REGION Network 3: Cylinder Selection ( Domestic / Commercial )
   // We have to receive from FIFO Entry-
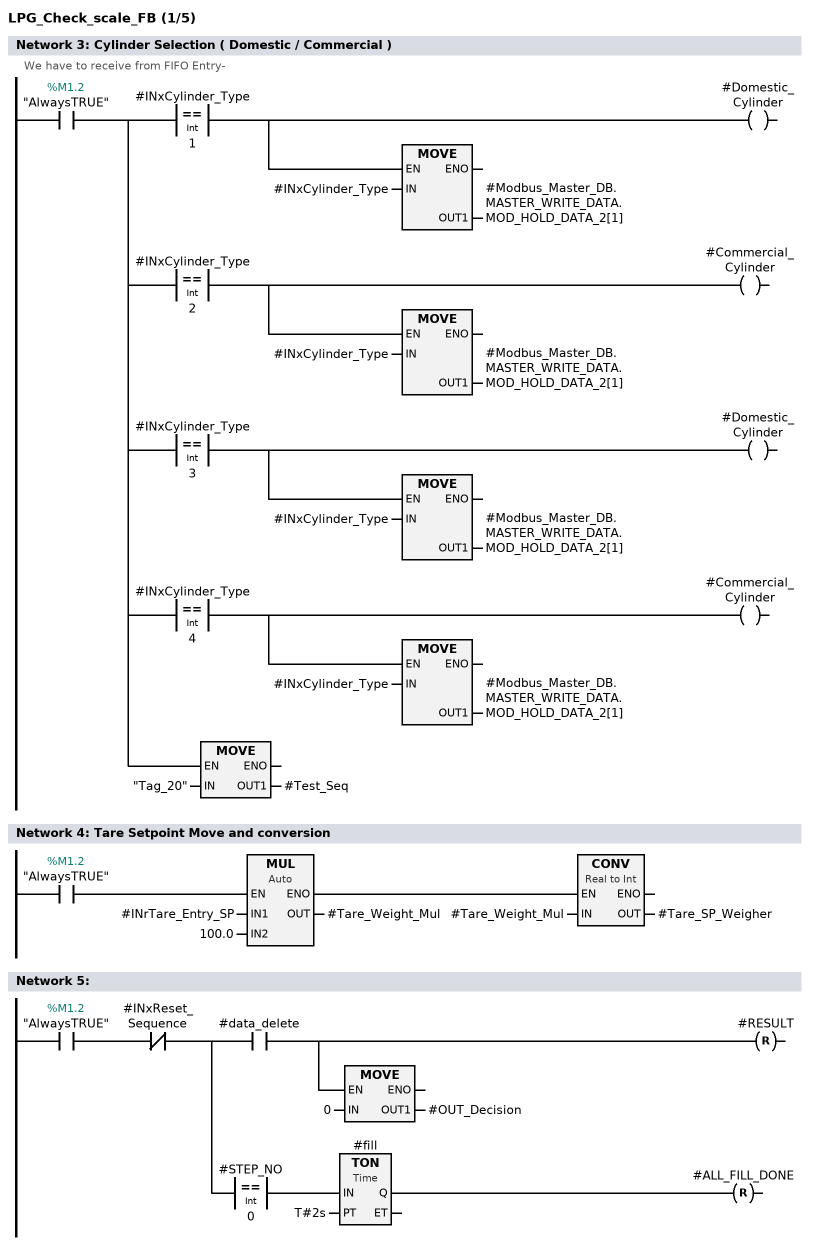
   RUNG wire#powerrail
      Contact( "AlwaysTRUE" )
      wire#w1
      { S7_Templates := "SrcType := Int" } EQ_Contact(in1 := #INxCylinder_Type, in2 := 1)
      wire#w2
      Coil( #Domestic_Cylinder )
   END_RUNG
   RUNG wire#w2
      Move(in := #INxCylinder_Type, out1 => #Modbus_Master_DB.MASTER_WRITE_DATA.MOD_HOLD_DATA_2[1])
   END_RUNG
   RUNG wire#w1
      { S7_Templates := "SrcType := Int" } EQ_Contact(in1 := #INxCylinder_Type, in2 := 2)
      wire#w3
      Coil( #Commercial_Cylinder )
   END_RUNG
   RUNG wire#w3
      Move(in := #INxCylinder_Type, out1 => #Modbus_Master_DB.MASTER_WRITE_DATA.MOD_HOLD_DATA_2[1])
   END_RUNG
   RUNG wire#w1
      { S7_Templates := "SrcType := Int" } EQ_Contact(in1 := #INxCylinder_Type, in2 := 3)
      wire#w4
      Coil( #Domestic_Cylinder )
   END_RUNG
   RUNG wire#w4
      Move(in := #INxCylinder_Type, out1 => #Modbus_Master_DB.MASTER_WRITE_DATA.MOD_HOLD_DATA_2[1])
   END_RUNG
   RUNG wire#w1
      { S7_Templates := "SrcType := Int" } EQ_Contact(in1 := #INxCylinder_Type, in2 := 4)
      wire#w5
      Coil( #Commercial_Cylinder )
   END_RUNG
   RUNG wire#w5
      Move(in := #INxCylinder_Type, out1 => #Modbus_Master_DB.MASTER_WRITE_DATA.MOD_HOLD_DATA_2[1])
   END_RUNG
   RUNG wire#w1
      Move(in := "Tag_20", out1 => #Test_Seq)
   END_RUNG
   // the same network as SCL:
   #Domestic_Cylinder := "AlwaysTRUE" AND (#INxCylinder_Type = 1);
   IF #Domestic_Cylinder THEN
       #Modbus_Master_DB.MASTER_WRITE_DATA.MOD_HOLD_DATA_2[1] := #INxCylinder_Type;
   END_IF;
   #Commercial_Cylinder := "AlwaysTRUE" AND (#INxCylinder_Type = 2);
   IF #Commercial_Cylinder THEN
       #Modbus_Master_DB.MASTER_WRITE_DATA.MOD_HOLD_DATA_2[1] := #INxCylinder_Type;
   END_IF;
   #Domestic_Cylinder := "AlwaysTRUE" AND (#INxCylinder_Type = 3);
   IF #Domestic_Cylinder THEN
       #Modbus_Master_DB.MASTER_WRITE_DATA.MOD_HOLD_DATA_2[1] := #INxCylinder_Type;
   END_IF;
   #Commercial_Cylinder := "AlwaysTRUE" AND (#INxCylinder_Type = 4);
   IF #Commercial_Cylinder THEN
       #Modbus_Master_DB.MASTER_WRITE_DATA.MOD_HOLD_DATA_2[1] := #INxCylinder_Type;
   END_IF;
   IF "AlwaysTRUE" THEN #Test_Seq := "Tag_20"; END_IF;
END_REGION

REGION Network 4: Tare Setpoint Move and conversion
   RUNG wire#powerrail
      Contact( "AlwaysTRUE" )
      Mul(in1 := #INrTare_Entry_SP, in2 := 100.0, out => #Tare_Weight_Mul)
      { S7_Templates := "[SrcType := Real, DestType := Int]" } Convert(in := #Tare_Weight_Mul, out => #Tare_SP_Weigher)
   END_RUNG
   // the same network as SCL:
   IF "AlwaysTRUE" THEN
       #Tare_Weight_Mul := #INrTare_Entry_SP * 100.0;
       #Tare_SP_Weigher := REAL_TO_INT(#Tare_Weight_Mul);
   END_IF;
END_REGION

REGION Network 5
   RUNG wire#powerrail
      Contact( "AlwaysTRUE" )
      I_Contact( #INxReset_Sequence )
      wire#w1
      Contact( #data_delete )
      wire#w2
      R_Coil( #RESULT )
   END_RUNG
   RUNG wire#w2
      Move(in := 0, out1 => #OUT_Decision)
   END_RUNG
   RUNG wire#w1
      { S7_Templates := "SrcType := Int" } EQ_Contact(in1 := #STEP_NO, in2 := 0)
      { S7_Templates := "time_type := Time" } #fill.TON(pt := T#2s, et =>)
      R_Coil( #ALL_FILL_DONE )
   END_RUNG
   // the same network as SCL:
   #_w1 := "AlwaysTRUE" AND NOT #INxReset_Sequence;
   IF #_w1 AND #data_delete THEN
       #RESULT := FALSE;
       #OUT_Decision := 0;
   END_IF;
   #fill(IN := #_w1 AND (#STEP_NO = 0), PT := T#2s);   // TON
   IF #fill.Q THEN #ALL_FILL_DONE := FALSE; END_IF;
END_REGION

REGION Network 6: Cylinder Selection
   // Cylinder Selection will write the logic later
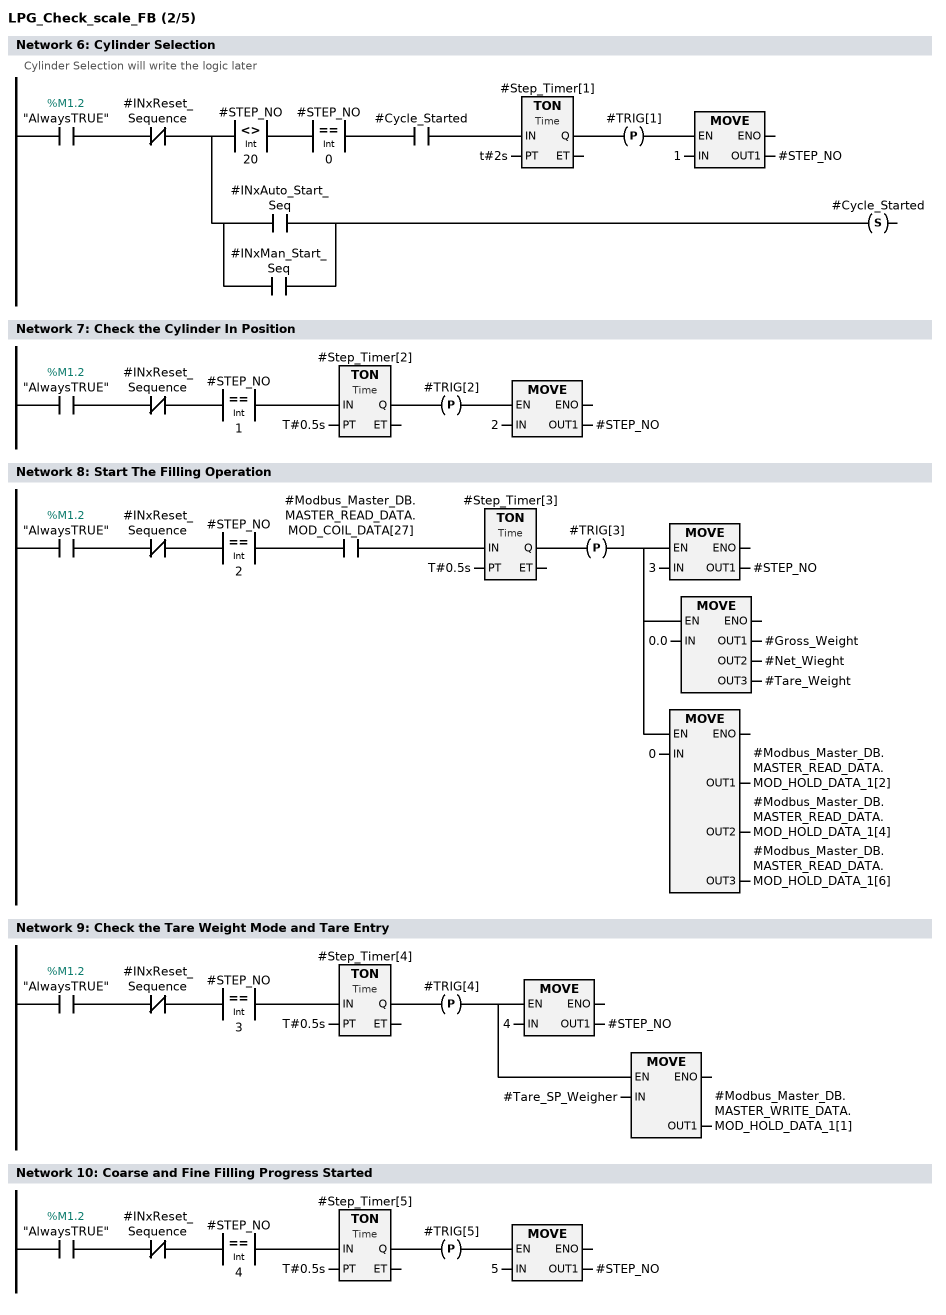
   RUNG wire#powerrail
      Contact( "AlwaysTRUE" )
      I_Contact( #INxReset_Sequence )
      wire#w1
      { S7_Templates := "SrcType := Int" } NE_Contact(in1 := #STEP_NO, in2 := 20)
      { S7_Templates := "SrcType := Int" } EQ_Contact(in1 := #STEP_NO, in2 := 0)
      Contact( #Cycle_Started )
      { S7_Templates := "time_type := Time" } #Step_Timer[1].TON(pt := t#2s, et =>)
      P_Trig( #TRIG[1] )
      Move(in := 1, out1 => #STEP_NO)
   END_RUNG
   RUNG wire#w1
      Contact( #INxAuto_Start_Seq )
      wire#w2
      S_Coil( #Cycle_Started )
   END_RUNG
   RUNG wire#w1
      Contact( #INxMan_Start_Seq )
   END_RUNG wire#w2
   // the same network as SCL:
   #_w1 := "AlwaysTRUE" AND NOT #INxReset_Sequence;
   #Step_Timer[1].TON(IN := #_w1 AND (#STEP_NO <> 20) AND (#STEP_NO = 0) AND #Cycle_Started, PT := t#2s);
   #_w2 := #Step_Timer[1].Q AND NOT #TRIG[1];   // rising edge
   #TRIG[1] := #Step_Timer[1].Q;
   IF #_w2 THEN #STEP_NO := 1; END_IF;
   IF #_w1 AND (#INxAuto_Start_Seq OR #INxMan_Start_Seq) THEN #Cycle_Started := TRUE; END_IF;
END_REGION

REGION Network 7: Check the Cylinder In Position
   RUNG wire#powerrail
      Contact( "AlwaysTRUE" )
      I_Contact( #INxReset_Sequence )
      { S7_Templates := "SrcType := Int" } EQ_Contact(in1 := #STEP_NO, in2 := 1)
      { S7_Templates := "time_type := Time" } #Step_Timer[2].TON(pt := T#0.5s, et =>)
      P_Trig( #TRIG[2] )
      Move(in := 2, out1 => #STEP_NO)
   END_RUNG
   // the same network as SCL:
   #Step_Timer[2].TON(IN := "AlwaysTRUE" AND NOT #INxReset_Sequence AND (#STEP_NO = 1), PT := T#0.5s);
   #_w1 := #Step_Timer[2].Q AND NOT #TRIG[2];   // rising edge
   #TRIG[2] := #Step_Timer[2].Q;
   IF #_w1 THEN #STEP_NO := 2; END_IF;
END_REGION

REGION Network 8: Start The Filling Operation
   RUNG wire#powerrail
      Contact( "AlwaysTRUE" )
      I_Contact( #INxReset_Sequence )
      { S7_Templates := "SrcType := Int" } EQ_Contact(in1 := #STEP_NO, in2 := 2)
      Contact( #Modbus_Master_DB.MASTER_READ_DATA.MOD_COIL_DATA[27] )
      { S7_Templates := "time_type := Time" } #Step_Timer[3].TON(pt := T#0.5s, et =>)
      P_Trig( #TRIG[3] )
      wire#w1
      Move(in := 3, out1 => #STEP_NO)
   END_RUNG
   RUNG wire#w1
      Move(in := 0.0, out1 => #Gross_Weight, out2 => #Net_Wieght, out3 => #Tare_Weight)
   END_RUNG
   RUNG wire#w1
      Move(in := 0, out1 => #Modbus_Master_DB.MASTER_READ_DATA.MOD_HOLD_DATA_1[2], out2 => #Modbus_Master_DB.MASTER_READ_DATA.MOD_HOLD_DATA_1[4], out3 => #Modbus_Master_DB.MASTER_READ_DATA.MOD_HOLD_DATA_1[6])
   END_RUNG
   // the same network as SCL:
   #Step_Timer[3].TON(IN := "AlwaysTRUE" AND NOT #INxReset_Sequence AND (#STEP_NO = 2) AND #Modbus_Master_DB.MASTER_READ_DATA.MOD_COIL_DATA[27],
                      PT := T#0.5s);
   #_w1 := #Step_Timer[3].Q AND NOT #TRIG[3];   // rising edge
   #TRIG[3] := #Step_Timer[3].Q;
   IF #_w1 THEN
       #STEP_NO := 3;
       #Gross_Weight := 0.0;
       #Net_Wieght := 0.0;
       #Tare_Weight := 0.0;
       #Modbus_Master_DB.MASTER_READ_DATA.MOD_HOLD_DATA_1[2] := 0;
       #Modbus_Master_DB.MASTER_READ_DATA.MOD_HOLD_DATA_1[4] := 0;
       #Modbus_Master_DB.MASTER_READ_DATA.MOD_HOLD_DATA_1[6] := 0;
   END_IF;
END_REGION

REGION Network 9: Check the Tare Weight Mode and Tare Entry
   RUNG wire#powerrail
      Contact( "AlwaysTRUE" )
      I_Contact( #INxReset_Sequence )
      { S7_Templates := "SrcType := Int" } EQ_Contact(in1 := #STEP_NO, in2 := 3)
      { S7_Templates := "time_type := Time" } #Step_Timer[4].TON(pt := T#0.5s, et =>)
      P_Trig( #TRIG[4] )
      wire#w1
      Move(in := 4, out1 => #STEP_NO)
   END_RUNG
   RUNG wire#w1
      Move(in := #Tare_SP_Weigher, out1 => #Modbus_Master_DB.MASTER_WRITE_DATA.MOD_HOLD_DATA_1[1])
   END_RUNG
   // the same network as SCL:
   #Step_Timer[4].TON(IN := "AlwaysTRUE" AND NOT #INxReset_Sequence AND (#STEP_NO = 3), PT := T#0.5s);
   #_w1 := #Step_Timer[4].Q AND NOT #TRIG[4];   // rising edge
   #TRIG[4] := #Step_Timer[4].Q;
   IF #_w1 THEN
       #STEP_NO := 4;
       #Modbus_Master_DB.MASTER_WRITE_DATA.MOD_HOLD_DATA_1[1] := #Tare_SP_Weigher;
   END_IF;
END_REGION

REGION Network 10: Coarse and Fine Filling Progress Started
   RUNG wire#powerrail
      Contact( "AlwaysTRUE" )
      I_Contact( #INxReset_Sequence )
      { S7_Templates := "SrcType := Int" } EQ_Contact(in1 := #STEP_NO, in2 := 4)
      { S7_Templates := "time_type := Time" } #Step_Timer[5].TON(pt := T#0.5s, et =>)
      P_Trig( #TRIG[5] )
      Move(in := 5, out1 => #STEP_NO)
   END_RUNG
   // the same network as SCL:
   #Step_Timer[5].TON(IN := "AlwaysTRUE" AND NOT #INxReset_Sequence AND (#STEP_NO = 4), PT := T#0.5s);
   #_w1 := #Step_Timer[5].Q AND NOT #TRIG[5];   // rising edge
   #TRIG[5] := #Step_Timer[5].Q;
   IF #_w1 THEN #STEP_NO := 5; END_IF;
END_REGION

REGION Network 11: Coarse Filling Completed
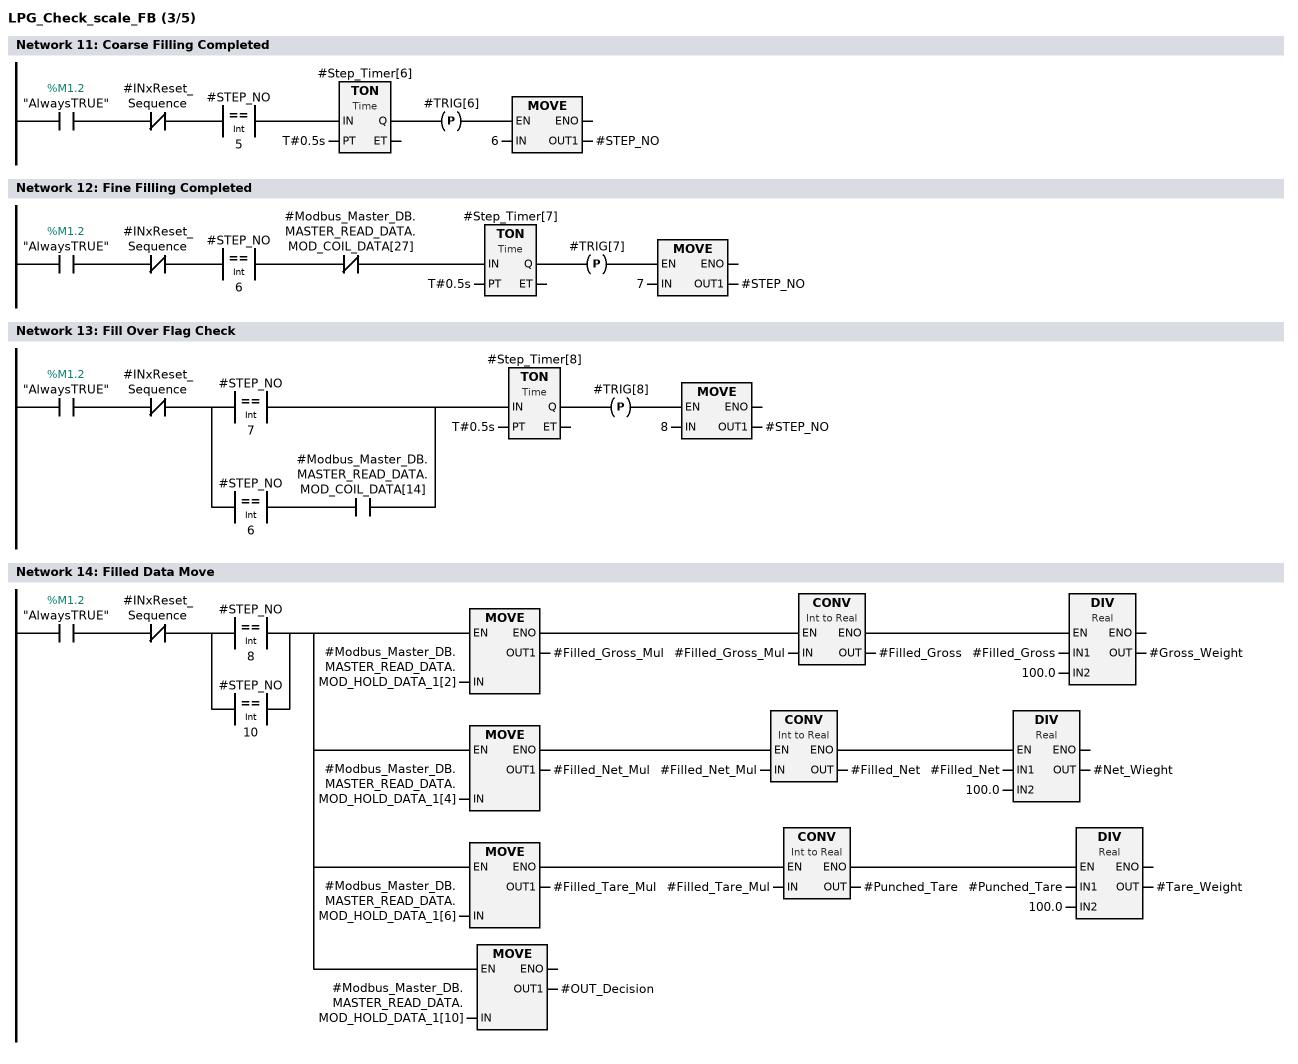
   RUNG wire#powerrail
      Contact( "AlwaysTRUE" )
      I_Contact( #INxReset_Sequence )
      { S7_Templates := "SrcType := Int" } EQ_Contact(in1 := #STEP_NO, in2 := 5)
      { S7_Templates := "time_type := Time" } #Step_Timer[6].TON(pt := T#0.5s, et =>)
      P_Trig( #TRIG[6] )
      Move(in := 6, out1 => #STEP_NO)
   END_RUNG
   // the same network as SCL:
   #Step_Timer[6].TON(IN := "AlwaysTRUE" AND NOT #INxReset_Sequence AND (#STEP_NO = 5), PT := T#0.5s);
   #_w1 := #Step_Timer[6].Q AND NOT #TRIG[6];   // rising edge
   #TRIG[6] := #Step_Timer[6].Q;
   IF #_w1 THEN #STEP_NO := 6; END_IF;
END_REGION

REGION Network 12: Fine Filling Completed
   RUNG wire#powerrail
      Contact( "AlwaysTRUE" )
      I_Contact( #INxReset_Sequence )
      { S7_Templates := "SrcType := Int" } EQ_Contact(in1 := #STEP_NO, in2 := 6)
      I_Contact( #Modbus_Master_DB.MASTER_READ_DATA.MOD_COIL_DATA[27] )
      { S7_Templates := "time_type := Time" } #Step_Timer[7].TON(pt := T#0.5s, et =>)
      P_Trig( #TRIG[7] )
      Move(in := 7, out1 => #STEP_NO)
   END_RUNG
   // the same network as SCL:
   #Step_Timer[7].TON(IN := "AlwaysTRUE" AND NOT #INxReset_Sequence AND (#STEP_NO = 6) AND NOT #Modbus_Master_DB.MASTER_READ_DATA.MOD_COIL_DATA[27],
                      PT := T#0.5s);
   #_w1 := #Step_Timer[7].Q AND NOT #TRIG[7];   // rising edge
   #TRIG[7] := #Step_Timer[7].Q;
   IF #_w1 THEN #STEP_NO := 7; END_IF;
END_REGION

REGION Network 13: Fill Over Flag Check
   RUNG wire#powerrail
      Contact( "AlwaysTRUE" )
      I_Contact( #INxReset_Sequence )
      wire#w1
      { S7_Templates := "SrcType := Int" } EQ_Contact(in1 := #STEP_NO, in2 := 7)
      wire#w2
      { S7_Templates := "time_type := Time" } #Step_Timer[8].TON(pt := T#0.5s, et =>)
      P_Trig( #TRIG[8] )
      Move(in := 8, out1 => #STEP_NO)
   END_RUNG
   RUNG wire#w1
      { S7_Templates := "SrcType := Int" } EQ_Contact(in1 := #STEP_NO, in2 := 6)
      Contact( #Modbus_Master_DB.MASTER_READ_DATA.MOD_COIL_DATA[14] )
   END_RUNG wire#w2
   // the same network as SCL:
   #Step_Timer[8].TON(IN := "AlwaysTRUE" AND NOT #INxReset_Sequence AND ((#STEP_NO = 7) OR ((#STEP_NO = 6) AND #Modbus_Master_DB.MASTER_READ_DATA.MOD_COIL_DATA[14])),
                      PT := T#0.5s);
   #_w1 := #Step_Timer[8].Q AND NOT #TRIG[8];   // rising edge
   #TRIG[8] := #Step_Timer[8].Q;
   IF #_w1 THEN #STEP_NO := 8; END_IF;
END_REGION

REGION Network 14: Filled Data Move
   RUNG wire#powerrail
      Contact( "AlwaysTRUE" )
      I_Contact( #INxReset_Sequence )
      wire#w1
      { S7_Templates := "SrcType := Int" } EQ_Contact(in1 := #STEP_NO, in2 := 8)
      wire#w2
      Move(in := #Modbus_Master_DB.MASTER_READ_DATA.MOD_HOLD_DATA_1[2], out1 => #Filled_Gross_Mul)
      { S7_Templates := "[SrcType := Int, DestType := Real]" } Convert(in := #Filled_Gross_Mul, out => #Filled_Gross)
      { S7_Templates := "SrcType := Real" } Div(in1 := #Filled_Gross, in2 := 100.0, out => #Gross_Weight)
   END_RUNG
   RUNG wire#w1
      { S7_Templates := "SrcType := Int" } EQ_Contact(in1 := #STEP_NO, in2 := 10)
   END_RUNG wire#w2
   RUNG wire#w2
      Move(in := #Modbus_Master_DB.MASTER_READ_DATA.MOD_HOLD_DATA_1[4], out1 => #Filled_Net_Mul)
      { S7_Templates := "[SrcType := Int, DestType := Real]" } Convert(in := #Filled_Net_Mul, out => #Filled_Net)
      { S7_Templates := "SrcType := Real" } Div(in1 := #Filled_Net, in2 := 100.0, out => #Net_Wieght)
   END_RUNG
   RUNG wire#w2
      Move(in := #Modbus_Master_DB.MASTER_READ_DATA.MOD_HOLD_DATA_1[6], out1 => #Filled_Tare_Mul)
      { S7_Templates := "[SrcType := Int, DestType := Real]" } Convert(in := #Filled_Tare_Mul, out => #Punched_Tare)
      { S7_Templates := "SrcType := Real" } Div(in1 := #Punched_Tare, in2 := 100.0, out => #Tare_Weight)
   END_RUNG
   RUNG wire#w2
      Move(in := #Modbus_Master_DB.MASTER_READ_DATA.MOD_HOLD_DATA_1[10], out1 => #OUT_Decision)
   END_RUNG
   // the same network as SCL:
   IF "AlwaysTRUE" AND NOT #INxReset_Sequence AND ((#STEP_NO = 8) OR (#STEP_NO = 10)) THEN
       #Filled_Gross_Mul := #Modbus_Master_DB.MASTER_READ_DATA.MOD_HOLD_DATA_1[2];
       #Filled_Gross := INT_TO_REAL(#Filled_Gross_Mul);
       #Gross_Weight := #Filled_Gross / 100.0;
       #Filled_Net_Mul := #Modbus_Master_DB.MASTER_READ_DATA.MOD_HOLD_DATA_1[4];
       #Filled_Net := INT_TO_REAL(#Filled_Net_Mul);
       #Net_Wieght := #Filled_Net / 100.0;
       #Filled_Tare_Mul := #Modbus_Master_DB.MASTER_READ_DATA.MOD_HOLD_DATA_1[6];
       #Punched_Tare := INT_TO_REAL(#Filled_Tare_Mul);
       #Tare_Weight := #Punched_Tare / 100.0;
       #OUT_Decision := #Modbus_Master_DB.MASTER_READ_DATA.MOD_HOLD_DATA_1[10];
   END_IF;
END_REGION

REGION Network 15: Filling Operation Complete
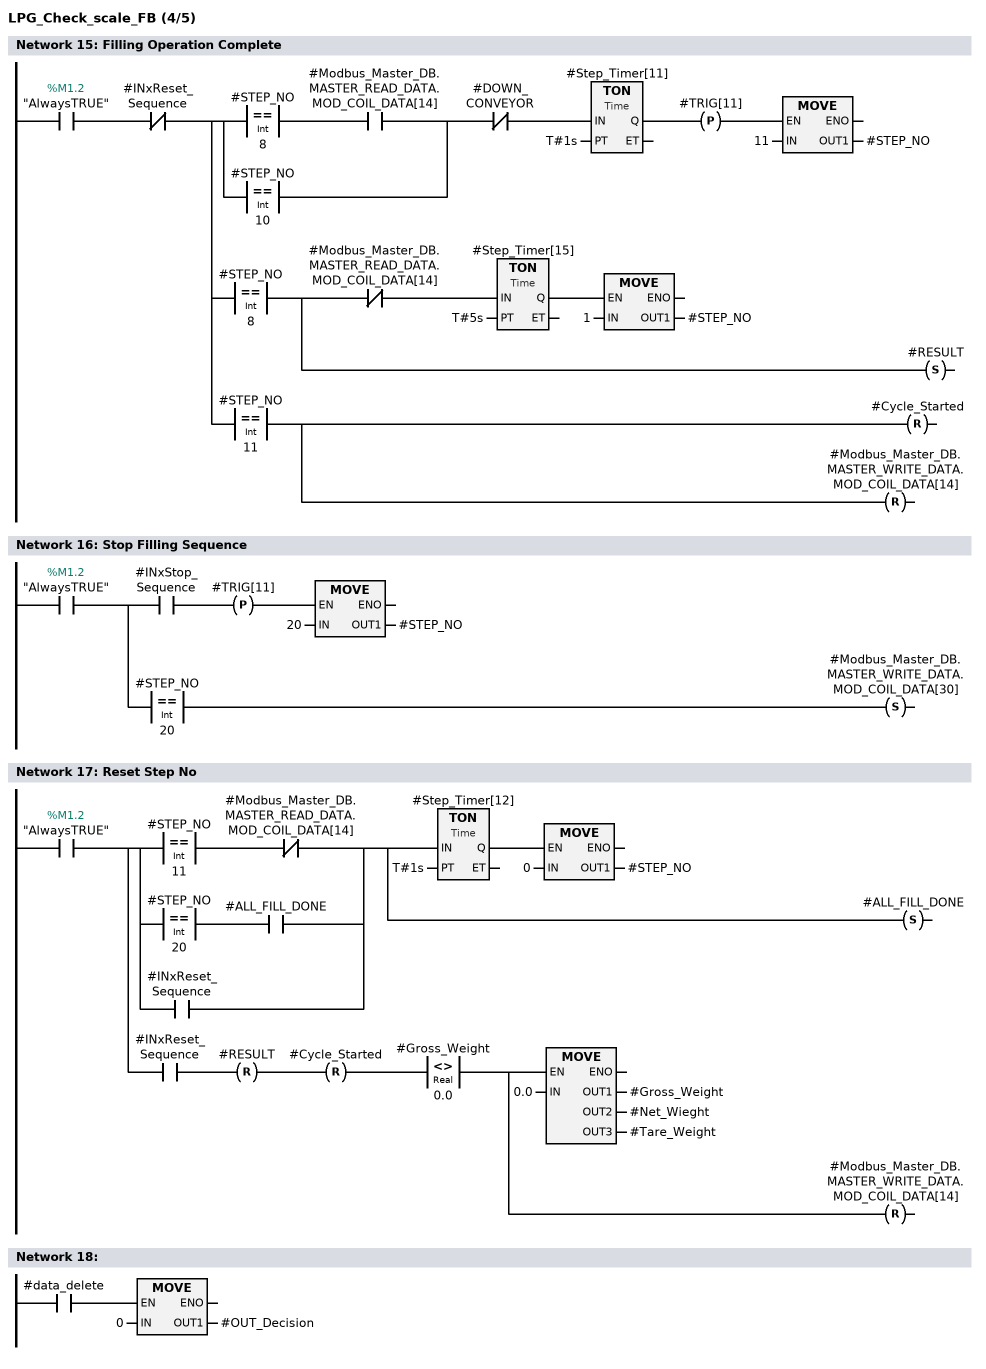
   RUNG wire#powerrail
      Contact( "AlwaysTRUE" )
      I_Contact( #INxReset_Sequence )
      wire#w1
      { S7_Templates := "SrcType := Int" } EQ_Contact(in1 := #STEP_NO, in2 := 8)
      Contact( #Modbus_Master_DB.MASTER_READ_DATA.MOD_COIL_DATA[14] )
      wire#w2
      I_Contact( #DOWN_CONVEYOR )
      { S7_Templates := "time_type := Time" } #Step_Timer[11].TON(pt := T#1s, et =>)
      P_Trig( #TRIG[11] )
      Move(in := 11, out1 => #STEP_NO)
   END_RUNG
   RUNG wire#w1
      { S7_Templates := "SrcType := Int" } EQ_Contact(in1 := #STEP_NO, in2 := 10)
   END_RUNG wire#w2
   RUNG wire#w1
      { S7_Templates := "SrcType := Int" } EQ_Contact(in1 := #STEP_NO, in2 := 8)
      wire#w3
      I_Contact( #Modbus_Master_DB.MASTER_READ_DATA.MOD_COIL_DATA[14] )
      { S7_Templates := "time_type := Time" } #Step_Timer[15].TON(pt := T#5s, et =>)
      Move(in := 1, out1 => #STEP_NO)
   END_RUNG
   RUNG wire#w3
      S_Coil( #RESULT )
   END_RUNG
   RUNG wire#w1
      { S7_Templates := "SrcType := Int" } EQ_Contact(in1 := #STEP_NO, in2 := 11)
      wire#w4
      R_Coil( #Cycle_Started )
   END_RUNG
   RUNG wire#w4
      R_Coil( #Modbus_Master_DB.MASTER_WRITE_DATA.MOD_COIL_DATA[14] )
   END_RUNG
   // the same network as SCL:
   #_w1 := "AlwaysTRUE" AND NOT #INxReset_Sequence;
   #Step_Timer[11].TON(IN := #_w1 AND (((#STEP_NO = 8) AND #Modbus_Master_DB.MASTER_READ_DATA.MOD_COIL_DATA[14]) OR (#STEP_NO = 10)) AND NOT #DOWN_CONVEYOR,
                       PT := T#1s);
   #_w2 := #Step_Timer[11].Q AND NOT #TRIG[11];   // rising edge
   #TRIG[11] := #Step_Timer[11].Q;
   IF #_w2 THEN #STEP_NO := 11; END_IF;
   #_w3 := #_w1 AND (#STEP_NO = 8);
   #Step_Timer[15].TON(IN := #_w3 AND NOT #Modbus_Master_DB.MASTER_READ_DATA.MOD_COIL_DATA[14], PT := T#5s);
   IF #Step_Timer[15].Q THEN #STEP_NO := 1; END_IF;
   IF #_w3 THEN #RESULT := TRUE; END_IF;
   IF #_w1 AND (#STEP_NO = 11) THEN
       #Cycle_Started := FALSE;
       #Modbus_Master_DB.MASTER_WRITE_DATA.MOD_COIL_DATA[14] := FALSE;
   END_IF;
END_REGION

REGION Network 16: Stop Filling Sequence
   RUNG wire#powerrail
      Contact( "AlwaysTRUE" )
      wire#w1
      Contact( #INxStop_Sequence )
      P_Trig( #TRIG[11] )
      Move(in := 20, out1 => #STEP_NO)
   END_RUNG
   RUNG wire#w1
      { S7_Templates := "SrcType := Int" } EQ_Contact(in1 := #STEP_NO, in2 := 20)
      S_Coil( #Modbus_Master_DB.MASTER_WRITE_DATA.MOD_COIL_DATA[30] )
   END_RUNG
   // the same network as SCL:
   #_w1 := "AlwaysTRUE" AND #INxStop_Sequence;
   #_w2 := #_w1 AND NOT #TRIG[11];   // rising edge
   #TRIG[11] := #_w1;
   IF #_w2 THEN #STEP_NO := 20; END_IF;
   IF "AlwaysTRUE" AND (#STEP_NO = 20) THEN
       #Modbus_Master_DB.MASTER_WRITE_DATA.MOD_COIL_DATA[30] := TRUE;
   END_IF;
END_REGION

REGION Network 17: Reset Step No
   RUNG wire#powerrail
      Contact( "AlwaysTRUE" )
      wire#w1
      { S7_Templates := "SrcType := Int" } EQ_Contact(in1 := #STEP_NO, in2 := 11)
      I_Contact( #Modbus_Master_DB.MASTER_READ_DATA.MOD_COIL_DATA[14] )
      wire#w2
      { S7_Templates := "time_type := Time" } #Step_Timer[12].TON(pt := T#1s, et =>)
      Move(in := 0, out1 => #STEP_NO)
   END_RUNG
   RUNG wire#w1
      { S7_Templates := "SrcType := Int" } EQ_Contact(in1 := #STEP_NO, in2 := 20)
      Contact( #ALL_FILL_DONE )
   END_RUNG wire#w2
   RUNG wire#w1
      Contact( #INxReset_Sequence )
   END_RUNG wire#w2
   RUNG wire#w2
      S_Coil( #ALL_FILL_DONE )
   END_RUNG
   RUNG wire#w1
      Contact( #INxReset_Sequence )
      R_Coil( #RESULT )
      R_Coil( #Cycle_Started )
      { S7_Templates := "SrcType := Real" } NE_Contact(in1 := #Gross_Weight, in2 := 0.0)
      wire#w3
      Move(in := 0.0, out1 => #Gross_Weight, out2 => #Net_Wieght, out3 => #Tare_Weight)
   END_RUNG
   RUNG wire#w3
      R_Coil( #Modbus_Master_DB.MASTER_WRITE_DATA.MOD_COIL_DATA[14] )
   END_RUNG
   // the same network as SCL:
   #_w1 := "AlwaysTRUE" AND (((#STEP_NO = 11) AND NOT #Modbus_Master_DB.MASTER_READ_DATA.MOD_COIL_DATA[14]) OR ((#STEP_NO = 20) AND #ALL_FILL_DONE) OR #INxReset_Sequence);
   #Step_Timer[12].TON(IN := #_w1, PT := T#1s);
   IF #Step_Timer[12].Q THEN #STEP_NO := 0; END_IF;
   IF #_w1 THEN #ALL_FILL_DONE := TRUE; END_IF;
   #_w2 := "AlwaysTRUE" AND #INxReset_Sequence;
   IF #_w2 THEN
       #RESULT := FALSE;
       #Cycle_Started := FALSE;
   END_IF;
   #_w3 := #_w2 AND (#Gross_Weight <> 0.0);
   IF #_w3 THEN
       #Gross_Weight := 0.0;
       #Net_Wieght := 0.0;
       #Tare_Weight := 0.0;
       #Modbus_Master_DB.MASTER_WRITE_DATA.MOD_COIL_DATA[14] := FALSE;
   END_IF;
END_REGION

REGION Network 18
   RUNG wire#powerrail
      Contact( #data_delete )
      Move(in := 0, out1 => #OUT_Decision)
   END_RUNG
   // the same network as SCL:
   IF #data_delete THEN #OUT_Decision := 0; END_IF;
END_REGION

REGION Network 19: Output Mapping
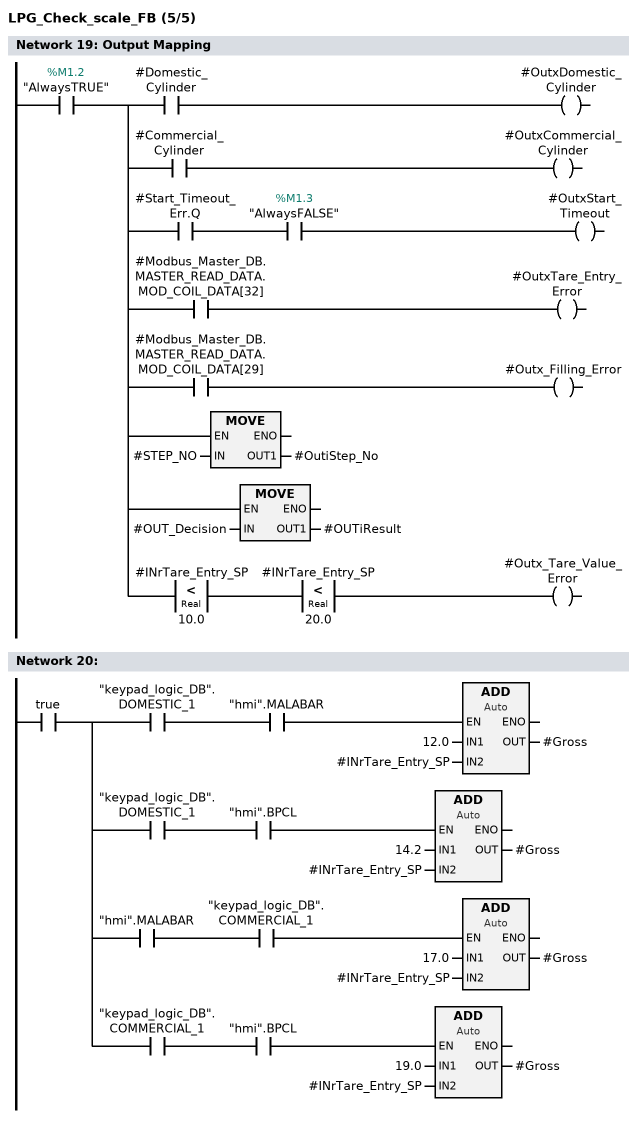
   RUNG wire#powerrail
      Contact( "AlwaysTRUE" )
      wire#w1
      Contact( #Domestic_Cylinder )
      Coil( #OutxDomestic_Cylinder )
   END_RUNG
   RUNG wire#w1
      Contact( #Commercial_Cylinder )
      Coil( #OutxCommercial_Cylinder )
   END_RUNG
   RUNG wire#w1
      Contact( #Start_Timeout_Err.Q )
      Contact( "AlwaysFALSE" )
      Coil( #OutxStart_Timeout )
   END_RUNG
   RUNG wire#w1
      Contact( #Modbus_Master_DB.MASTER_READ_DATA.MOD_COIL_DATA[32] )
      Coil( #OutxTare_Entry_Error )
   END_RUNG
   RUNG wire#w1
      Contact( #Modbus_Master_DB.MASTER_READ_DATA.MOD_COIL_DATA[29] )
      Coil( #Outx_Filling_Error )
   END_RUNG
   RUNG wire#w1
      Move(in := #STEP_NO, out1 => #OutiStep_No)
   END_RUNG
   RUNG wire#w1
      Move(in := #OUT_Decision, out1 => #OUTiResult)
   END_RUNG
   RUNG wire#w1
      { S7_Templates := "SrcType := Real" } LT_Contact(in1 := #INrTare_Entry_SP, in2 := 10.0)
      { S7_Templates := "SrcType := Real" } LT_Contact(in1 := #INrTare_Entry_SP, in2 := 20.0)
      Coil( #Outx_Tare_Value_Error )
   END_RUNG
   // the same network as SCL:
   #OutxDomestic_Cylinder := "AlwaysTRUE" AND #Domestic_Cylinder;
   #OutxCommercial_Cylinder := "AlwaysTRUE" AND #Commercial_Cylinder;
   #OutxStart_Timeout := "AlwaysTRUE" AND #Start_Timeout_Err.Q AND "AlwaysFALSE";
   #OutxTare_Entry_Error := "AlwaysTRUE" AND #Modbus_Master_DB.MASTER_READ_DATA.MOD_COIL_DATA[32];
   #Outx_Filling_Error := "AlwaysTRUE" AND #Modbus_Master_DB.MASTER_READ_DATA.MOD_COIL_DATA[29];
   IF "AlwaysTRUE" THEN
       #OutiStep_No := #STEP_NO;
       #OUTiResult := #OUT_Decision;
   END_IF;
   #Outx_Tare_Value_Error := "AlwaysTRUE" AND (#INrTare_Entry_SP < 10.0) AND (#INrTare_Entry_SP < 20.0);
END_REGION

REGION Network 20
   RUNG wire#powerrail
      Contact( true )
      wire#w1
      Contact( "keypad_logic_DB".DOMESTIC_1 )
      Contact( "hmi".MALABAR )
      Add(in1 := 12.0, in2 := #INrTare_Entry_SP, out => #Gross)
   END_RUNG
   RUNG wire#w1
      Contact( "keypad_logic_DB".DOMESTIC_1 )
      Contact( "hmi".BPCL )
      Add(in1 := 14.2, in2 := #INrTare_Entry_SP, out => #Gross)
   END_RUNG
   RUNG wire#w1
      Contact( "hmi".MALABAR )
      Contact( "keypad_logic_DB".COMMERCIAL_1 )
      Add(in1 := 17.0, in2 := #INrTare_Entry_SP, out => #Gross)
   END_RUNG
   RUNG wire#w1
      Contact( "keypad_logic_DB".COMMERCIAL_1 )
      Contact( "hmi".BPCL )
      Add(in1 := 19.0, in2 := #INrTare_Entry_SP, out => #Gross)
   END_RUNG
   // the same network as SCL:
   IF true AND "keypad_logic_DB".DOMESTIC_1 AND "hmi".MALABAR THEN
       #Gross := 12.0 + #INrTare_Entry_SP;
   END_IF;
   IF true AND "keypad_logic_DB".DOMESTIC_1 AND "hmi".BPCL THEN #Gross := 14.2 + #INrTare_Entry_SP; END_IF;
   IF true AND "hmi".MALABAR AND "keypad_logic_DB".COMMERCIAL_1 THEN
       #Gross := 17.0 + #INrTare_Entry_SP;
   END_IF;
   IF true AND "keypad_logic_DB".COMMERCIAL_1 AND "hmi".BPCL THEN #Gross := 19.0 + #INrTare_Entry_SP; END_IF;
END_REGION
END_FUNCTION_BLOCK

FUNCTION_BLOCK "TCP_CHECK_SCALE"   // FB172, LAD
{ S7_Optimized_Access := 'TRUE' }
VERSION : 0.1
// stored: AutoNumber false, IsIECCheckEnabled false, IsRetainMemResEnabled false, MemoryReserve 100, SetENOAutomatically false, UDAEnableTagReadback false
   VAR_OUTPUT
      Modbus_Busy : Bool;
   END_VAR
   VAR_IN_OUT
      Mod_TCP_Setup : "Mod_TCP_Data";
      LPG_Fill_Data : "LPG_FILL_DATA_1";
   END_VAR
   VAR
      PStep_No : Struct
         MASTER_STEP_NO : "Master_Step_No";
      END_STRUCT;
      Write_Bit_Address : Int;
      TRIG : Array[1..100] of Bool;
      MOD_MASTER1_REQ : Array[1..10] of Bool;
      MOD_MASTER2_REQ : Array[1..10] of Bool;
      MOD_MASTER3_REQ : Array[1..10] of Bool;
      MOD_MASTER4_REQ : Array[1..10] of Bool;
      MOD_MASTER5_REQ : Array[1..10] of Bool;
      MOD_MASTER6_REQ : Array[1..10] of Bool;
      MAS_TRG_EXTN { S7_SetPoint := 'True'} : TOF_TIME;
      Tare_delay { S7_SetPoint := 'True'} : TON_TIME;
   END_VAR
   VAR_TEMP   // added for the SCL form of the ladder/FBD networks
      _w1 : Bool;
      _w2 : Bool;
      _w3 : Bool;
      _w4 : Bool;
   END_VAR
BEGIN

REGION Network 1: FILLING LINE-1 STATION-1
END_REGION

REGION Network 2: Write Master-1 Holding Register Request(Tare Weight Entry)
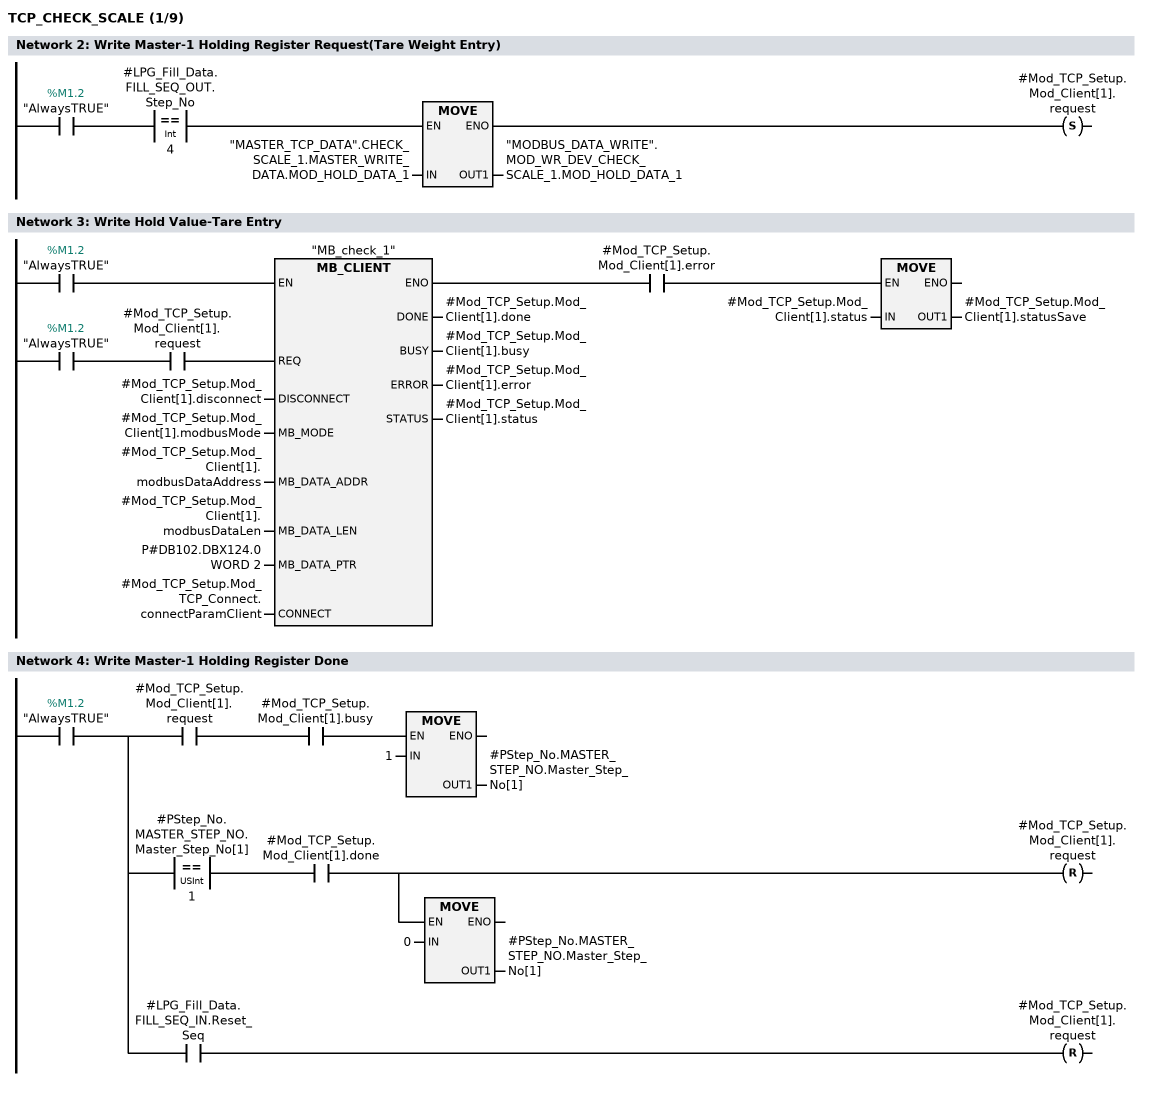
   RUNG wire#powerrail
      Contact( "AlwaysTRUE" )
      { S7_Templates := "SrcType := Int" } EQ_Contact(in1 := #LPG_Fill_Data.FILL_SEQ_OUT.Step_No, in2 := 4)
      Move(in := "MASTER_TCP_DATA".CHECK_SCALE_1.MASTER_WRITE_DATA.MOD_HOLD_DATA_1, out1 => "MODBUS_DATA_WRITE".MOD_WR_DEV_CHECK_SCALE_1.MOD_HOLD_DATA_1)
      S_Coil( #Mod_TCP_Setup.Mod_Client[1].request )
   END_RUNG
   // the same network as SCL:
   IF "AlwaysTRUE" AND (#LPG_Fill_Data.FILL_SEQ_OUT.Step_No = 4) THEN
       "MODBUS_DATA_WRITE".MOD_WR_DEV_CHECK_SCALE_1.MOD_HOLD_DATA_1 := "MASTER_TCP_DATA".CHECK_SCALE_1.MASTER_WRITE_DATA.MOD_HOLD_DATA_1;
       #Mod_TCP_Setup.Mod_Client[1].request := TRUE;
   END_IF;
END_REGION

REGION Network 3: Write Hold Value-Tare Entry
   RUNG wire#powerrail
      Contact( "AlwaysTRUE" )
      "MB_check_1".MB_CLIENT(REQ := wire#w1, DISCONNECT := #Mod_TCP_Setup.Mod_Client[1].disconnect, MB_MODE := #Mod_TCP_Setup.Mod_Client[1].modbusMode, MB_DATA_ADDR := #Mod_TCP_Setup.Mod_Client[1].modbusDataAddress, MB_DATA_LEN := #Mod_TCP_Setup.Mod_Client[1].modbusDataLen, MB_DATA_PTR := P#DB102.DBX124.0 WORD 2, CONNECT := #Mod_TCP_Setup.Mod_TCP_Connect.connectParamClient, DONE => #Mod_TCP_Setup.Mod_Client[1].done, BUSY => #Mod_TCP_Setup.Mod_Client[1].busy, ERROR => #Mod_TCP_Setup.Mod_Client[1].error, STATUS => #Mod_TCP_Setup.Mod_Client[1].status)
      Contact( #Mod_TCP_Setup.Mod_Client[1].error )
      Move(in := #Mod_TCP_Setup.Mod_Client[1].status, out1 => #Mod_TCP_Setup.Mod_Client[1].statusSave)
   END_RUNG
   RUNG wire#powerrail
      Contact( "AlwaysTRUE" )
      Contact( #Mod_TCP_Setup.Mod_Client[1].request )
   END_RUNG wire#w1
   // the same network as SCL:
   "MB_check_1"(EN := "AlwaysTRUE",   // MB_CLIENT
                REQ := "AlwaysTRUE" AND #Mod_TCP_Setup.Mod_Client[1].request,
                DISCONNECT := #Mod_TCP_Setup.Mod_Client[1].disconnect,
                MB_MODE := #Mod_TCP_Setup.Mod_Client[1].modbusMode,
                MB_DATA_ADDR := #Mod_TCP_Setup.Mod_Client[1].modbusDataAddress,
                MB_DATA_LEN := #Mod_TCP_Setup.Mod_Client[1].modbusDataLen,
                MB_DATA_PTR := P#DB102.DBX124.0 WORD 2,
                CONNECT := #Mod_TCP_Setup.Mod_TCP_Connect.connectParamClient,
                DONE => #Mod_TCP_Setup.Mod_Client[1].done,
                BUSY => #Mod_TCP_Setup.Mod_Client[1].busy,
                ERROR => #Mod_TCP_Setup.Mod_Client[1].error,
                STATUS => #Mod_TCP_Setup.Mod_Client[1].status,
                ENO => #_w1);
   IF #_w1 AND #Mod_TCP_Setup.Mod_Client[1].error THEN
       #Mod_TCP_Setup.Mod_Client[1].statusSave := #Mod_TCP_Setup.Mod_Client[1].status;
   END_IF;
END_REGION

REGION Network 4: Write Master-1 Holding Register Done
   RUNG wire#powerrail
      Contact( "AlwaysTRUE" )
      wire#w1
      Contact( #Mod_TCP_Setup.Mod_Client[1].request )
      Contact( #Mod_TCP_Setup.Mod_Client[1].busy )
      Move(in := 1, out1 => #PStep_No.MASTER_STEP_NO.Master_Step_No[1])
   END_RUNG
   RUNG wire#w1
      { S7_Templates := "SrcType := USInt" } EQ_Contact(in1 := #PStep_No.MASTER_STEP_NO.Master_Step_No[1], in2 := 1)
      Contact( #Mod_TCP_Setup.Mod_Client[1].done )
      wire#w2
      R_Coil( #Mod_TCP_Setup.Mod_Client[1].request )
   END_RUNG
   RUNG wire#w2
      Move(in := 0, out1 => #PStep_No.MASTER_STEP_NO.Master_Step_No[1])
   END_RUNG
   RUNG wire#w1
      Contact( #LPG_Fill_Data.FILL_SEQ_IN.Reset_Seq )
      R_Coil( #Mod_TCP_Setup.Mod_Client[1].request )
   END_RUNG
   // the same network as SCL:
   IF "AlwaysTRUE" AND #Mod_TCP_Setup.Mod_Client[1].request AND #Mod_TCP_Setup.Mod_Client[1].busy THEN
       #PStep_No.MASTER_STEP_NO.Master_Step_No[1] := 1;
   END_IF;
   #_w1 := "AlwaysTRUE" AND (#PStep_No.MASTER_STEP_NO.Master_Step_No[1] = 1) AND #Mod_TCP_Setup.Mod_Client[1].done;
   IF #_w1 THEN
       #Mod_TCP_Setup.Mod_Client[1].request := FALSE;
       #PStep_No.MASTER_STEP_NO.Master_Step_No[1] := 0;
   END_IF;
   IF "AlwaysTRUE" AND #LPG_Fill_Data.FILL_SEQ_IN.Reset_Seq THEN
       #Mod_TCP_Setup.Mod_Client[1].request := FALSE;
   END_IF;
END_REGION

REGION Network 5: Modbus Master2 Read Request(Filled Data)
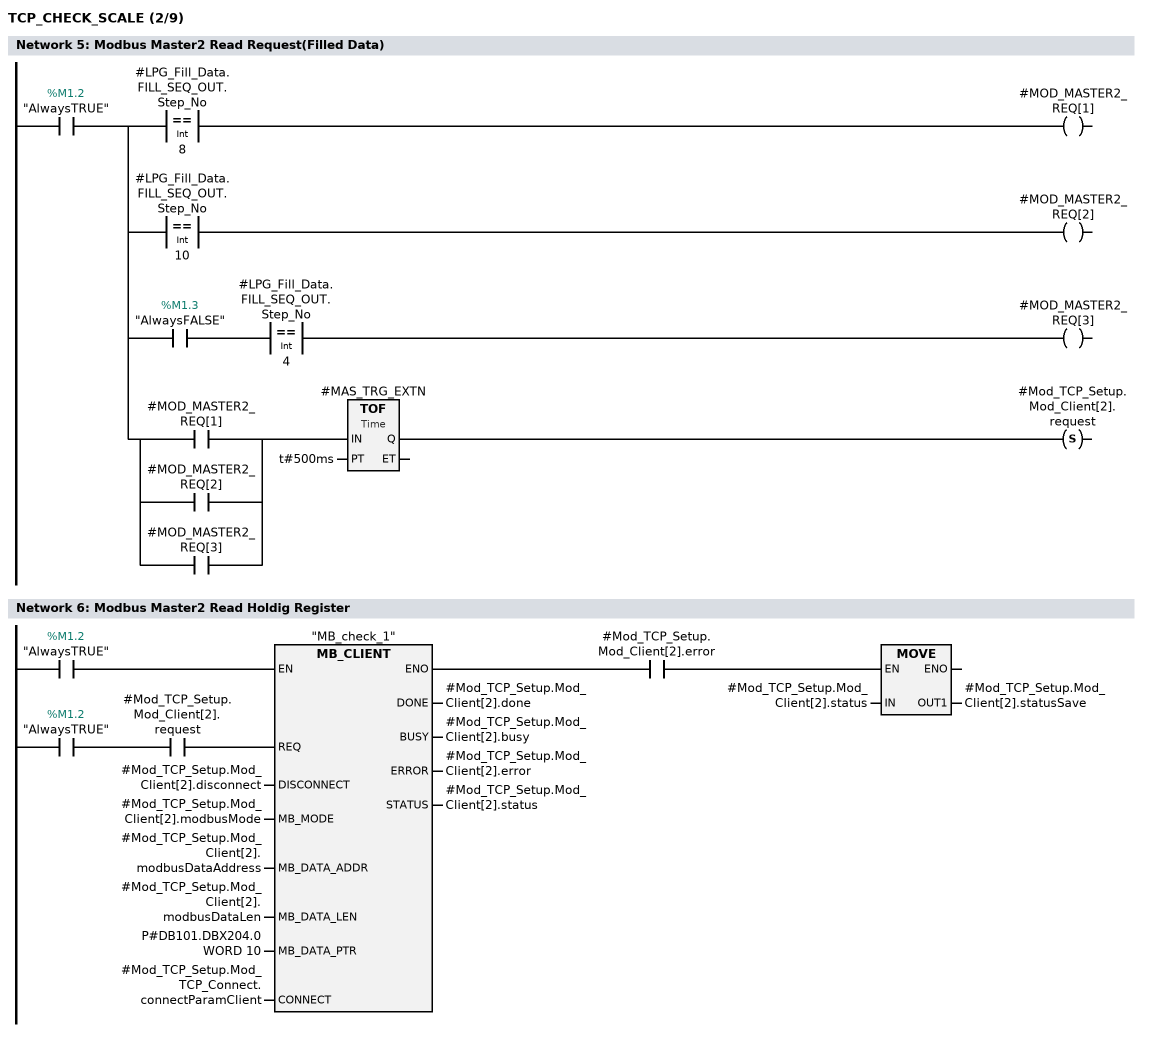
   RUNG wire#powerrail
      Contact( "AlwaysTRUE" )
      wire#w1
      { S7_Templates := "SrcType := Int" } EQ_Contact(in1 := #LPG_Fill_Data.FILL_SEQ_OUT.Step_No, in2 := 8)
      Coil( #MOD_MASTER2_REQ[1] )
   END_RUNG
   RUNG wire#w1
      { S7_Templates := "SrcType := Int" } EQ_Contact(in1 := #LPG_Fill_Data.FILL_SEQ_OUT.Step_No, in2 := 10)
      Coil( #MOD_MASTER2_REQ[2] )
   END_RUNG
   RUNG wire#w1
      Contact( "AlwaysFALSE" )
      { S7_Templates := "SrcType := Int" } EQ_Contact(in1 := #LPG_Fill_Data.FILL_SEQ_OUT.Step_No, in2 := 4)
      Coil( #MOD_MASTER2_REQ[3] )
   END_RUNG
   RUNG wire#w1
      Contact( #MOD_MASTER2_REQ[1] )
      wire#w2
      { S7_Templates := "time_type := Time" } #MAS_TRG_EXTN.TOF(pt := t#500ms, et =>)
      S_Coil( #Mod_TCP_Setup.Mod_Client[2].request )
   END_RUNG
   RUNG wire#w1
      Contact( #MOD_MASTER2_REQ[2] )
   END_RUNG wire#w2
   RUNG wire#w1
      Contact( #MOD_MASTER2_REQ[3] )
   END_RUNG wire#w2
   // the same network as SCL:
   #MOD_MASTER2_REQ[1] := "AlwaysTRUE" AND (#LPG_Fill_Data.FILL_SEQ_OUT.Step_No = 8);
   #MOD_MASTER2_REQ[2] := "AlwaysTRUE" AND (#LPG_Fill_Data.FILL_SEQ_OUT.Step_No = 10);
   #MOD_MASTER2_REQ[3] := "AlwaysTRUE" AND "AlwaysFALSE" AND (#LPG_Fill_Data.FILL_SEQ_OUT.Step_No = 4);
   #MAS_TRG_EXTN(IN := "AlwaysTRUE" AND (#MOD_MASTER2_REQ[1] OR #MOD_MASTER2_REQ[2] OR #MOD_MASTER2_REQ[3]),   // TOF
                 PT := t#500ms);
   IF #MAS_TRG_EXTN.Q THEN #Mod_TCP_Setup.Mod_Client[2].request := TRUE; END_IF;
END_REGION

REGION Network 6: Modbus Master2 Read Holdig Register
   RUNG wire#powerrail
      Contact( "AlwaysTRUE" )
      "MB_check_1".MB_CLIENT(REQ := wire#w1, DISCONNECT := #Mod_TCP_Setup.Mod_Client[2].disconnect, MB_MODE := #Mod_TCP_Setup.Mod_Client[2].modbusMode, MB_DATA_ADDR := #Mod_TCP_Setup.Mod_Client[2].modbusDataAddress, MB_DATA_LEN := #Mod_TCP_Setup.Mod_Client[2].modbusDataLen, MB_DATA_PTR := P#DB101.DBX204.0 WORD 10, CONNECT := #Mod_TCP_Setup.Mod_TCP_Connect.connectParamClient, DONE => #Mod_TCP_Setup.Mod_Client[2].done, BUSY => #Mod_TCP_Setup.Mod_Client[2].busy, ERROR => #Mod_TCP_Setup.Mod_Client[2].error, STATUS => #Mod_TCP_Setup.Mod_Client[2].status)
      Contact( #Mod_TCP_Setup.Mod_Client[2].error )
      Move(in := #Mod_TCP_Setup.Mod_Client[2].status, out1 => #Mod_TCP_Setup.Mod_Client[2].statusSave)
   END_RUNG
   RUNG wire#powerrail
      Contact( "AlwaysTRUE" )
      Contact( #Mod_TCP_Setup.Mod_Client[2].request )
   END_RUNG wire#w1
   // the same network as SCL:
   "MB_check_1"(EN := "AlwaysTRUE",   // MB_CLIENT
                REQ := "AlwaysTRUE" AND #Mod_TCP_Setup.Mod_Client[2].request,
                DISCONNECT := #Mod_TCP_Setup.Mod_Client[2].disconnect,
                MB_MODE := #Mod_TCP_Setup.Mod_Client[2].modbusMode,
                MB_DATA_ADDR := #Mod_TCP_Setup.Mod_Client[2].modbusDataAddress,
                MB_DATA_LEN := #Mod_TCP_Setup.Mod_Client[2].modbusDataLen,
                MB_DATA_PTR := P#DB101.DBX204.0 WORD 10,
                CONNECT := #Mod_TCP_Setup.Mod_TCP_Connect.connectParamClient,
                DONE => #Mod_TCP_Setup.Mod_Client[2].done,
                BUSY => #Mod_TCP_Setup.Mod_Client[2].busy,
                ERROR => #Mod_TCP_Setup.Mod_Client[2].error,
                STATUS => #Mod_TCP_Setup.Mod_Client[2].status,
                ENO => #_w1);
   IF #_w1 AND #Mod_TCP_Setup.Mod_Client[2].error THEN
       #Mod_TCP_Setup.Mod_Client[2].statusSave := #Mod_TCP_Setup.Mod_Client[2].status;
   END_IF;
END_REGION

REGION Network 7: Read Master-2 Holding Register Value
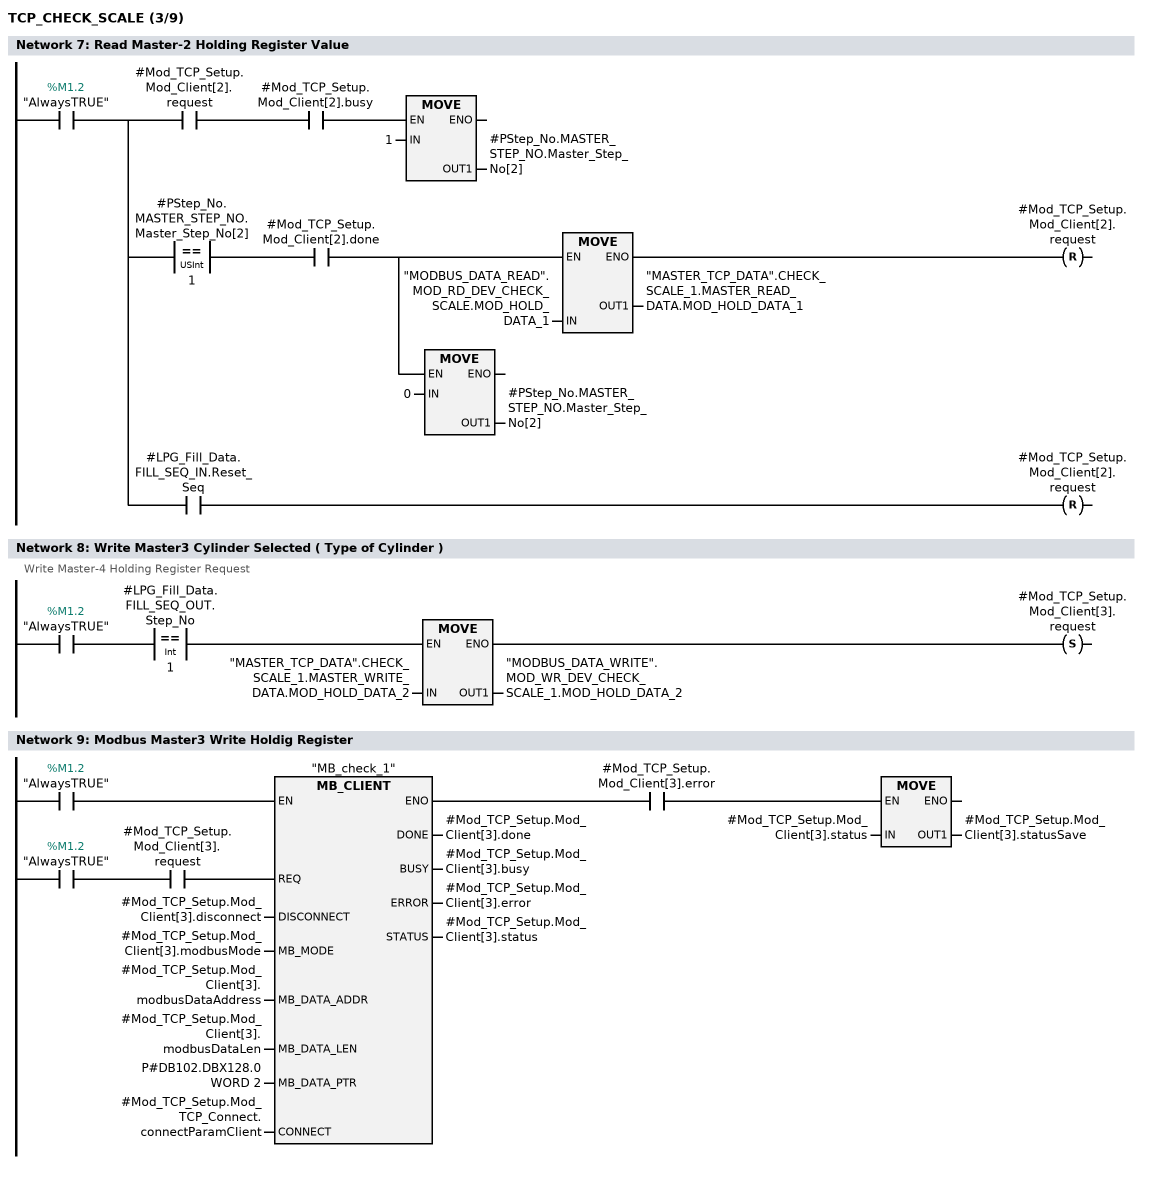
   RUNG wire#powerrail
      Contact( "AlwaysTRUE" )
      wire#w1
      Contact( #Mod_TCP_Setup.Mod_Client[2].request )
      Contact( #Mod_TCP_Setup.Mod_Client[2].busy )
      Move(in := 1, out1 => #PStep_No.MASTER_STEP_NO.Master_Step_No[2])
   END_RUNG
   RUNG wire#w1
      { S7_Templates := "SrcType := USInt" } EQ_Contact(in1 := #PStep_No.MASTER_STEP_NO.Master_Step_No[2], in2 := 1)
      Contact( #Mod_TCP_Setup.Mod_Client[2].done )
      wire#w2
      Move(in := "MODBUS_DATA_READ".MOD_RD_DEV_CHECK_SCALE.MOD_HOLD_DATA_1, out1 => "MASTER_TCP_DATA".CHECK_SCALE_1.MASTER_READ_DATA.MOD_HOLD_DATA_1)
      R_Coil( #Mod_TCP_Setup.Mod_Client[2].request )
   END_RUNG
   RUNG wire#w2
      Move(in := 0, out1 => #PStep_No.MASTER_STEP_NO.Master_Step_No[2])
   END_RUNG
   RUNG wire#w1
      Contact( #LPG_Fill_Data.FILL_SEQ_IN.Reset_Seq )
      R_Coil( #Mod_TCP_Setup.Mod_Client[2].request )
   END_RUNG
   // the same network as SCL:
   IF "AlwaysTRUE" AND #Mod_TCP_Setup.Mod_Client[2].request AND #Mod_TCP_Setup.Mod_Client[2].busy THEN
       #PStep_No.MASTER_STEP_NO.Master_Step_No[2] := 1;
   END_IF;
   IF "AlwaysTRUE" AND (#PStep_No.MASTER_STEP_NO.Master_Step_No[2] = 1) AND #Mod_TCP_Setup.Mod_Client[2].done THEN
       "MASTER_TCP_DATA".CHECK_SCALE_1.MASTER_READ_DATA.MOD_HOLD_DATA_1 := "MODBUS_DATA_READ".MOD_RD_DEV_CHECK_SCALE.MOD_HOLD_DATA_1;
   END_IF;
   #_w1 := "AlwaysTRUE" AND (#PStep_No.MASTER_STEP_NO.Master_Step_No[2] = 1) AND #Mod_TCP_Setup.Mod_Client[2].done;
   IF #_w1 THEN
       #Mod_TCP_Setup.Mod_Client[2].request := FALSE;
       #PStep_No.MASTER_STEP_NO.Master_Step_No[2] := 0;
   END_IF;
   IF "AlwaysTRUE" AND #LPG_Fill_Data.FILL_SEQ_IN.Reset_Seq THEN
       #Mod_TCP_Setup.Mod_Client[2].request := FALSE;
   END_IF;
END_REGION

REGION Network 8: Write Master3 Cylinder Selected ( Type of Cylinder )
   // Write Master-4 Holding Register Request
   RUNG wire#powerrail
      Contact( "AlwaysTRUE" )
      { S7_Templates := "SrcType := Int" } EQ_Contact(in1 := #LPG_Fill_Data.FILL_SEQ_OUT.Step_No, in2 := 1)
      Move(in := "MASTER_TCP_DATA".CHECK_SCALE_1.MASTER_WRITE_DATA.MOD_HOLD_DATA_2, out1 => "MODBUS_DATA_WRITE".MOD_WR_DEV_CHECK_SCALE_1.MOD_HOLD_DATA_2)
      S_Coil( #Mod_TCP_Setup.Mod_Client[3].request )
   END_RUNG
   // the same network as SCL:
   IF "AlwaysTRUE" AND (#LPG_Fill_Data.FILL_SEQ_OUT.Step_No = 1) THEN
       "MODBUS_DATA_WRITE".MOD_WR_DEV_CHECK_SCALE_1.MOD_HOLD_DATA_2 := "MASTER_TCP_DATA".CHECK_SCALE_1.MASTER_WRITE_DATA.MOD_HOLD_DATA_2;
       #Mod_TCP_Setup.Mod_Client[3].request := TRUE;
   END_IF;
END_REGION

REGION Network 9: Modbus Master3 Write Holdig Register
   RUNG wire#powerrail
      Contact( "AlwaysTRUE" )
      "MB_check_1".MB_CLIENT(REQ := wire#w1, DISCONNECT := #Mod_TCP_Setup.Mod_Client[3].disconnect, MB_MODE := #Mod_TCP_Setup.Mod_Client[3].modbusMode, MB_DATA_ADDR := #Mod_TCP_Setup.Mod_Client[3].modbusDataAddress, MB_DATA_LEN := #Mod_TCP_Setup.Mod_Client[3].modbusDataLen, MB_DATA_PTR := P#DB102.DBX128.0 WORD 2, CONNECT := #Mod_TCP_Setup.Mod_TCP_Connect.connectParamClient, DONE => #Mod_TCP_Setup.Mod_Client[3].done, BUSY => #Mod_TCP_Setup.Mod_Client[3].busy, ERROR => #Mod_TCP_Setup.Mod_Client[3].error, STATUS => #Mod_TCP_Setup.Mod_Client[3].status)
      Contact( #Mod_TCP_Setup.Mod_Client[3].error )
      Move(in := #Mod_TCP_Setup.Mod_Client[3].status, out1 => #Mod_TCP_Setup.Mod_Client[3].statusSave)
   END_RUNG
   RUNG wire#powerrail
      Contact( "AlwaysTRUE" )
      Contact( #Mod_TCP_Setup.Mod_Client[3].request )
   END_RUNG wire#w1
   // the same network as SCL:
   "MB_check_1"(EN := "AlwaysTRUE",   // MB_CLIENT
                REQ := "AlwaysTRUE" AND #Mod_TCP_Setup.Mod_Client[3].request,
                DISCONNECT := #Mod_TCP_Setup.Mod_Client[3].disconnect,
                MB_MODE := #Mod_TCP_Setup.Mod_Client[3].modbusMode,
                MB_DATA_ADDR := #Mod_TCP_Setup.Mod_Client[3].modbusDataAddress,
                MB_DATA_LEN := #Mod_TCP_Setup.Mod_Client[3].modbusDataLen,
                MB_DATA_PTR := P#DB102.DBX128.0 WORD 2,
                CONNECT := #Mod_TCP_Setup.Mod_TCP_Connect.connectParamClient,
                DONE => #Mod_TCP_Setup.Mod_Client[3].done,
                BUSY => #Mod_TCP_Setup.Mod_Client[3].busy,
                ERROR => #Mod_TCP_Setup.Mod_Client[3].error,
                STATUS => #Mod_TCP_Setup.Mod_Client[3].status,
                ENO => #_w1);
   IF #_w1 AND #Mod_TCP_Setup.Mod_Client[3].error THEN
       #Mod_TCP_Setup.Mod_Client[3].statusSave := #Mod_TCP_Setup.Mod_Client[3].status;
   END_IF;
END_REGION

REGION Network 10: Write Master-3 Holding Register Done
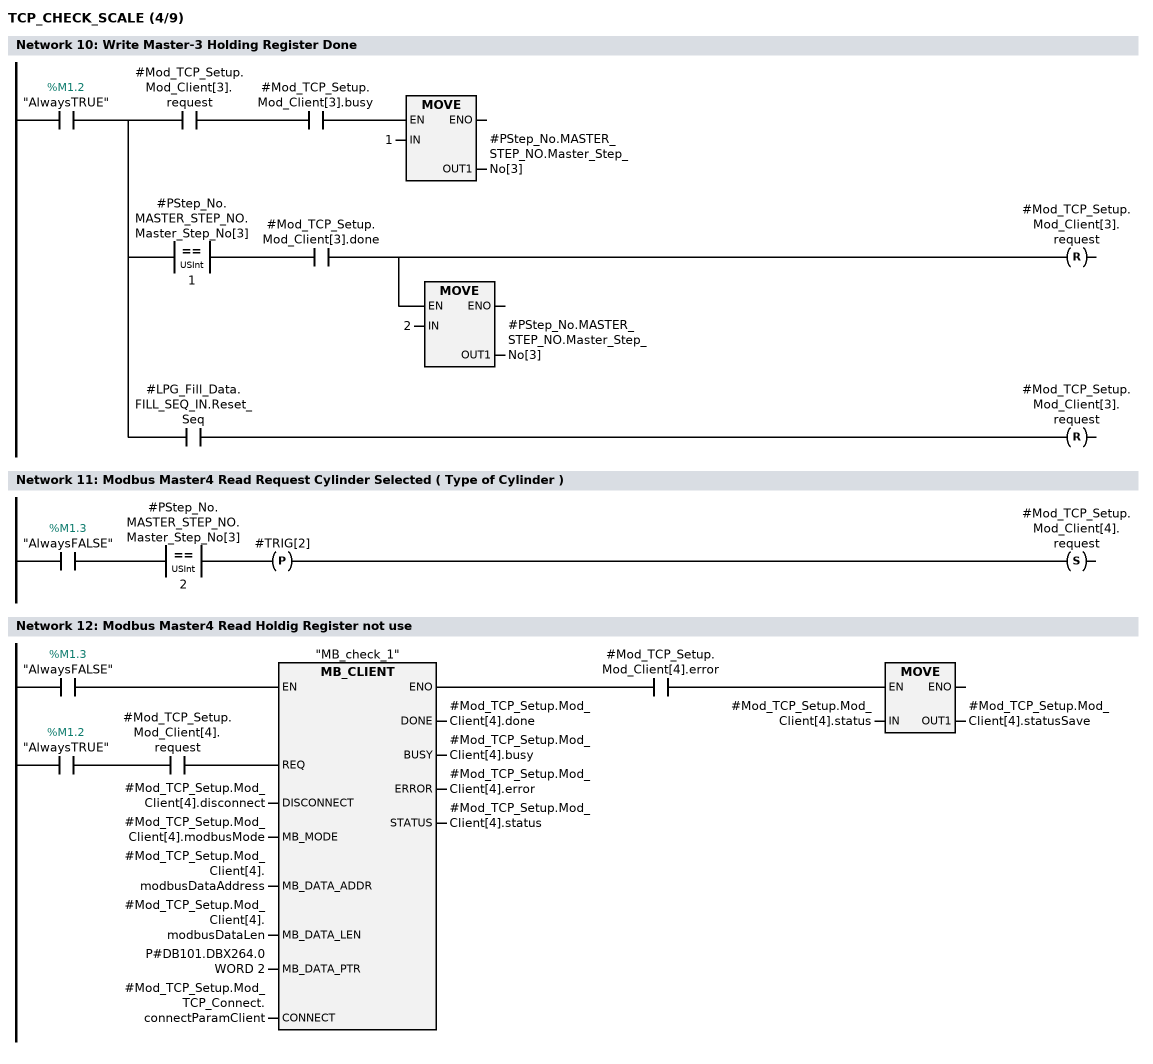
   RUNG wire#powerrail
      Contact( "AlwaysTRUE" )
      wire#w1
      Contact( #Mod_TCP_Setup.Mod_Client[3].request )
      Contact( #Mod_TCP_Setup.Mod_Client[3].busy )
      Move(in := 1, out1 => #PStep_No.MASTER_STEP_NO.Master_Step_No[3])
   END_RUNG
   RUNG wire#w1
      { S7_Templates := "SrcType := USInt" } EQ_Contact(in1 := #PStep_No.MASTER_STEP_NO.Master_Step_No[3], in2 := 1)
      Contact( #Mod_TCP_Setup.Mod_Client[3].done )
      wire#w2
      R_Coil( #Mod_TCP_Setup.Mod_Client[3].request )
   END_RUNG
   RUNG wire#w2
      Move(in := 2, out1 => #PStep_No.MASTER_STEP_NO.Master_Step_No[3])
   END_RUNG
   RUNG wire#w1
      Contact( #LPG_Fill_Data.FILL_SEQ_IN.Reset_Seq )
      R_Coil( #Mod_TCP_Setup.Mod_Client[3].request )
   END_RUNG
   // the same network as SCL:
   IF "AlwaysTRUE" AND #Mod_TCP_Setup.Mod_Client[3].request AND #Mod_TCP_Setup.Mod_Client[3].busy THEN
       #PStep_No.MASTER_STEP_NO.Master_Step_No[3] := 1;
   END_IF;
   #_w1 := "AlwaysTRUE" AND (#PStep_No.MASTER_STEP_NO.Master_Step_No[3] = 1) AND #Mod_TCP_Setup.Mod_Client[3].done;
   IF #_w1 THEN
       #Mod_TCP_Setup.Mod_Client[3].request := FALSE;
       #PStep_No.MASTER_STEP_NO.Master_Step_No[3] := 2;
   END_IF;
   IF "AlwaysTRUE" AND #LPG_Fill_Data.FILL_SEQ_IN.Reset_Seq THEN
       #Mod_TCP_Setup.Mod_Client[3].request := FALSE;
   END_IF;
END_REGION

REGION Network 11: Modbus Master4 Read Request Cylinder Selected ( Type of Cylinder )
   RUNG wire#powerrail
      Contact( "AlwaysFALSE" )
      { S7_Templates := "SrcType := USInt" } EQ_Contact(in1 := #PStep_No.MASTER_STEP_NO.Master_Step_No[3], in2 := 2)
      P_Trig( #TRIG[2] )
      S_Coil( #Mod_TCP_Setup.Mod_Client[4].request )
   END_RUNG
   // the same network as SCL:
   #_w1 := "AlwaysFALSE" AND (#PStep_No.MASTER_STEP_NO.Master_Step_No[3] = 2);
   #_w2 := #_w1 AND NOT #TRIG[2];   // rising edge
   #TRIG[2] := #_w1;
   IF #_w2 THEN #Mod_TCP_Setup.Mod_Client[4].request := TRUE; END_IF;
END_REGION

REGION Network 12: Modbus Master4 Read Holdig Register not use
   RUNG wire#powerrail
      Contact( "AlwaysFALSE" )
      "MB_check_1".MB_CLIENT(REQ := wire#w1, DISCONNECT := #Mod_TCP_Setup.Mod_Client[4].disconnect, MB_MODE := #Mod_TCP_Setup.Mod_Client[4].modbusMode, MB_DATA_ADDR := #Mod_TCP_Setup.Mod_Client[4].modbusDataAddress, MB_DATA_LEN := #Mod_TCP_Setup.Mod_Client[4].modbusDataLen, MB_DATA_PTR := P#DB101.DBX264.0 WORD 2, CONNECT := #Mod_TCP_Setup.Mod_TCP_Connect.connectParamClient, DONE => #Mod_TCP_Setup.Mod_Client[4].done, BUSY => #Mod_TCP_Setup.Mod_Client[4].busy, ERROR => #Mod_TCP_Setup.Mod_Client[4].error, STATUS => #Mod_TCP_Setup.Mod_Client[4].status)
      Contact( #Mod_TCP_Setup.Mod_Client[4].error )
      Move(in := #Mod_TCP_Setup.Mod_Client[4].status, out1 => #Mod_TCP_Setup.Mod_Client[4].statusSave)
   END_RUNG
   RUNG wire#powerrail
      Contact( "AlwaysTRUE" )
      Contact( #Mod_TCP_Setup.Mod_Client[4].request )
   END_RUNG wire#w1
   // the same network as SCL:
   "MB_check_1"(EN := "AlwaysFALSE",   // MB_CLIENT
                REQ := "AlwaysTRUE" AND #Mod_TCP_Setup.Mod_Client[4].request,
                DISCONNECT := #Mod_TCP_Setup.Mod_Client[4].disconnect,
                MB_MODE := #Mod_TCP_Setup.Mod_Client[4].modbusMode,
                MB_DATA_ADDR := #Mod_TCP_Setup.Mod_Client[4].modbusDataAddress,
                MB_DATA_LEN := #Mod_TCP_Setup.Mod_Client[4].modbusDataLen,
                MB_DATA_PTR := P#DB101.DBX264.0 WORD 2,
                CONNECT := #Mod_TCP_Setup.Mod_TCP_Connect.connectParamClient,
                DONE => #Mod_TCP_Setup.Mod_Client[4].done,
                BUSY => #Mod_TCP_Setup.Mod_Client[4].busy,
                ERROR => #Mod_TCP_Setup.Mod_Client[4].error,
                STATUS => #Mod_TCP_Setup.Mod_Client[4].status,
                ENO => #_w1);
   IF #_w1 AND #Mod_TCP_Setup.Mod_Client[4].error THEN
       #Mod_TCP_Setup.Mod_Client[4].statusSave := #Mod_TCP_Setup.Mod_Client[4].status;
   END_IF;
END_REGION

REGION Network 13: Read Master-4 Holding Register Value
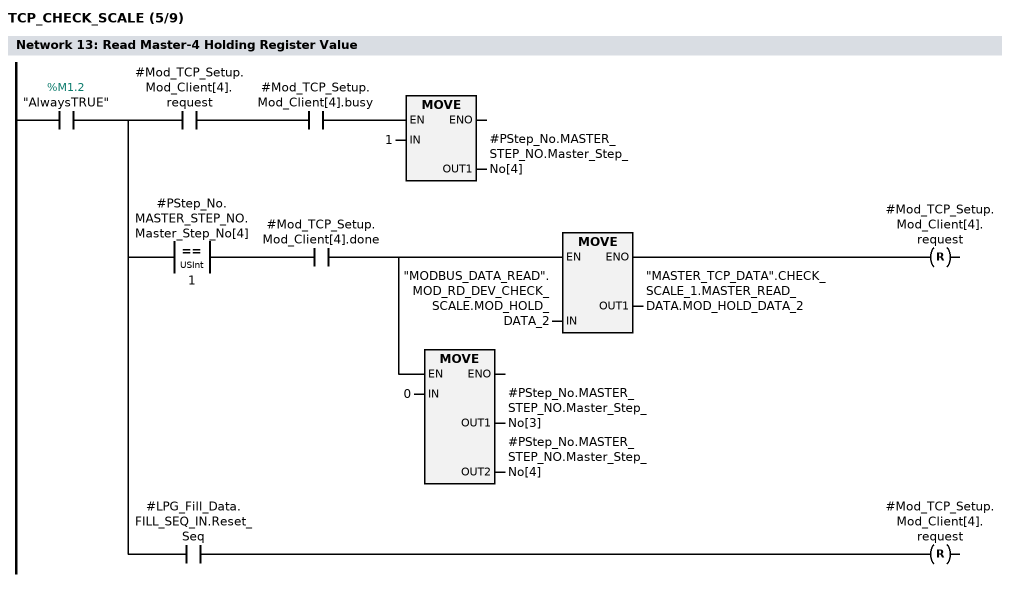
   RUNG wire#powerrail
      Contact( "AlwaysTRUE" )
      wire#w1
      Contact( #Mod_TCP_Setup.Mod_Client[4].request )
      Contact( #Mod_TCP_Setup.Mod_Client[4].busy )
      Move(in := 1, out1 => #PStep_No.MASTER_STEP_NO.Master_Step_No[4])
   END_RUNG
   RUNG wire#w1
      { S7_Templates := "SrcType := USInt" } EQ_Contact(in1 := #PStep_No.MASTER_STEP_NO.Master_Step_No[4], in2 := 1)
      Contact( #Mod_TCP_Setup.Mod_Client[4].done )
      wire#w2
      Move(in := "MODBUS_DATA_READ".MOD_RD_DEV_CHECK_SCALE.MOD_HOLD_DATA_2, out1 => "MASTER_TCP_DATA".CHECK_SCALE_1.MASTER_READ_DATA.MOD_HOLD_DATA_2)
      R_Coil( #Mod_TCP_Setup.Mod_Client[4].request )
   END_RUNG
   RUNG wire#w2
      Move(in := 0, out1 => #PStep_No.MASTER_STEP_NO.Master_Step_No[3], out2 => #PStep_No.MASTER_STEP_NO.Master_Step_No[4])
   END_RUNG
   RUNG wire#w1
      Contact( #LPG_Fill_Data.FILL_SEQ_IN.Reset_Seq )
      R_Coil( #Mod_TCP_Setup.Mod_Client[4].request )
   END_RUNG
   // the same network as SCL:
   IF "AlwaysTRUE" AND #Mod_TCP_Setup.Mod_Client[4].request AND #Mod_TCP_Setup.Mod_Client[4].busy THEN
       #PStep_No.MASTER_STEP_NO.Master_Step_No[4] := 1;
   END_IF;
   IF "AlwaysTRUE" AND (#PStep_No.MASTER_STEP_NO.Master_Step_No[4] = 1) AND #Mod_TCP_Setup.Mod_Client[4].done THEN
       "MASTER_TCP_DATA".CHECK_SCALE_1.MASTER_READ_DATA.MOD_HOLD_DATA_2 := "MODBUS_DATA_READ".MOD_RD_DEV_CHECK_SCALE.MOD_HOLD_DATA_2;
   END_IF;
   #_w1 := "AlwaysTRUE" AND (#PStep_No.MASTER_STEP_NO.Master_Step_No[4] = 1) AND #Mod_TCP_Setup.Mod_Client[4].done;
   IF #_w1 THEN
       #Mod_TCP_Setup.Mod_Client[4].request := FALSE;
       #PStep_No.MASTER_STEP_NO.Master_Step_No[3] := 0;
       #PStep_No.MASTER_STEP_NO.Master_Step_No[4] := 0;
   END_IF;
   IF "AlwaysTRUE" AND #LPG_Fill_Data.FILL_SEQ_IN.Reset_Seq THEN
       #Mod_TCP_Setup.Mod_Client[4].request := FALSE;
   END_IF;
END_REGION

REGION Network 14: Modbus Master5 Read Request(Coil Status)
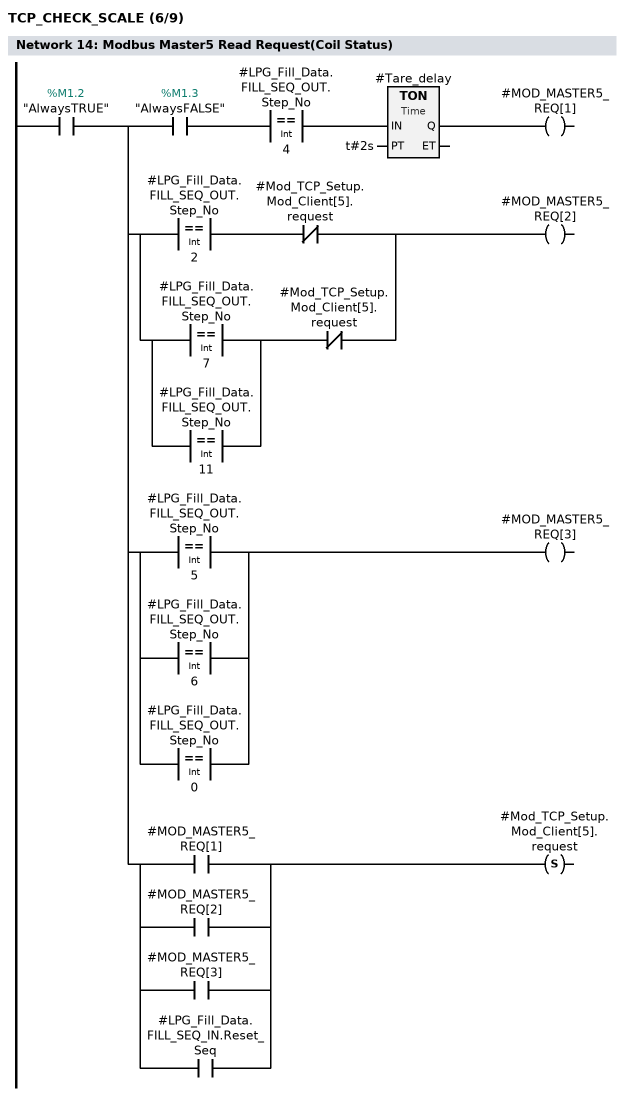
   RUNG wire#powerrail
      Contact( "AlwaysTRUE" )
      wire#w1
      Contact( "AlwaysFALSE" )
      { S7_Templates := "SrcType := Int" } EQ_Contact(in1 := #LPG_Fill_Data.FILL_SEQ_OUT.Step_No, in2 := 4)
      { S7_Templates := "time_type := Time" } #Tare_delay.TON(pt := t#2s, et =>)
      Coil( #MOD_MASTER5_REQ[1] )
   END_RUNG
   RUNG wire#w1
      { S7_Templates := "SrcType := Int" } EQ_Contact(in1 := #LPG_Fill_Data.FILL_SEQ_OUT.Step_No, in2 := 2)
      I_Contact( #Mod_TCP_Setup.Mod_Client[5].request )
      wire#w2
      Coil( #MOD_MASTER5_REQ[2] )
   END_RUNG
   RUNG wire#w1
      { S7_Templates := "SrcType := Int" } EQ_Contact(in1 := #LPG_Fill_Data.FILL_SEQ_OUT.Step_No, in2 := 7)
      wire#w3
      I_Contact( #Mod_TCP_Setup.Mod_Client[5].request )
   END_RUNG wire#w2
   RUNG wire#w1
      { S7_Templates := "SrcType := Int" } EQ_Contact(in1 := #LPG_Fill_Data.FILL_SEQ_OUT.Step_No, in2 := 11)
   END_RUNG wire#w3
   RUNG wire#w1
      { S7_Templates := "SrcType := Int" } EQ_Contact(in1 := #LPG_Fill_Data.FILL_SEQ_OUT.Step_No, in2 := 5)
      wire#w4
      Coil( #MOD_MASTER5_REQ[3] )
   END_RUNG
   RUNG wire#w1
      { S7_Templates := "SrcType := Int" } EQ_Contact(in1 := #LPG_Fill_Data.FILL_SEQ_OUT.Step_No, in2 := 6)
   END_RUNG wire#w4
   RUNG wire#w1
      { S7_Templates := "SrcType := Int" } EQ_Contact(in1 := #LPG_Fill_Data.FILL_SEQ_OUT.Step_No, in2 := 0)
   END_RUNG wire#w4
   RUNG wire#w1
      Contact( #MOD_MASTER5_REQ[1] )
      wire#w5
      S_Coil( #Mod_TCP_Setup.Mod_Client[5].request )
   END_RUNG
   RUNG wire#w1
      Contact( #MOD_MASTER5_REQ[2] )
   END_RUNG wire#w5
   RUNG wire#w1
      Contact( #MOD_MASTER5_REQ[3] )
   END_RUNG wire#w5
   RUNG wire#w1
      Contact( #LPG_Fill_Data.FILL_SEQ_IN.Reset_Seq )
   END_RUNG wire#w5
   // the same network as SCL:
   #Tare_delay(IN := "AlwaysTRUE" AND "AlwaysFALSE" AND (#LPG_Fill_Data.FILL_SEQ_OUT.Step_No = 4), PT := t#2s);   // TON
   #MOD_MASTER5_REQ[1] := #Tare_delay.Q;
   #MOD_MASTER5_REQ[2] := "AlwaysTRUE" AND (((#LPG_Fill_Data.FILL_SEQ_OUT.Step_No = 2) AND NOT #Mod_TCP_Setup.Mod_Client[5].request) OR (((#LPG_Fill_Data.FILL_SEQ_OUT.Step_No = 7) OR (#LPG_Fill_Data.FILL_SEQ_OUT.Step_No = 11)) AND NOT #Mod_TCP_Setup.Mod_Client[5].request));
   #MOD_MASTER5_REQ[3] := "AlwaysTRUE" AND ((#LPG_Fill_Data.FILL_SEQ_OUT.Step_No = 5) OR (#LPG_Fill_Data.FILL_SEQ_OUT.Step_No = 6) OR (#LPG_Fill_Data.FILL_SEQ_OUT.Step_No = 0));
   IF "AlwaysTRUE" AND (#MOD_MASTER5_REQ[1] OR #MOD_MASTER5_REQ[2] OR #MOD_MASTER5_REQ[3] OR #LPG_Fill_Data.FILL_SEQ_IN.Reset_Seq) THEN
       #Mod_TCP_Setup.Mod_Client[5].request := TRUE;
   END_IF;
END_REGION

REGION Network 15: Modbus Master5 Read Coil Status
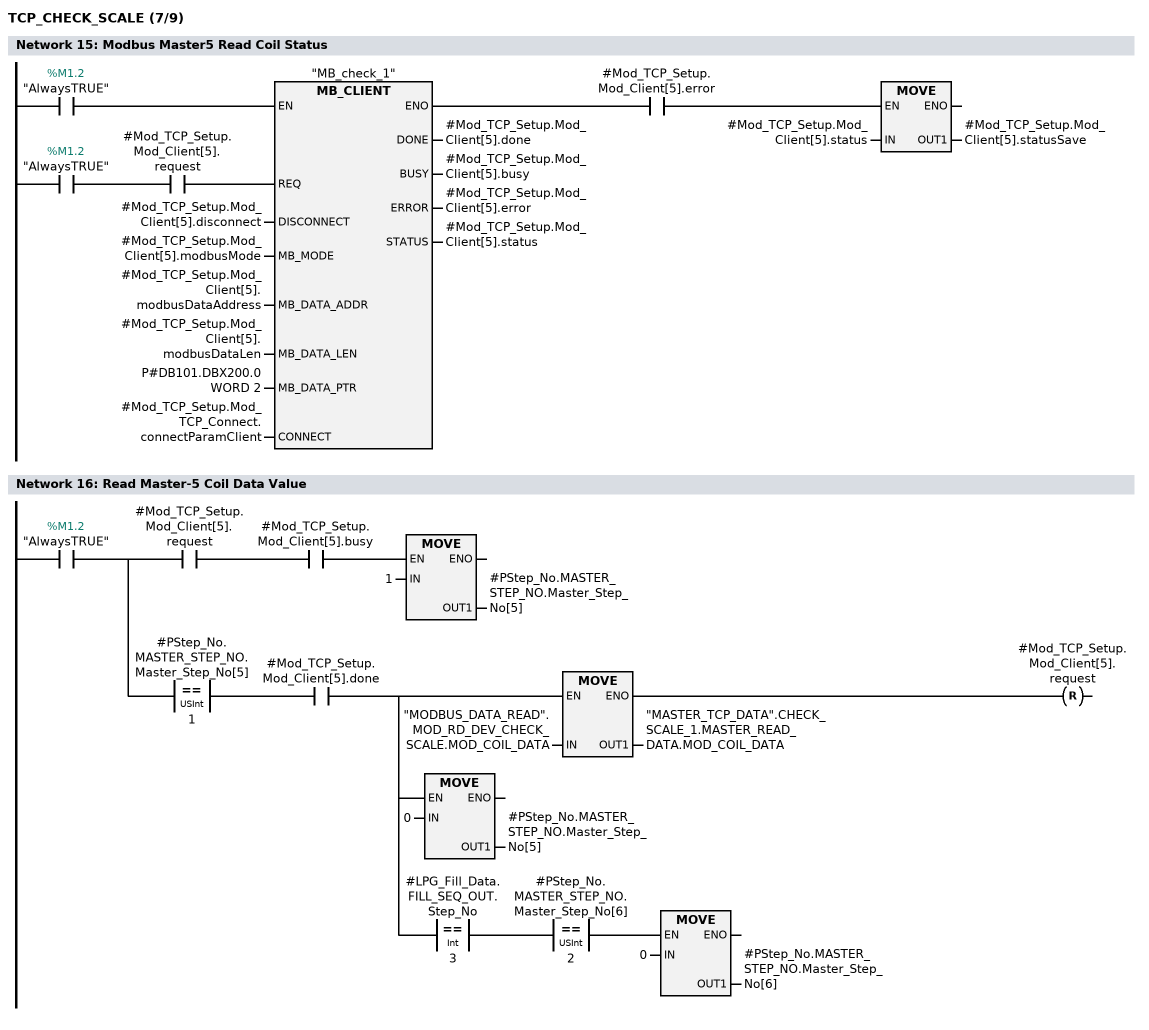
   RUNG wire#powerrail
      Contact( "AlwaysTRUE" )
      "MB_check_1".MB_CLIENT(REQ := wire#w1, DISCONNECT := #Mod_TCP_Setup.Mod_Client[5].disconnect, MB_MODE := #Mod_TCP_Setup.Mod_Client[5].modbusMode, MB_DATA_ADDR := #Mod_TCP_Setup.Mod_Client[5].modbusDataAddress, MB_DATA_LEN := #Mod_TCP_Setup.Mod_Client[5].modbusDataLen, MB_DATA_PTR := P#DB101.DBX200.0 WORD 2, CONNECT := #Mod_TCP_Setup.Mod_TCP_Connect.connectParamClient, DONE => #Mod_TCP_Setup.Mod_Client[5].done, BUSY => #Mod_TCP_Setup.Mod_Client[5].busy, ERROR => #Mod_TCP_Setup.Mod_Client[5].error, STATUS => #Mod_TCP_Setup.Mod_Client[5].status)
      Contact( #Mod_TCP_Setup.Mod_Client[5].error )
      Move(in := #Mod_TCP_Setup.Mod_Client[5].status, out1 => #Mod_TCP_Setup.Mod_Client[5].statusSave)
   END_RUNG
   RUNG wire#powerrail
      Contact( "AlwaysTRUE" )
      Contact( #Mod_TCP_Setup.Mod_Client[5].request )
   END_RUNG wire#w1
   // the same network as SCL:
   "MB_check_1"(EN := "AlwaysTRUE",   // MB_CLIENT
                REQ := "AlwaysTRUE" AND #Mod_TCP_Setup.Mod_Client[5].request,
                DISCONNECT := #Mod_TCP_Setup.Mod_Client[5].disconnect,
                MB_MODE := #Mod_TCP_Setup.Mod_Client[5].modbusMode,
                MB_DATA_ADDR := #Mod_TCP_Setup.Mod_Client[5].modbusDataAddress,
                MB_DATA_LEN := #Mod_TCP_Setup.Mod_Client[5].modbusDataLen,
                MB_DATA_PTR := P#DB101.DBX200.0 WORD 2,
                CONNECT := #Mod_TCP_Setup.Mod_TCP_Connect.connectParamClient,
                DONE => #Mod_TCP_Setup.Mod_Client[5].done,
                BUSY => #Mod_TCP_Setup.Mod_Client[5].busy,
                ERROR => #Mod_TCP_Setup.Mod_Client[5].error,
                STATUS => #Mod_TCP_Setup.Mod_Client[5].status,
                ENO => #_w1);
   IF #_w1 AND #Mod_TCP_Setup.Mod_Client[5].error THEN
       #Mod_TCP_Setup.Mod_Client[5].statusSave := #Mod_TCP_Setup.Mod_Client[5].status;
   END_IF;
END_REGION

REGION Network 16: Read Master-5 Coil Data Value
   RUNG wire#powerrail
      Contact( "AlwaysTRUE" )
      wire#w1
      Contact( #Mod_TCP_Setup.Mod_Client[5].request )
      Contact( #Mod_TCP_Setup.Mod_Client[5].busy )
      Move(in := 1, out1 => #PStep_No.MASTER_STEP_NO.Master_Step_No[5])
   END_RUNG
   RUNG wire#w1
      { S7_Templates := "SrcType := USInt" } EQ_Contact(in1 := #PStep_No.MASTER_STEP_NO.Master_Step_No[5], in2 := 1)
      Contact( #Mod_TCP_Setup.Mod_Client[5].done )
      wire#w2
      Move(in := "MODBUS_DATA_READ".MOD_RD_DEV_CHECK_SCALE.MOD_COIL_DATA, out1 => "MASTER_TCP_DATA".CHECK_SCALE_1.MASTER_READ_DATA.MOD_COIL_DATA)
      R_Coil( #Mod_TCP_Setup.Mod_Client[5].request )
   END_RUNG
   RUNG wire#w2
      Move(in := 0, out1 => #PStep_No.MASTER_STEP_NO.Master_Step_No[5])
   END_RUNG
   RUNG wire#w2
      { S7_Templates := "SrcType := Int" } EQ_Contact(in1 := #LPG_Fill_Data.FILL_SEQ_OUT.Step_No, in2 := 3)
      { S7_Templates := "SrcType := USInt" } EQ_Contact(in1 := #PStep_No.MASTER_STEP_NO.Master_Step_No[6], in2 := 2)
      Move(in := 0, out1 => #PStep_No.MASTER_STEP_NO.Master_Step_No[6])
   END_RUNG
   // the same network as SCL:
   IF "AlwaysTRUE" AND #Mod_TCP_Setup.Mod_Client[5].request AND #Mod_TCP_Setup.Mod_Client[5].busy THEN
       #PStep_No.MASTER_STEP_NO.Master_Step_No[5] := 1;
   END_IF;
   #_w1 := "AlwaysTRUE" AND (#PStep_No.MASTER_STEP_NO.Master_Step_No[5] = 1) AND #Mod_TCP_Setup.Mod_Client[5].done;
   IF #_w1 THEN
       "MASTER_TCP_DATA".CHECK_SCALE_1.MASTER_READ_DATA.MOD_COIL_DATA := "MODBUS_DATA_READ".MOD_RD_DEV_CHECK_SCALE.MOD_COIL_DATA;
       #Mod_TCP_Setup.Mod_Client[5].request := FALSE;
       #PStep_No.MASTER_STEP_NO.Master_Step_No[5] := 0;
   END_IF;
   IF #_w1 AND (#LPG_Fill_Data.FILL_SEQ_OUT.Step_No = 3) AND (#PStep_No.MASTER_STEP_NO.Master_Step_No[6] = 2) THEN
       #PStep_No.MASTER_STEP_NO.Master_Step_No[6] := 0;
   END_IF;
END_REGION

REGION Network 17: Write Coil Data
   // if multiple bit write not working
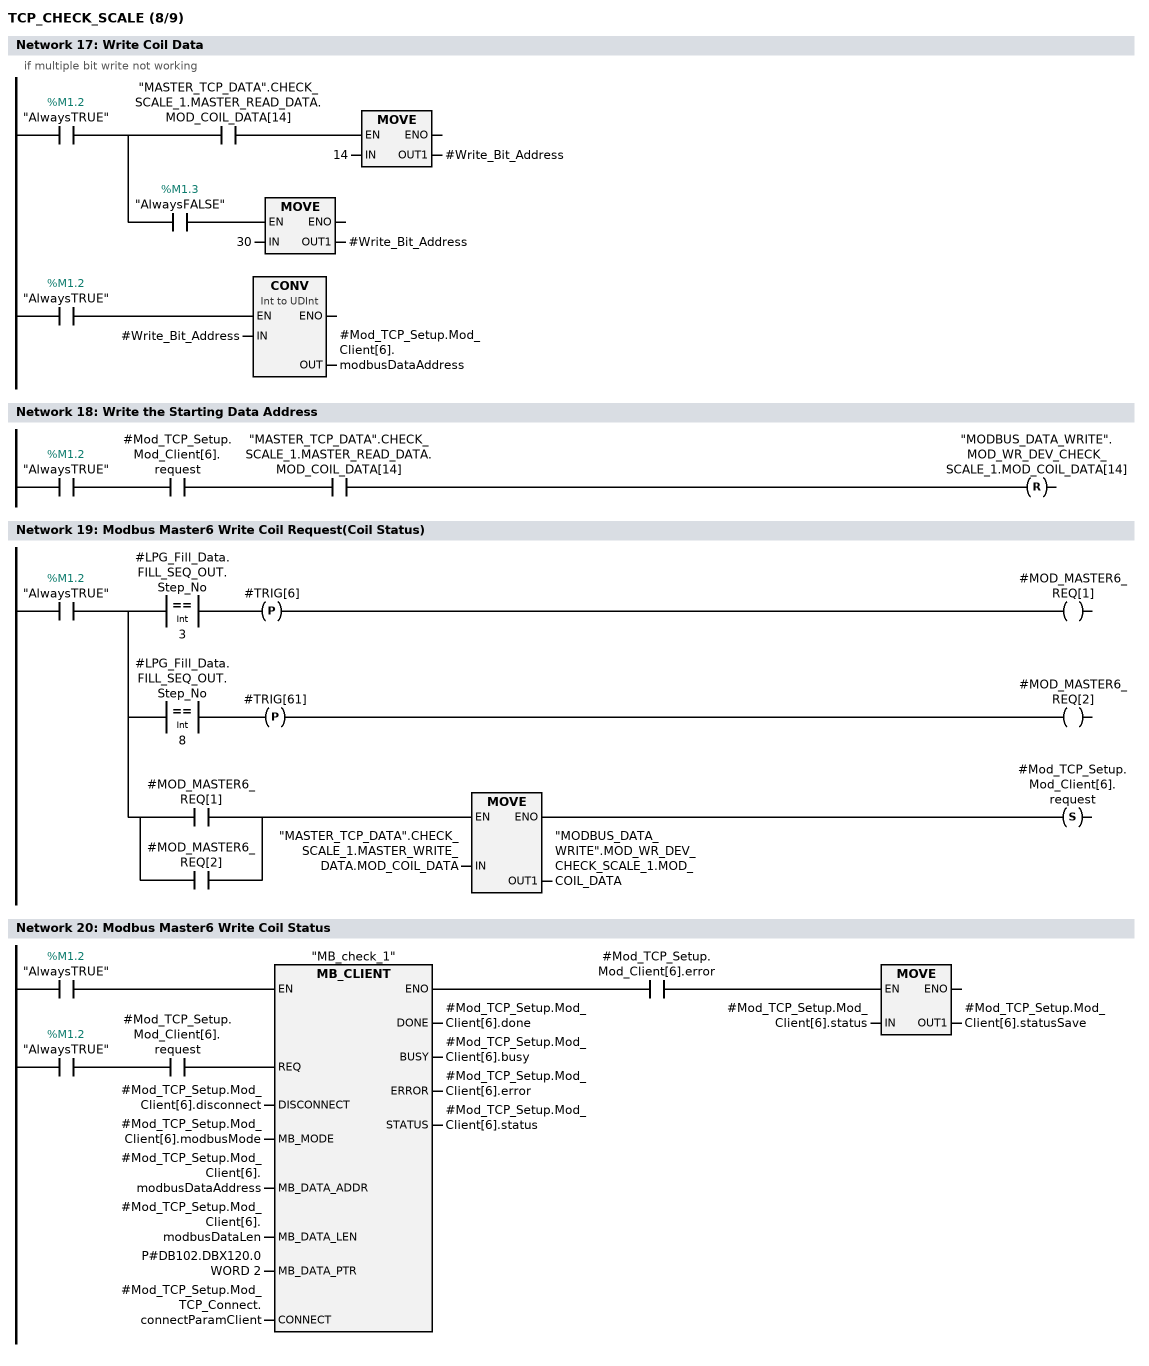
   RUNG wire#powerrail
      Contact( "AlwaysTRUE" )
      wire#w1
      Contact( "MASTER_TCP_DATA".CHECK_SCALE_1.MASTER_READ_DATA.MOD_COIL_DATA[14] )
      Move(in := 14, out1 => #Write_Bit_Address)
   END_RUNG
   RUNG wire#w1
      Contact( "AlwaysFALSE" )
      Move(in := 30, out1 => #Write_Bit_Address)
   END_RUNG
   RUNG wire#powerrail
      Contact( "AlwaysTRUE" )
      { S7_Templates := "[SrcType := Int, DestType := UDInt]" } Convert(in := #Write_Bit_Address, out => #Mod_TCP_Setup.Mod_Client[6].modbusDataAddress)
   END_RUNG
   // the same network as SCL:
   IF "AlwaysTRUE" AND "MASTER_TCP_DATA".CHECK_SCALE_1.MASTER_READ_DATA.MOD_COIL_DATA[14] THEN
       #Write_Bit_Address := 14;
   END_IF;
   IF "AlwaysTRUE" AND "AlwaysFALSE" THEN #Write_Bit_Address := 30; END_IF;
   IF "AlwaysTRUE" THEN
       #Mod_TCP_Setup.Mod_Client[6].modbusDataAddress := INT_TO_UDINT(#Write_Bit_Address);
   END_IF;
END_REGION

REGION Network 18: Write the Starting Data Address
   RUNG wire#powerrail
      Contact( "AlwaysTRUE" )
      Contact( #Mod_TCP_Setup.Mod_Client[6].request )
      Contact( "MASTER_TCP_DATA".CHECK_SCALE_1.MASTER_READ_DATA.MOD_COIL_DATA[14] )
      R_Coil( "MODBUS_DATA_WRITE".MOD_WR_DEV_CHECK_SCALE_1.MOD_COIL_DATA[14] )
   END_RUNG
   // the same network as SCL:
   IF "AlwaysTRUE" AND #Mod_TCP_Setup.Mod_Client[6].request AND "MASTER_TCP_DATA".CHECK_SCALE_1.MASTER_READ_DATA.MOD_COIL_DATA[14] THEN
       "MODBUS_DATA_WRITE".MOD_WR_DEV_CHECK_SCALE_1.MOD_COIL_DATA[14] := FALSE;
   END_IF;
END_REGION

REGION Network 19: Modbus Master6 Write Coil Request(Coil Status)
   RUNG wire#powerrail
      Contact( "AlwaysTRUE" )
      wire#w1
      { S7_Templates := "SrcType := Int" } EQ_Contact(in1 := #LPG_Fill_Data.FILL_SEQ_OUT.Step_No, in2 := 3)
      P_Trig( #TRIG[6] )
      Coil( #MOD_MASTER6_REQ[1] )
   END_RUNG
   RUNG wire#w1
      { S7_Templates := "SrcType := Int" } EQ_Contact(in1 := #LPG_Fill_Data.FILL_SEQ_OUT.Step_No, in2 := 8)
      P_Trig( #TRIG[61] )
      Coil( #MOD_MASTER6_REQ[2] )
   END_RUNG
   RUNG wire#w1
      Contact( #MOD_MASTER6_REQ[1] )
      wire#w2
      Move(in := "MASTER_TCP_DATA".CHECK_SCALE_1.MASTER_WRITE_DATA.MOD_COIL_DATA, out1 => "MODBUS_DATA_WRITE".MOD_WR_DEV_CHECK_SCALE_1.MOD_COIL_DATA)
      S_Coil( #Mod_TCP_Setup.Mod_Client[6].request )
   END_RUNG
   RUNG wire#w1
      Contact( #MOD_MASTER6_REQ[2] )
   END_RUNG wire#w2
   // the same network as SCL:
   #_w1 := "AlwaysTRUE" AND (#LPG_Fill_Data.FILL_SEQ_OUT.Step_No = 3);
   #_w2 := #_w1 AND NOT #TRIG[6];   // rising edge
   #TRIG[6] := #_w1;
   #MOD_MASTER6_REQ[1] := #_w2;
   #_w3 := "AlwaysTRUE" AND (#LPG_Fill_Data.FILL_SEQ_OUT.Step_No = 8);
   #_w4 := #_w3 AND NOT #TRIG[61];   // rising edge
   #TRIG[61] := #_w3;
   #MOD_MASTER6_REQ[2] := #_w4;
   IF "AlwaysTRUE" AND (#MOD_MASTER6_REQ[1] OR #MOD_MASTER6_REQ[2]) THEN
       "MODBUS_DATA_WRITE".MOD_WR_DEV_CHECK_SCALE_1.MOD_COIL_DATA := "MASTER_TCP_DATA".CHECK_SCALE_1.MASTER_WRITE_DATA.MOD_COIL_DATA;
       #Mod_TCP_Setup.Mod_Client[6].request := TRUE;
   END_IF;
END_REGION

REGION Network 20: Modbus Master6 Write Coil Status
   RUNG wire#powerrail
      Contact( "AlwaysTRUE" )
      "MB_check_1".MB_CLIENT(REQ := wire#w1, DISCONNECT := #Mod_TCP_Setup.Mod_Client[6].disconnect, MB_MODE := #Mod_TCP_Setup.Mod_Client[6].modbusMode, MB_DATA_ADDR := #Mod_TCP_Setup.Mod_Client[6].modbusDataAddress, MB_DATA_LEN := #Mod_TCP_Setup.Mod_Client[6].modbusDataLen, MB_DATA_PTR := P#DB102.DBX120.0 WORD 2, CONNECT := #Mod_TCP_Setup.Mod_TCP_Connect.connectParamClient, DONE => #Mod_TCP_Setup.Mod_Client[6].done, BUSY => #Mod_TCP_Setup.Mod_Client[6].busy, ERROR => #Mod_TCP_Setup.Mod_Client[6].error, STATUS => #Mod_TCP_Setup.Mod_Client[6].status)
      Contact( #Mod_TCP_Setup.Mod_Client[6].error )
      Move(in := #Mod_TCP_Setup.Mod_Client[6].status, out1 => #Mod_TCP_Setup.Mod_Client[6].statusSave)
   END_RUNG
   RUNG wire#powerrail
      Contact( "AlwaysTRUE" )
      Contact( #Mod_TCP_Setup.Mod_Client[6].request )
   END_RUNG wire#w1
   // the same network as SCL:
   "MB_check_1"(EN := "AlwaysTRUE",   // MB_CLIENT
                REQ := "AlwaysTRUE" AND #Mod_TCP_Setup.Mod_Client[6].request,
                DISCONNECT := #Mod_TCP_Setup.Mod_Client[6].disconnect,
                MB_MODE := #Mod_TCP_Setup.Mod_Client[6].modbusMode,
                MB_DATA_ADDR := #Mod_TCP_Setup.Mod_Client[6].modbusDataAddress,
                MB_DATA_LEN := #Mod_TCP_Setup.Mod_Client[6].modbusDataLen,
                MB_DATA_PTR := P#DB102.DBX120.0 WORD 2,
                CONNECT := #Mod_TCP_Setup.Mod_TCP_Connect.connectParamClient,
                DONE => #Mod_TCP_Setup.Mod_Client[6].done,
                BUSY => #Mod_TCP_Setup.Mod_Client[6].busy,
                ERROR => #Mod_TCP_Setup.Mod_Client[6].error,
                STATUS => #Mod_TCP_Setup.Mod_Client[6].status,
                ENO => #_w1);
   IF #_w1 AND #Mod_TCP_Setup.Mod_Client[6].error THEN
       #Mod_TCP_Setup.Mod_Client[6].statusSave := #Mod_TCP_Setup.Mod_Client[6].status;
   END_IF;
END_REGION

REGION Network 21: Write Master-6 Coil Data
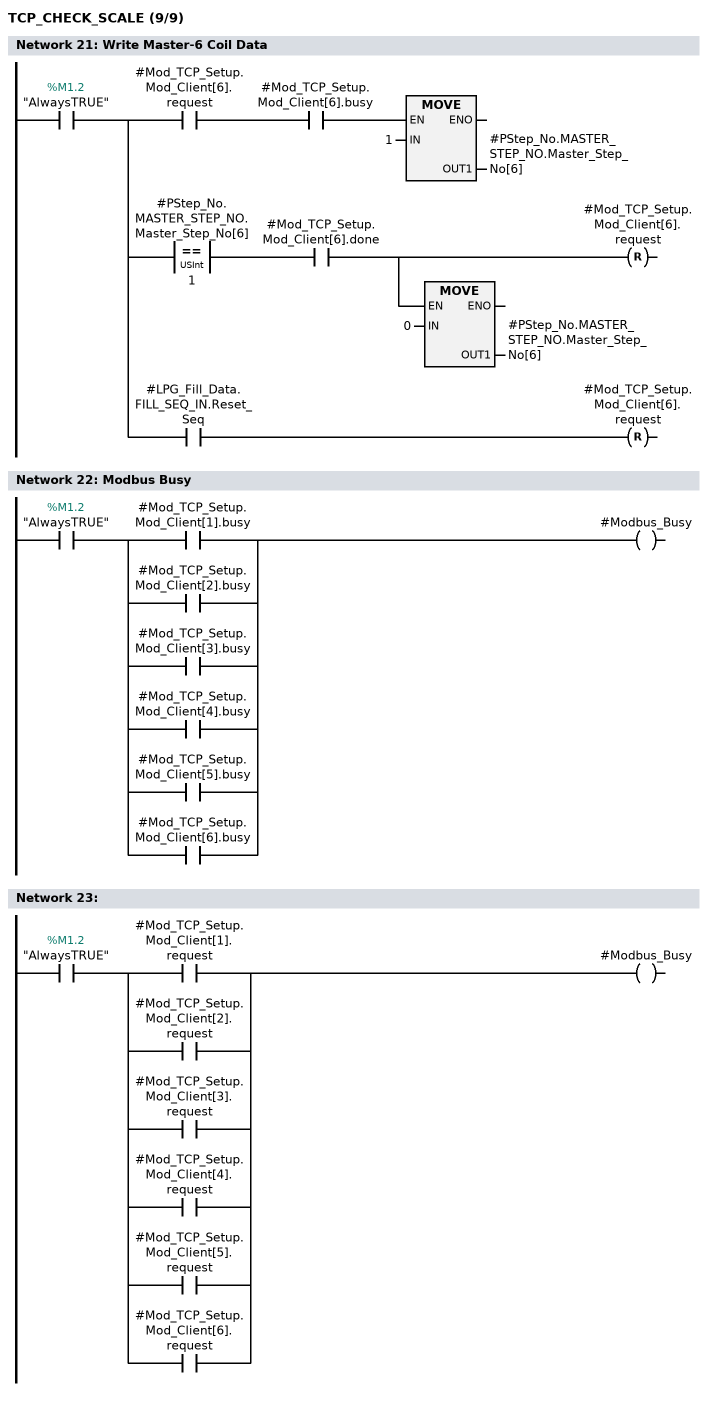
   RUNG wire#powerrail
      Contact( "AlwaysTRUE" )
      wire#w1
      Contact( #Mod_TCP_Setup.Mod_Client[6].request )
      Contact( #Mod_TCP_Setup.Mod_Client[6].busy )
      Move(in := 1, out1 => #PStep_No.MASTER_STEP_NO.Master_Step_No[6])
   END_RUNG
   RUNG wire#w1
      { S7_Templates := "SrcType := USInt" } EQ_Contact(in1 := #PStep_No.MASTER_STEP_NO.Master_Step_No[6], in2 := 1)
      Contact( #Mod_TCP_Setup.Mod_Client[6].done )
      wire#w2
      R_Coil( #Mod_TCP_Setup.Mod_Client[6].request )
   END_RUNG
   RUNG wire#w2
      Move(in := 0, out1 => #PStep_No.MASTER_STEP_NO.Master_Step_No[6])
   END_RUNG
   RUNG wire#w1
      Contact( #LPG_Fill_Data.FILL_SEQ_IN.Reset_Seq )
      R_Coil( #Mod_TCP_Setup.Mod_Client[6].request )
   END_RUNG
   // the same network as SCL:
   IF "AlwaysTRUE" AND #Mod_TCP_Setup.Mod_Client[6].request AND #Mod_TCP_Setup.Mod_Client[6].busy THEN
       #PStep_No.MASTER_STEP_NO.Master_Step_No[6] := 1;
   END_IF;
   #_w1 := "AlwaysTRUE" AND (#PStep_No.MASTER_STEP_NO.Master_Step_No[6] = 1) AND #Mod_TCP_Setup.Mod_Client[6].done;
   IF #_w1 THEN
       #Mod_TCP_Setup.Mod_Client[6].request := FALSE;
       #PStep_No.MASTER_STEP_NO.Master_Step_No[6] := 0;
   END_IF;
   IF "AlwaysTRUE" AND #LPG_Fill_Data.FILL_SEQ_IN.Reset_Seq THEN
       #Mod_TCP_Setup.Mod_Client[6].request := FALSE;
   END_IF;
END_REGION

REGION Network 22: Modbus Busy
   RUNG wire#powerrail
      Contact( "AlwaysTRUE" )
      wire#w1
      Contact( #Mod_TCP_Setup.Mod_Client[1].busy )
      wire#w2
      Coil( #Modbus_Busy )
   END_RUNG
   RUNG wire#w1
      Contact( #Mod_TCP_Setup.Mod_Client[2].busy )
   END_RUNG wire#w2
   RUNG wire#w1
      Contact( #Mod_TCP_Setup.Mod_Client[3].busy )
   END_RUNG wire#w2
   RUNG wire#w1
      Contact( #Mod_TCP_Setup.Mod_Client[4].busy )
   END_RUNG wire#w2
   RUNG wire#w1
      Contact( #Mod_TCP_Setup.Mod_Client[5].busy )
   END_RUNG wire#w2
   RUNG wire#w1
      Contact( #Mod_TCP_Setup.Mod_Client[6].busy )
   END_RUNG wire#w2
   // the same network as SCL:
   #Modbus_Busy := "AlwaysTRUE" AND (#Mod_TCP_Setup.Mod_Client[1].busy OR #Mod_TCP_Setup.Mod_Client[2].busy OR #Mod_TCP_Setup.Mod_Client[3].busy OR #Mod_TCP_Setup.Mod_Client[4].busy OR #Mod_TCP_Setup.Mod_Client[5].busy OR #Mod_TCP_Setup.Mod_Client[6].busy);
END_REGION

REGION Network 23
   RUNG wire#powerrail
      Contact( "AlwaysTRUE" )
      wire#w1
      Contact( #Mod_TCP_Setup.Mod_Client[1].request )
      wire#w2
      Coil( #Modbus_Busy )
   END_RUNG
   RUNG wire#w1
      Contact( #Mod_TCP_Setup.Mod_Client[2].request )
   END_RUNG wire#w2
   RUNG wire#w1
      Contact( #Mod_TCP_Setup.Mod_Client[3].request )
   END_RUNG wire#w2
   RUNG wire#w1
      Contact( #Mod_TCP_Setup.Mod_Client[4].request )
   END_RUNG wire#w2
   RUNG wire#w1
      Contact( #Mod_TCP_Setup.Mod_Client[5].request )
   END_RUNG wire#w2
   RUNG wire#w1
      Contact( #Mod_TCP_Setup.Mod_Client[6].request )
   END_RUNG wire#w2
   // the same network as SCL:
   #Modbus_Busy := "AlwaysTRUE" AND (#Mod_TCP_Setup.Mod_Client[1].request OR #Mod_TCP_Setup.Mod_Client[2].request OR #Mod_TCP_Setup.Mod_Client[3].request OR #Mod_TCP_Setup.Mod_Client[4].request OR #Mod_TCP_Setup.Mod_Client[5].request OR #Mod_TCP_Setup.Mod_Client[6].request);
END_REGION
END_FUNCTION_BLOCK

FUNCTION "CORRECTION_SCALE" : Void   // FC4, LAD
{ S7_Optimized_Access := 'TRUE' }
VERSION : 0.1
// stored: AutoNumber false, IsIECCheckEnabled false, SetENOAutomatically false, UDAEnableTagReadback false
   VAR_TEMP
      cycle_start : Bool;
   END_VAR
BEGIN

REGION Network 1
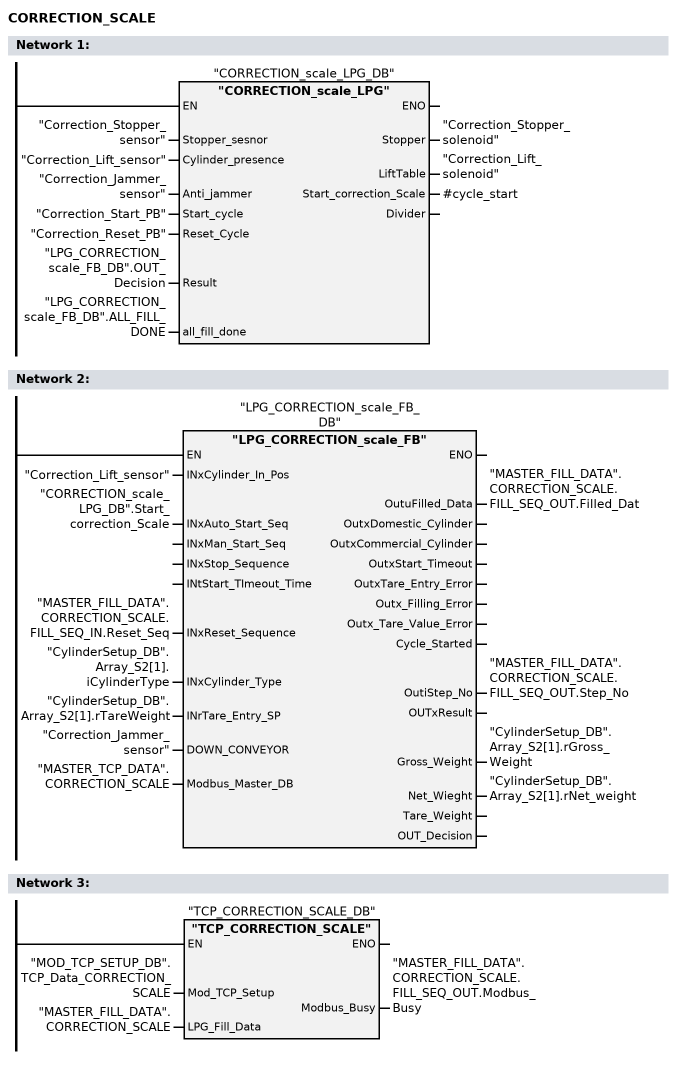
   RUNG wire#powerrail
      "CORRECTION_scale_LPG_DB"(Stopper_sesnor := "Correction_Stopper_sensor", Cylinder_presence := "Correction_Lift_sensor", Anti_jammer := "Correction_Jammer_sensor", Start_cycle := "Correction_Start_PB", Reset_Cycle := "Correction_Reset_PB", Result := "LPG_CORRECTION_scale_FB_DB".OUT_Decision, all_fill_done := "LPG_CORRECTION_scale_FB_DB".ALL_FILL_DONE, Stopper => "Correction_Stopper_solenoid", LiftTable => "Correction_Lift_solenoid", Start_correction_Scale => #cycle_start, Divider =>)
   END_RUNG
   // the same network as SCL:
   "CORRECTION_scale_LPG_DB"(Stopper_sesnor := "Correction_Stopper_sensor",   // "CORRECTION_scale_LPG"
                           Cylinder_presence := "Correction_Lift_sensor",
                           Anti_jammer := "Correction_Jammer_sensor",
                           Start_cycle := "Correction_Start_PB",
                           Reset_Cycle := "Correction_Reset_PB",
                           Result := "LPG_CORRECTION_scale_FB_DB".OUT_Decision,
                           all_fill_done := "LPG_CORRECTION_scale_FB_DB".ALL_FILL_DONE,
                           Stopper => "Correction_Stopper_solenoid",
                           LiftTable => "Correction_Lift_solenoid",
                           Start_correction_Scale => #cycle_start);
END_REGION

REGION Network 2
   RUNG wire#powerrail
      "LPG_CORRECTION_scale_FB_DB"(INxCylinder_In_Pos := "Correction_Lift_sensor", INxAuto_Start_Seq := "CORRECTION_scale_LPG_DB".Start_correction_Scale, INxMan_Start_Seq :=, INxStop_Sequence :=, INtStart_TImeout_Time :=, INxReset_Sequence := "MASTER_FILL_DATA".CORRECTION_SCALE.FILL_SEQ_IN.Reset_Seq, INxCylinder_Type := "CylinderSetup_DB".Array_S2[1].iCylinderType, INrTare_Entry_SP := "CylinderSetup_DB".Array_S2[1].rTareWeight, DOWN_CONVEYOR := "Correction_Jammer_sensor", Modbus_Master_DB := "MASTER_TCP_DATA".CORRECTION_SCALE, OutuFilled_Data => "MASTER_FILL_DATA".CORRECTION_SCALE.FILL_SEQ_OUT.Filled_Dat, OutxDomestic_Cylinder =>, OutxCommercial_Cylinder =>, OutxStart_Timeout =>, OutxTare_Entry_Error =>, Outx_Filling_Error =>, Outx_Tare_Value_Error =>, Cycle_Started =>, OutiStep_No => "MASTER_FILL_DATA".CORRECTION_SCALE.FILL_SEQ_OUT.Step_No, OUTxResult =>, Gross_Weight => "CylinderSetup_DB".Array_S2[1].rGross_Weight, Net_Wieght => "CylinderSetup_DB".Array_S2[1].rNet_weight, Tare_Weight =>, OUT_Decision =>)
   END_RUNG
   // the same network as SCL:
   "LPG_CORRECTION_scale_FB_DB"(INxCylinder_In_Pos := "Correction_Lift_sensor",   // "LPG_CORRECTION_scale_FB"
                           INxAuto_Start_Seq := "CORRECTION_scale_LPG_DB".Start_correction_Scale,
                           INxReset_Sequence := "MASTER_FILL_DATA".CORRECTION_SCALE.FILL_SEQ_IN.Reset_Seq,
                           INxCylinder_Type := "CylinderSetup_DB".Array_S2[1].iCylinderType,
                           INrTare_Entry_SP := "CylinderSetup_DB".Array_S2[1].rTareWeight,
                           DOWN_CONVEYOR := "Correction_Jammer_sensor",
                           Modbus_Master_DB := "MASTER_TCP_DATA".CORRECTION_SCALE,
                           OutuFilled_Data => "MASTER_FILL_DATA".CORRECTION_SCALE.FILL_SEQ_OUT.Filled_Dat,
                           OutiStep_No => "MASTER_FILL_DATA".CORRECTION_SCALE.FILL_SEQ_OUT.Step_No,
                           Gross_Weight => "CylinderSetup_DB".Array_S2[1].rGross_Weight,
                           Net_Wieght => "CylinderSetup_DB".Array_S2[1].rNet_weight);
END_REGION

REGION Network 3
   RUNG wire#powerrail
      "TCP_CORRECTION_SCALE_DB"(Mod_TCP_Setup := "MOD_TCP_SETUP_DB".TCP_Data_CORRECTION_SCALE, LPG_Fill_Data := "MASTER_FILL_DATA".CORRECTION_SCALE, Modbus_Busy => "MASTER_FILL_DATA".CORRECTION_SCALE.FILL_SEQ_OUT.Modbus_Busy)
   END_RUNG
   // the same network as SCL:
   "TCP_CORRECTION_SCALE_DB"(Mod_TCP_Setup := "MOD_TCP_SETUP_DB".TCP_Data_CORRECTION_SCALE,   // "TCP_CORRECTION_SCALE"
                           LPG_Fill_Data := "MASTER_FILL_DATA".CORRECTION_SCALE,
                           Modbus_Busy => "MASTER_FILL_DATA".CORRECTION_SCALE.FILL_SEQ_OUT.Modbus_Busy);
END_REGION
END_FUNCTION

FUNCTION_BLOCK "CORRECTION_scale_LPG"   // FB11, LAD
{ S7_Optimized_Access := 'TRUE' }
VERSION : 0.1
// stored: AutoNumber false, IsIECCheckEnabled false, IsRetainMemResEnabled false, MemoryReserve 100, SetENOAutomatically false, UDAEnableTagReadback false
   VAR_INPUT
      Stopper_sesnor : Bool;
      Cylinder_presence : Bool;
      Anti_jammer : Bool;
      Start_cycle : Bool;
      Reset_Cycle : Bool;
      Result : Int;
      all_fill_done : Bool;
   END_VAR
   VAR_OUTPUT
      Stopper : Bool;
      LiftTable : Bool;
      Start_correction_Scale : Bool;
      Divider : Bool;
   END_VAR
   VAR
      Check_Scale_Started : Bool;
      Lift_Table { S7_SetPoint := 'True'} : TON_TIME;
      PASS : Bool;
      FAIL : Bool;
      LIFT_down { S7_SetPoint := 'True'} : TON_TIME;
      checking { S7_SetPoint := 'True'} : TON_TIME;
      idx7 : Int;
      p_trig : Array[0..10] of Bool;
   END_VAR
   VAR RETAIN
      Stopper_count { S7_SetPoint := 'True'} : CTU_INT;
   END_VAR
   VAR
      counter_reset : Bool;
      datasend : Bool;
      Filling_done : Bool;
   END_VAR
   VAR_TEMP
      temp : Int;
   END_VAR
   VAR_TEMP   // added for the SCL form of the ladder/FBD networks
      _w1 : Bool;
      _w2 : Bool;
      _w3 : Bool;
   END_VAR
BEGIN

REGION Network 1
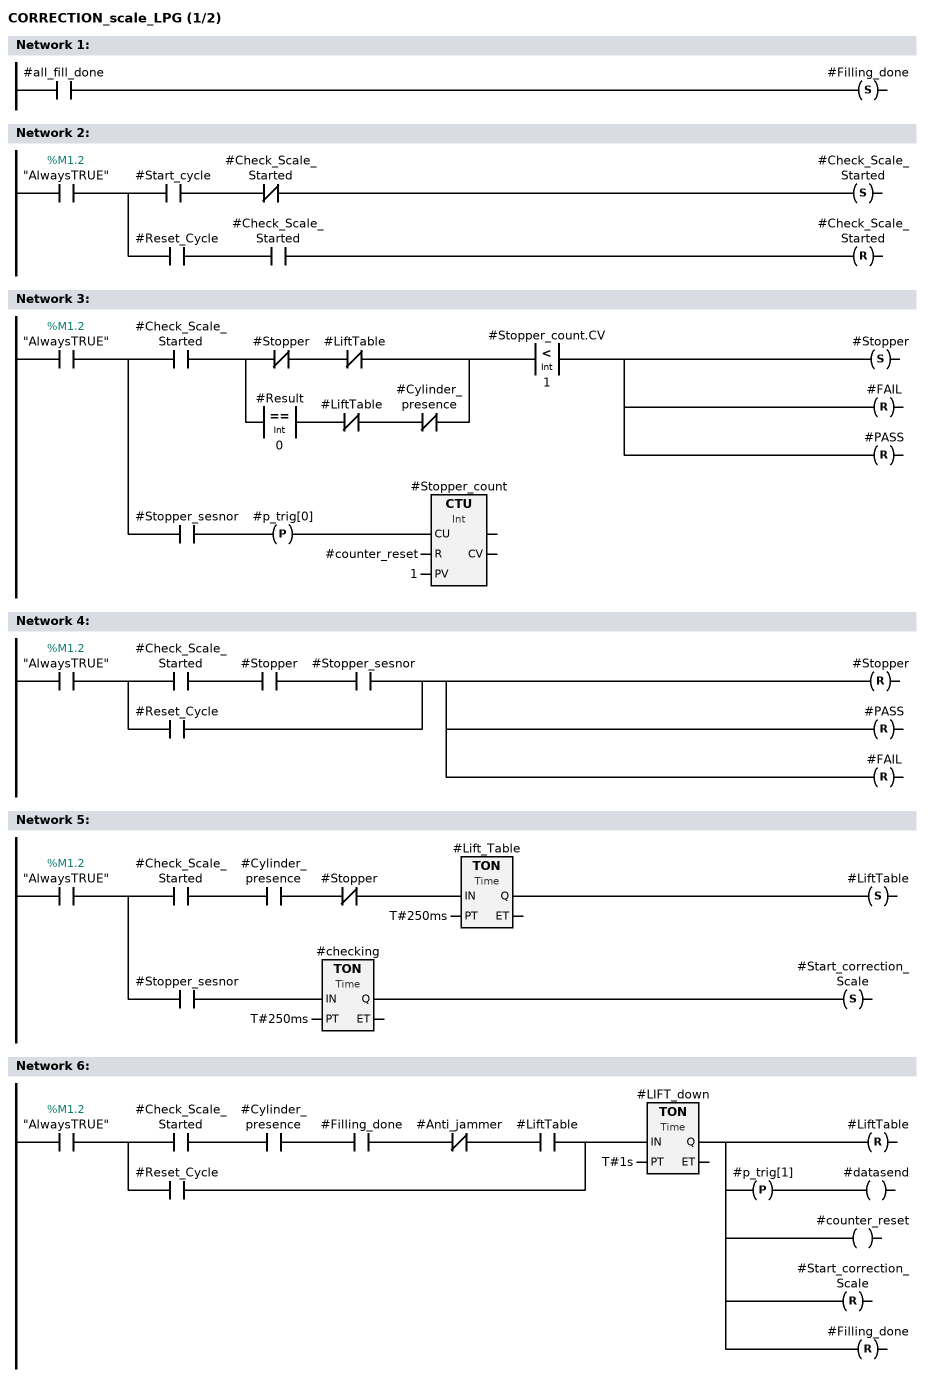
   RUNG wire#powerrail
      Contact( #all_fill_done )
      S_Coil( #Filling_done )
   END_RUNG
   // the same network as SCL:
   IF #all_fill_done THEN #Filling_done := TRUE; END_IF;
END_REGION

REGION Network 2
   RUNG wire#powerrail
      Contact( "AlwaysTRUE" )
      wire#w1
      Contact( #Start_cycle )
      I_Contact( #Check_Scale_Started )
      S_Coil( #Check_Scale_Started )
   END_RUNG
   RUNG wire#w1
      Contact( #Reset_Cycle )
      Contact( #Check_Scale_Started )
      R_Coil( #Check_Scale_Started )
   END_RUNG
   // the same network as SCL:
   IF "AlwaysTRUE" AND #Start_cycle AND NOT #Check_Scale_Started THEN #Check_Scale_Started := TRUE; END_IF;
   IF "AlwaysTRUE" AND #Reset_Cycle AND #Check_Scale_Started THEN #Check_Scale_Started := FALSE; END_IF;
END_REGION

REGION Network 3
   RUNG wire#powerrail
      Contact( "AlwaysTRUE" )
      wire#w1
      Contact( #Check_Scale_Started )
      wire#w2
      I_Contact( #Stopper )
      I_Contact( #LiftTable )
      wire#w3
      { S7_Templates := "SrcType := Int" } LT_Contact(in1 := #Stopper_count.CV, in2 := 1)
      wire#w4
      S_Coil( #Stopper )
   END_RUNG
   RUNG wire#w2
      { S7_Templates := "SrcType := Int" } EQ_Contact(in1 := #Result, in2 := 0)
      I_Contact( #LiftTable )
      I_Contact( #Cylinder_presence )
   END_RUNG wire#w3
   RUNG wire#w4
      R_Coil( #FAIL )
   END_RUNG
   RUNG wire#w4
      R_Coil( #PASS )
   END_RUNG
   RUNG wire#w1
      Contact( #Stopper_sesnor )
      P_Trig( #p_trig[0] )
      { S7_Templates := "value_type := Int" } #Stopper_count.CTU(r := #counter_reset, pv := 1, cv =>)
   END_RUNG
   // the same network as SCL:
   #_w1 := "AlwaysTRUE" AND #Check_Scale_Started AND ((NOT #Stopper AND NOT #LiftTable) OR ((#Result = 0) AND NOT #LiftTable AND NOT #Cylinder_presence)) AND (#Stopper_count.CV < 1);
   IF #_w1 THEN
       #Stopper := TRUE;
       #FAIL := FALSE;
       #PASS := FALSE;
   END_IF;
   #_w2 := "AlwaysTRUE" AND #Stopper_sesnor;
   #_w3 := #_w2 AND NOT #p_trig[0];   // rising edge
   #p_trig[0] := #_w2;
   #Stopper_count(CU := #_w3, R := #counter_reset, PV := 1);   // CTU
END_REGION

REGION Network 4
   RUNG wire#powerrail
      Contact( "AlwaysTRUE" )
      wire#w1
      Contact( #Check_Scale_Started )
      Contact( #Stopper )
      Contact( #Stopper_sesnor )
      wire#w2
      R_Coil( #Stopper )
   END_RUNG
   RUNG wire#w1
      Contact( #Reset_Cycle )
   END_RUNG wire#w2
   RUNG wire#w2
      R_Coil( #PASS )
   END_RUNG
   RUNG wire#w2
      R_Coil( #FAIL )
   END_RUNG
   // the same network as SCL:
   #_w1 := "AlwaysTRUE" AND ((#Check_Scale_Started AND #Stopper AND #Stopper_sesnor) OR #Reset_Cycle);
   IF #_w1 THEN
       #Stopper := FALSE;
       #PASS := FALSE;
       #FAIL := FALSE;
   END_IF;
END_REGION

REGION Network 5
   RUNG wire#powerrail
      Contact( "AlwaysTRUE" )
      wire#w1
      Contact( #Check_Scale_Started )
      Contact( #Cylinder_presence )
      I_Contact( #Stopper )
      { S7_Templates := "time_type := Time" } #Lift_Table.TON(pt := T#250ms, et =>)
      S_Coil( #LiftTable )
   END_RUNG
   RUNG wire#w1
      Contact( #Stopper_sesnor )
      { S7_Templates := "time_type := Time" } #checking.TON(pt := T#250ms, et =>)
      S_Coil( #Start_correction_Scale )
   END_RUNG
   // the same network as SCL:
   #Lift_Table(IN := "AlwaysTRUE" AND #Check_Scale_Started AND #Cylinder_presence AND NOT #Stopper,   // TON
               PT := T#250ms);
   IF #Lift_Table.Q THEN #LiftTable := TRUE; END_IF;
   #checking(IN := "AlwaysTRUE" AND #Stopper_sesnor, PT := T#250ms);   // TON
   IF #checking.Q THEN #Start_correction_Scale := TRUE; END_IF;
END_REGION

REGION Network 6
   RUNG wire#powerrail
      Contact( "AlwaysTRUE" )
      wire#w1
      Contact( #Check_Scale_Started )
      Contact( #Cylinder_presence )
      Contact( #Filling_done )
      I_Contact( #Anti_jammer )
      Contact( #LiftTable )
      wire#w2
      { S7_Templates := "time_type := Time" } #LIFT_down.TON(pt := T#1s, et =>)
      wire#w3
      R_Coil( #LiftTable )
   END_RUNG
   RUNG wire#w1
      Contact( #Reset_Cycle )
   END_RUNG wire#w2
   RUNG wire#w3
      P_Trig( #p_trig[1] )
      Coil( #datasend )
   END_RUNG
   RUNG wire#w3
      Coil( #counter_reset )
   END_RUNG
   RUNG wire#w3
      R_Coil( #Start_correction_Scale )
   END_RUNG
   RUNG wire#w3
      R_Coil( #Filling_done )
   END_RUNG
   // the same network as SCL:
   #LIFT_down(IN := "AlwaysTRUE" AND ((#Check_Scale_Started AND #Cylinder_presence AND #Filling_done AND NOT #Anti_jammer AND #LiftTable) OR #Reset_Cycle),   // TON
              PT := T#1s);
   IF #LIFT_down.Q THEN #LiftTable := FALSE; END_IF;
   #_w1 := #LIFT_down.Q AND NOT #p_trig[1];   // rising edge
   #p_trig[1] := #LIFT_down.Q;
   #datasend := #_w1;
   #counter_reset := #LIFT_down.Q;
   IF #LIFT_down.Q THEN
       #Start_correction_Scale := FALSE;
       #Filling_done := FALSE;
   END_IF;
END_REGION

REGION Network 7
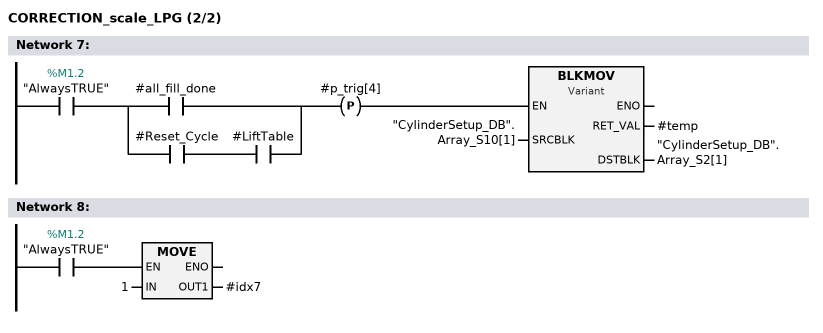
   RUNG wire#powerrail
      Contact( "AlwaysTRUE" )
      wire#w1
      Contact( #all_fill_done )
      wire#w2
      P_Trig( #p_trig[4] )
      { S7_Templates := "blk_type := Variant" } BLKMOV(SRCBLK := "CylinderSetup_DB".Array_S10[1], RET_VAL => #temp, DSTBLK => "CylinderSetup_DB".Array_S2[1])
   END_RUNG
   RUNG wire#w1
      Contact( #Reset_Cycle )
      Contact( #LiftTable )
   END_RUNG wire#w2
   // the same network as SCL:
   #_w1 := "AlwaysTRUE" AND (#all_fill_done OR (#Reset_Cycle AND #LiftTable));
   #_w2 := #_w1 AND NOT #p_trig[4];   // rising edge
   #p_trig[4] := #_w1;
   IF #_w2 THEN
       #temp := BLKMOV(SRCBLK := "CylinderSetup_DB".Array_S10[1], DSTBLK => "CylinderSetup_DB".Array_S2[1]);
   END_IF;
END_REGION

REGION Network 8
   RUNG wire#powerrail
      Contact( "AlwaysTRUE" )
      Move(in := 1, out1 => #idx7)
   END_RUNG
   // the same network as SCL:
   IF "AlwaysTRUE" THEN #idx7 := 1; END_IF;
END_REGION
END_FUNCTION_BLOCK

FUNCTION_BLOCK "LPG_CORRECTION_scale_FB"   // FB103, LAD
TITLE = Fiiling Operation FB
{ S7_Optimized_Access := 'TRUE' }
VERSION : 0.1
// stored: AutoNumber false, IsIECCheckEnabled false, IsRetainMemResEnabled false, MemoryReserve 100, SetENOAutomatically false, UDAEnableTagReadback false
   VAR_INPUT
      INxCylinder_In_Pos : Bool;   // Cylinder In Position
      INxAuto_Start_Seq : Bool;   // Start Filling Sequence
      INxMan_Start_Seq : Bool;
      INxStop_Sequence : Bool;   // Stop Filling Sequence
      INtStart_TImeout_Time : DInt;   // Start Timeout Time in Sec
      INxReset_Sequence : Bool;   // Reset Sequence
      INxCylinder_Type : Int;
      INrTare_Entry_SP : Real;
      DOWN_CONVEYOR : Bool;
   END_VAR
   VAR_OUTPUT
      OutuFilled_Data : Array[1..3] of Real;
      OutxDomestic_Cylinder : Bool;
      OutxCommercial_Cylinder : Bool;
      OutxStart_Timeout : Bool;
      OutxTare_Entry_Error : Bool;   // Coil 27
      Outx_Filling_Error : Bool;
      Outx_Tare_Value_Error : Bool;
      Cycle_Started : Bool;
      OutiStep_No : Int;
      OUTxResult : Bool;
      Gross_Weight : Real;
      Net_Wieght : Real;
      Tare_Weight : Real;
      OUT_Decision : Int;
   END_VAR
   VAR_IN_OUT
      Modbus_Master_DB : "MOD_MASTER_DATA_1";
   END_VAR
   VAR
      TRIG : Array[1..25] of Bool;
      STEP_NO : Int;
      Step_Timer { S7_SetPoint := 'True'} : Array[1..15] of IEC_TIMER;
      Domestic_Cylinder { S7_SetPoint := 'True'} : Bool;
      Commercial_Cylinder : Bool;
      Cyl_Done { S7_SetPoint := 'True'} : TOF_TIME;
      Tare_Enrty_Extn { S7_SetPoint := 'True'} : TOF_TIME;
      Start_Timeout_Err { S7_SetPoint := 'True'} : TON_TIME;
      Tare_Entry_Timer { S7_SetPoint := 'True'} : TON_TIME;
      Filled_Gross : Real;
      Filled_Net : Real;
      Punched_Tare : Real;
      Test_Seq : Int;
      RESULT : Bool;
      IEC_Timer_0_Instance { S7_SetPoint := 'True'} : TOF_TIME;
      Gross { S7_SetPoint := 'True'} : Real;
      gross_diff : Real;
      pass : Bool;
      Decision : Word;
      ALL_FILL_DONE : Bool;
      fill { S7_SetPoint := 'True'} : TON_TIME;
      IEC_Timer_0_Instance_1 { S7_SetPoint := 'True'} : TON_TIME;
   END_VAR
   VAR_TEMP
      Tare_Weight_Mul : Real;
      Tare_Enter_Time : DInt;
      Stt_TImeout_Time : DInt;
      Tare_Entry_Time : DInt;
      Tare_SP_Weigher : Int;
      Filled_Gross_Mul : Int;
      Filled_Net_Mul : Int;
      Filled_Tare_Mul : Int;
      "final wieght" : Real;
      final_weight_1 : Real;
   END_VAR
   // Tare_Enrty_Extn.PT := T#1s;
   VAR_TEMP   // added for the SCL form of the ladder/FBD networks
      _w1 : Bool;
      _w2 : Bool;
      _w3 : Bool;
   END_VAR
BEGIN

REGION Network 1: Empty Network
END_REGION

REGION Network 2: Input Mapping
END_REGION

REGION Network 3: Cylinder Selection ( Domestic / Commercial )
   // We have to receive from FIFO Entry-
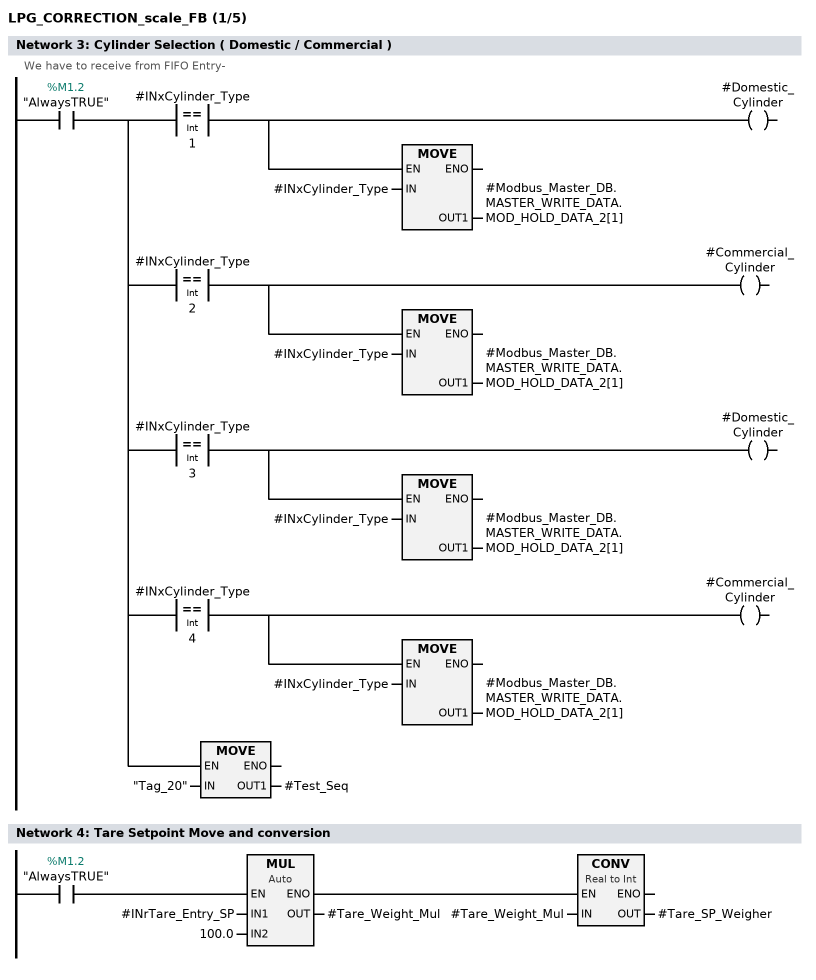
   RUNG wire#powerrail
      Contact( "AlwaysTRUE" )
      wire#w1
      { S7_Templates := "SrcType := Int" } EQ_Contact(in1 := #INxCylinder_Type, in2 := 1)
      wire#w2
      Coil( #Domestic_Cylinder )
   END_RUNG
   RUNG wire#w2
      Move(in := #INxCylinder_Type, out1 => #Modbus_Master_DB.MASTER_WRITE_DATA.MOD_HOLD_DATA_2[1])
   END_RUNG
   RUNG wire#w1
      { S7_Templates := "SrcType := Int" } EQ_Contact(in1 := #INxCylinder_Type, in2 := 2)
      wire#w3
      Coil( #Commercial_Cylinder )
   END_RUNG
   RUNG wire#w3
      Move(in := #INxCylinder_Type, out1 => #Modbus_Master_DB.MASTER_WRITE_DATA.MOD_HOLD_DATA_2[1])
   END_RUNG
   RUNG wire#w1
      { S7_Templates := "SrcType := Int" } EQ_Contact(in1 := #INxCylinder_Type, in2 := 3)
      wire#w4
      Coil( #Domestic_Cylinder )
   END_RUNG
   RUNG wire#w4
      Move(in := #INxCylinder_Type, out1 => #Modbus_Master_DB.MASTER_WRITE_DATA.MOD_HOLD_DATA_2[1])
   END_RUNG
   RUNG wire#w1
      { S7_Templates := "SrcType := Int" } EQ_Contact(in1 := #INxCylinder_Type, in2 := 4)
      wire#w5
      Coil( #Commercial_Cylinder )
   END_RUNG
   RUNG wire#w5
      Move(in := #INxCylinder_Type, out1 => #Modbus_Master_DB.MASTER_WRITE_DATA.MOD_HOLD_DATA_2[1])
   END_RUNG
   RUNG wire#w1
      Move(in := "Tag_20", out1 => #Test_Seq)
   END_RUNG
   // the same network as SCL:
   #Domestic_Cylinder := "AlwaysTRUE" AND (#INxCylinder_Type = 1);
   IF #Domestic_Cylinder THEN
       #Modbus_Master_DB.MASTER_WRITE_DATA.MOD_HOLD_DATA_2[1] := #INxCylinder_Type;
   END_IF;
   #Commercial_Cylinder := "AlwaysTRUE" AND (#INxCylinder_Type = 2);
   IF #Commercial_Cylinder THEN
       #Modbus_Master_DB.MASTER_WRITE_DATA.MOD_HOLD_DATA_2[1] := #INxCylinder_Type;
   END_IF;
   #Domestic_Cylinder := "AlwaysTRUE" AND (#INxCylinder_Type = 3);
   IF #Domestic_Cylinder THEN
       #Modbus_Master_DB.MASTER_WRITE_DATA.MOD_HOLD_DATA_2[1] := #INxCylinder_Type;
   END_IF;
   #Commercial_Cylinder := "AlwaysTRUE" AND (#INxCylinder_Type = 4);
   IF #Commercial_Cylinder THEN
       #Modbus_Master_DB.MASTER_WRITE_DATA.MOD_HOLD_DATA_2[1] := #INxCylinder_Type;
   END_IF;
   IF "AlwaysTRUE" THEN #Test_Seq := "Tag_20"; END_IF;
END_REGION

REGION Network 4: Tare Setpoint Move and conversion
   RUNG wire#powerrail
      Contact( "AlwaysTRUE" )
      Mul(in1 := #INrTare_Entry_SP, in2 := 100.0, out => #Tare_Weight_Mul)
      { S7_Templates := "[SrcType := Real, DestType := Int]" } Convert(in := #Tare_Weight_Mul, out => #Tare_SP_Weigher)
   END_RUNG
   // the same network as SCL:
   IF "AlwaysTRUE" THEN
       #Tare_Weight_Mul := #INrTare_Entry_SP * 100.0;
       #Tare_SP_Weigher := REAL_TO_INT(#Tare_Weight_Mul);
   END_IF;
END_REGION

REGION Network 5: Cylinder Selection
   // Cylinder Selection will write the logic later
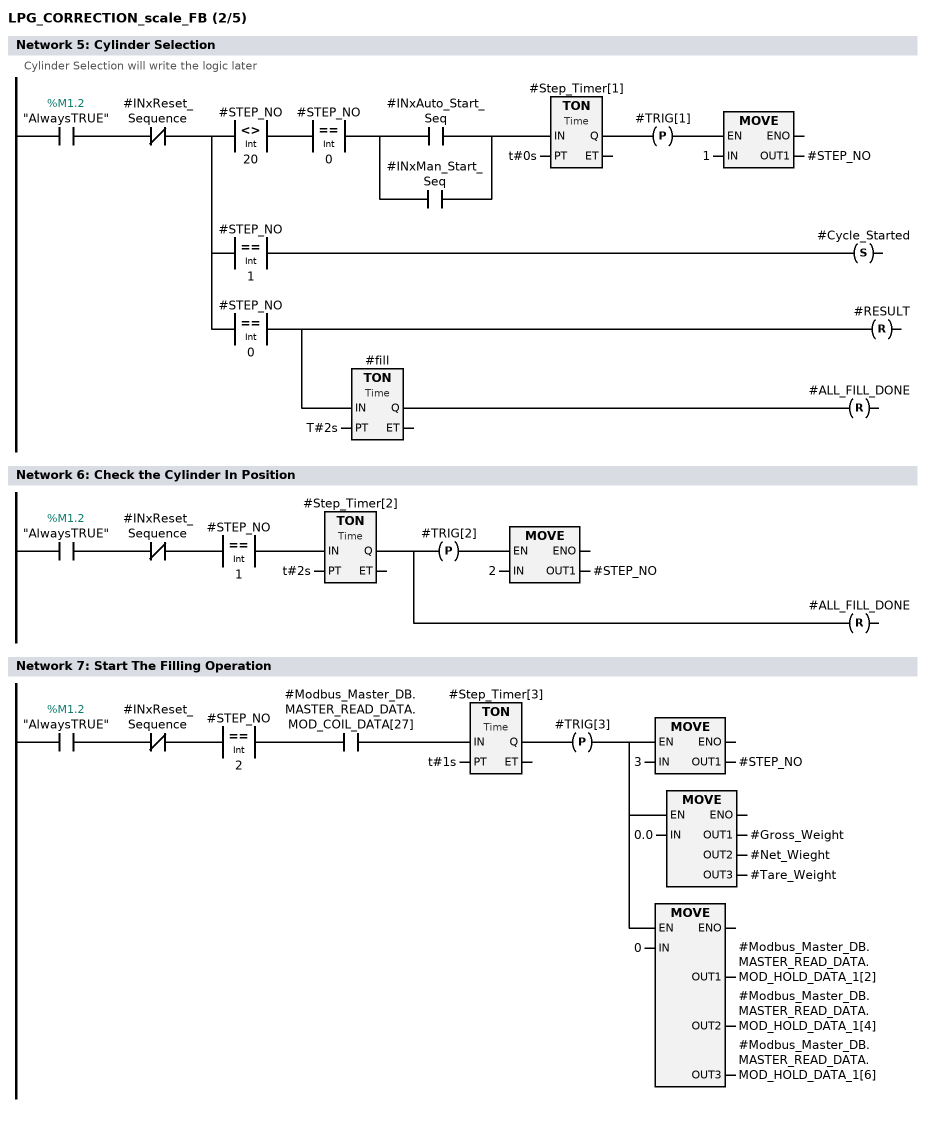
   RUNG wire#powerrail
      Contact( "AlwaysTRUE" )
      I_Contact( #INxReset_Sequence )
      wire#w1
      { S7_Templates := "SrcType := Int" } NE_Contact(in1 := #STEP_NO, in2 := 20)
      { S7_Templates := "SrcType := Int" } EQ_Contact(in1 := #STEP_NO, in2 := 0)
      wire#w2
      Contact( #INxAuto_Start_Seq )
      wire#w3
      { S7_Templates := "time_type := Time" } #Step_Timer[1].TON(pt := t#0s, et =>)
      P_Trig( #TRIG[1] )
      Move(in := 1, out1 => #STEP_NO)
   END_RUNG
   RUNG wire#w2
      Contact( #INxMan_Start_Seq )
   END_RUNG wire#w3
   RUNG wire#w1
      { S7_Templates := "SrcType := Int" } EQ_Contact(in1 := #STEP_NO, in2 := 1)
      S_Coil( #Cycle_Started )
   END_RUNG
   RUNG wire#w1
      { S7_Templates := "SrcType := Int" } EQ_Contact(in1 := #STEP_NO, in2 := 0)
      wire#w4
      R_Coil( #RESULT )
   END_RUNG
   RUNG wire#w4
      { S7_Templates := "time_type := Time" } #fill.TON(pt := T#2s, et =>)
      R_Coil( #ALL_FILL_DONE )
   END_RUNG
   // the same network as SCL:
   #_w1 := "AlwaysTRUE" AND NOT #INxReset_Sequence;
   #Step_Timer[1].TON(IN := #_w1 AND (#STEP_NO <> 20) AND (#STEP_NO = 0) AND (#INxAuto_Start_Seq OR #INxMan_Start_Seq),
                      PT := t#0s);
   #_w2 := #Step_Timer[1].Q AND NOT #TRIG[1];   // rising edge
   #TRIG[1] := #Step_Timer[1].Q;
   IF #_w2 THEN #STEP_NO := 1; END_IF;
   IF #_w1 AND (#STEP_NO = 1) THEN #Cycle_Started := TRUE; END_IF;
   #_w3 := #_w1 AND (#STEP_NO = 0);
   IF #_w3 THEN #RESULT := FALSE; END_IF;
   #fill(IN := #_w3, PT := T#2s);   // TON
   IF #fill.Q THEN #ALL_FILL_DONE := FALSE; END_IF;
END_REGION

REGION Network 6: Check the Cylinder In Position
   RUNG wire#powerrail
      Contact( "AlwaysTRUE" )
      I_Contact( #INxReset_Sequence )
      { S7_Templates := "SrcType := Int" } EQ_Contact(in1 := #STEP_NO, in2 := 1)
      { S7_Templates := "time_type := Time" } #Step_Timer[2].TON(pt := t#2s, et =>)
      wire#w1
      P_Trig( #TRIG[2] )
      Move(in := 2, out1 => #STEP_NO)
   END_RUNG
   RUNG wire#w1
      R_Coil( #ALL_FILL_DONE )
   END_RUNG
   // the same network as SCL:
   #Step_Timer[2].TON(IN := "AlwaysTRUE" AND NOT #INxReset_Sequence AND (#STEP_NO = 1), PT := t#2s);
   #_w1 := #Step_Timer[2].Q AND NOT #TRIG[2];   // rising edge
   #TRIG[2] := #Step_Timer[2].Q;
   IF #_w1 THEN #STEP_NO := 2; END_IF;
   IF #Step_Timer[2].Q THEN #ALL_FILL_DONE := FALSE; END_IF;
END_REGION

REGION Network 7: Start The Filling Operation
   RUNG wire#powerrail
      Contact( "AlwaysTRUE" )
      I_Contact( #INxReset_Sequence )
      { S7_Templates := "SrcType := Int" } EQ_Contact(in1 := #STEP_NO, in2 := 2)
      Contact( #Modbus_Master_DB.MASTER_READ_DATA.MOD_COIL_DATA[27] )
      { S7_Templates := "time_type := Time" } #Step_Timer[3].TON(pt := t#1s, et =>)
      P_Trig( #TRIG[3] )
      wire#w1
      Move(in := 3, out1 => #STEP_NO)
   END_RUNG
   RUNG wire#w1
      Move(in := 0.0, out1 => #Gross_Weight, out2 => #Net_Wieght, out3 => #Tare_Weight)
   END_RUNG
   RUNG wire#w1
      Move(in := 0, out1 => #Modbus_Master_DB.MASTER_READ_DATA.MOD_HOLD_DATA_1[2], out2 => #Modbus_Master_DB.MASTER_READ_DATA.MOD_HOLD_DATA_1[4], out3 => #Modbus_Master_DB.MASTER_READ_DATA.MOD_HOLD_DATA_1[6])
   END_RUNG
   // the same network as SCL:
   #Step_Timer[3].TON(IN := "AlwaysTRUE" AND NOT #INxReset_Sequence AND (#STEP_NO = 2) AND #Modbus_Master_DB.MASTER_READ_DATA.MOD_COIL_DATA[27],
                      PT := t#1s);
   #_w1 := #Step_Timer[3].Q AND NOT #TRIG[3];   // rising edge
   #TRIG[3] := #Step_Timer[3].Q;
   IF #_w1 THEN
       #STEP_NO := 3;
       #Gross_Weight := 0.0;
       #Net_Wieght := 0.0;
       #Tare_Weight := 0.0;
       #Modbus_Master_DB.MASTER_READ_DATA.MOD_HOLD_DATA_1[2] := 0;
       #Modbus_Master_DB.MASTER_READ_DATA.MOD_HOLD_DATA_1[4] := 0;
       #Modbus_Master_DB.MASTER_READ_DATA.MOD_HOLD_DATA_1[6] := 0;
   END_IF;
END_REGION

REGION Network 8: Check the Tare Weight Mode and Tare Entry
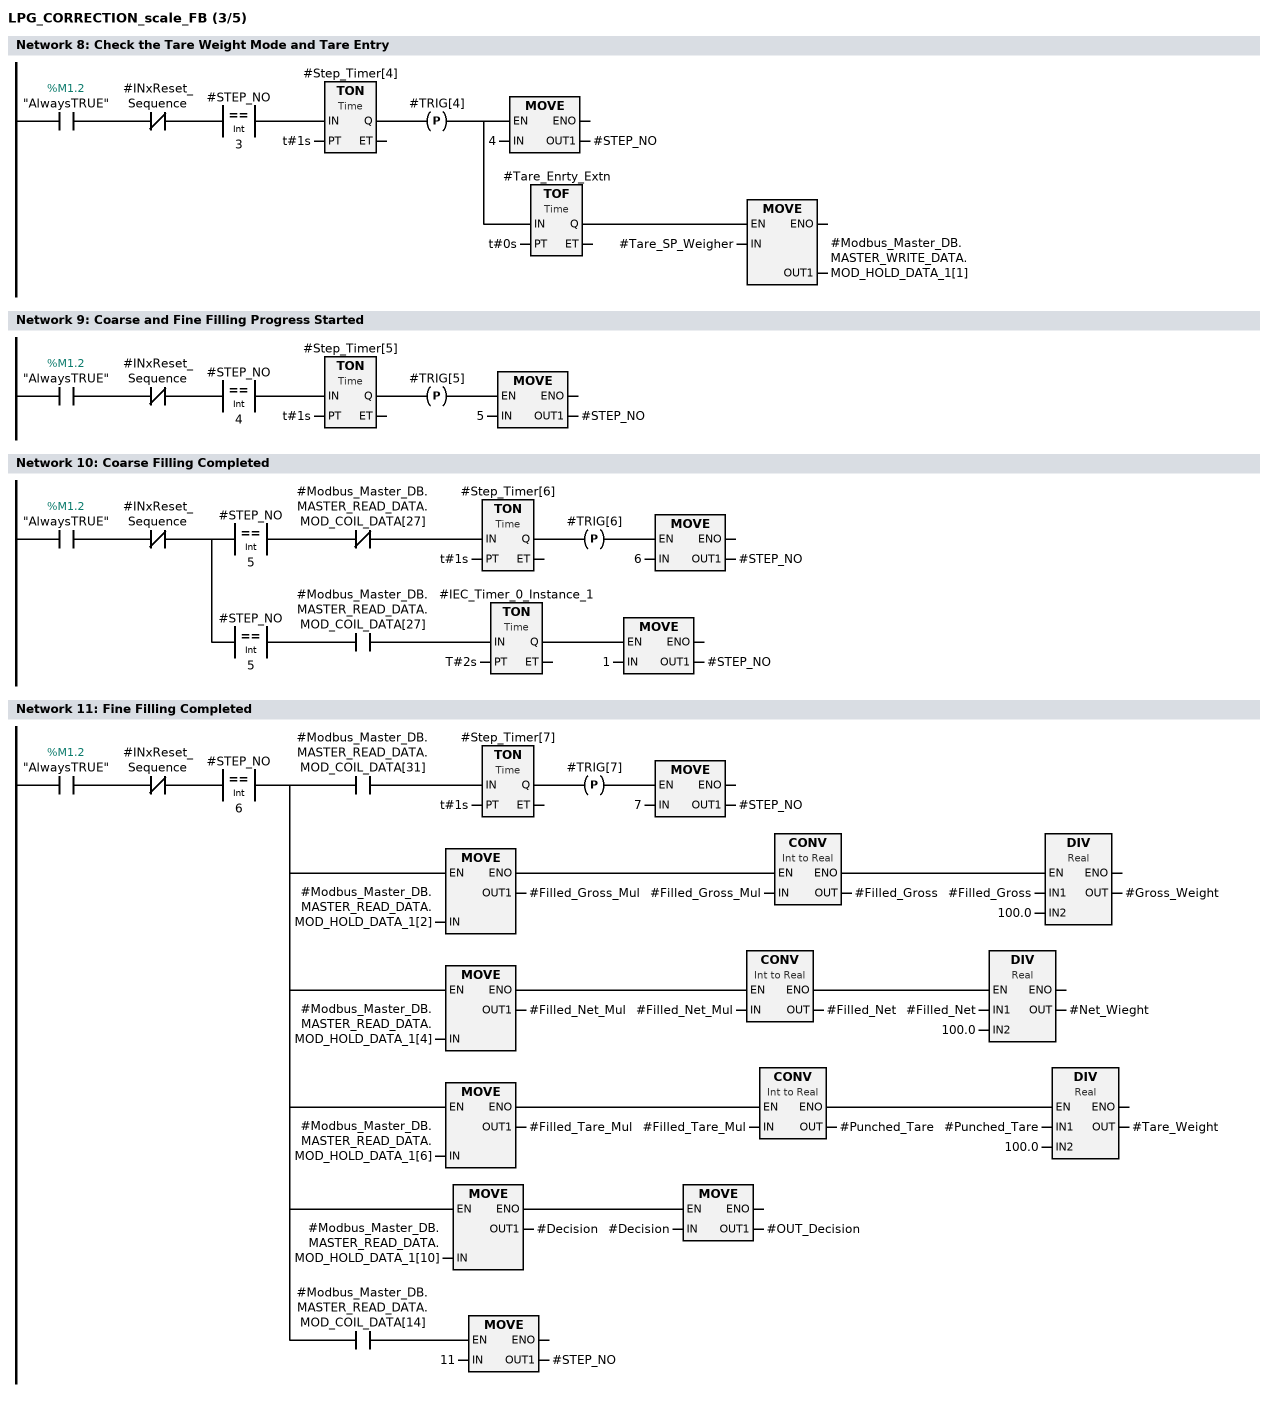
   RUNG wire#powerrail
      Contact( "AlwaysTRUE" )
      I_Contact( #INxReset_Sequence )
      { S7_Templates := "SrcType := Int" } EQ_Contact(in1 := #STEP_NO, in2 := 3)
      { S7_Templates := "time_type := Time" } #Step_Timer[4].TON(pt := t#1s, et =>)
      P_Trig( #TRIG[4] )
      wire#w1
      Move(in := 4, out1 => #STEP_NO)
   END_RUNG
   RUNG wire#w1
      { S7_Templates := "time_type := Time" } #Tare_Enrty_Extn.TOF(pt := t#0s, et =>)
      Move(in := #Tare_SP_Weigher, out1 => #Modbus_Master_DB.MASTER_WRITE_DATA.MOD_HOLD_DATA_1[1])
   END_RUNG
   // the same network as SCL:
   #Step_Timer[4].TON(IN := "AlwaysTRUE" AND NOT #INxReset_Sequence AND (#STEP_NO = 3), PT := t#1s);
   #_w1 := #Step_Timer[4].Q AND NOT #TRIG[4];   // rising edge
   #TRIG[4] := #Step_Timer[4].Q;
   IF #_w1 THEN #STEP_NO := 4; END_IF;
   #Tare_Enrty_Extn(IN := #_w1, PT := t#0s);   // TOF
   IF #Tare_Enrty_Extn.Q THEN
       #Modbus_Master_DB.MASTER_WRITE_DATA.MOD_HOLD_DATA_1[1] := #Tare_SP_Weigher;
   END_IF;
END_REGION

REGION Network 9: Coarse and Fine Filling Progress Started
   RUNG wire#powerrail
      Contact( "AlwaysTRUE" )
      I_Contact( #INxReset_Sequence )
      { S7_Templates := "SrcType := Int" } EQ_Contact(in1 := #STEP_NO, in2 := 4)
      { S7_Templates := "time_type := Time" } #Step_Timer[5].TON(pt := t#1s, et =>)
      P_Trig( #TRIG[5] )
      Move(in := 5, out1 => #STEP_NO)
   END_RUNG
   // the same network as SCL:
   #Step_Timer[5].TON(IN := "AlwaysTRUE" AND NOT #INxReset_Sequence AND (#STEP_NO = 4), PT := t#1s);
   #_w1 := #Step_Timer[5].Q AND NOT #TRIG[5];   // rising edge
   #TRIG[5] := #Step_Timer[5].Q;
   IF #_w1 THEN #STEP_NO := 5; END_IF;
END_REGION

REGION Network 10: Coarse Filling Completed
   RUNG wire#powerrail
      Contact( "AlwaysTRUE" )
      I_Contact( #INxReset_Sequence )
      wire#w1
      { S7_Templates := "SrcType := Int" } EQ_Contact(in1 := #STEP_NO, in2 := 5)
      I_Contact( #Modbus_Master_DB.MASTER_READ_DATA.MOD_COIL_DATA[27] )
      { S7_Templates := "time_type := Time" } #Step_Timer[6].TON(pt := t#1s, et =>)
      P_Trig( #TRIG[6] )
      Move(in := 6, out1 => #STEP_NO)
   END_RUNG
   RUNG wire#w1
      { S7_Templates := "SrcType := Int" } EQ_Contact(in1 := #STEP_NO, in2 := 5)
      Contact( #Modbus_Master_DB.MASTER_READ_DATA.MOD_COIL_DATA[27] )
      { S7_Templates := "time_type := Time" } #IEC_Timer_0_Instance_1.TON(pt := T#2s, et =>)
      Move(in := 1, out1 => #STEP_NO)
   END_RUNG
   // the same network as SCL:
   #_w1 := "AlwaysTRUE" AND NOT #INxReset_Sequence;
   #Step_Timer[6].TON(IN := #_w1 AND (#STEP_NO = 5) AND NOT #Modbus_Master_DB.MASTER_READ_DATA.MOD_COIL_DATA[27],
                      PT := t#1s);
   #_w2 := #Step_Timer[6].Q AND NOT #TRIG[6];   // rising edge
   #TRIG[6] := #Step_Timer[6].Q;
   IF #_w2 THEN #STEP_NO := 6; END_IF;
   #IEC_Timer_0_Instance_1(IN := #_w1 AND (#STEP_NO = 5) AND #Modbus_Master_DB.MASTER_READ_DATA.MOD_COIL_DATA[27],   // TON
                           PT := T#2s);
   IF #IEC_Timer_0_Instance_1.Q THEN #STEP_NO := 1; END_IF;
END_REGION

REGION Network 11: Fine Filling Completed
   RUNG wire#powerrail
      Contact( "AlwaysTRUE" )
      I_Contact( #INxReset_Sequence )
      { S7_Templates := "SrcType := Int" } EQ_Contact(in1 := #STEP_NO, in2 := 6)
      wire#w1
      Contact( #Modbus_Master_DB.MASTER_READ_DATA.MOD_COIL_DATA[31] )
      { S7_Templates := "time_type := Time" } #Step_Timer[7].TON(pt := t#1s, et =>)
      P_Trig( #TRIG[7] )
      Move(in := 7, out1 => #STEP_NO)
   END_RUNG
   RUNG wire#w1
      Move(in := #Modbus_Master_DB.MASTER_READ_DATA.MOD_HOLD_DATA_1[2], out1 => #Filled_Gross_Mul)
      { S7_Templates := "[SrcType := Int, DestType := Real]" } Convert(in := #Filled_Gross_Mul, out => #Filled_Gross)
      { S7_Templates := "SrcType := Real" } Div(in1 := #Filled_Gross, in2 := 100.0, out => #Gross_Weight)
   END_RUNG
   RUNG wire#w1
      Move(in := #Modbus_Master_DB.MASTER_READ_DATA.MOD_HOLD_DATA_1[4], out1 => #Filled_Net_Mul)
      { S7_Templates := "[SrcType := Int, DestType := Real]" } Convert(in := #Filled_Net_Mul, out => #Filled_Net)
      { S7_Templates := "SrcType := Real" } Div(in1 := #Filled_Net, in2 := 100.0, out => #Net_Wieght)
   END_RUNG
   RUNG wire#w1
      Move(in := #Modbus_Master_DB.MASTER_READ_DATA.MOD_HOLD_DATA_1[6], out1 => #Filled_Tare_Mul)
      { S7_Templates := "[SrcType := Int, DestType := Real]" } Convert(in := #Filled_Tare_Mul, out => #Punched_Tare)
      { S7_Templates := "SrcType := Real" } Div(in1 := #Punched_Tare, in2 := 100.0, out => #Tare_Weight)
   END_RUNG
   RUNG wire#w1
      Move(in := #Modbus_Master_DB.MASTER_READ_DATA.MOD_HOLD_DATA_1[10], out1 => #Decision)
      Move(in := #Decision, out1 => #OUT_Decision)
   END_RUNG
   RUNG wire#w1
      Contact( #Modbus_Master_DB.MASTER_READ_DATA.MOD_COIL_DATA[14] )
      Move(in := 11, out1 => #STEP_NO)
   END_RUNG
   // the same network as SCL:
   #_w1 := "AlwaysTRUE" AND NOT #INxReset_Sequence AND (#STEP_NO = 6);
   #Step_Timer[7].TON(IN := #_w1 AND #Modbus_Master_DB.MASTER_READ_DATA.MOD_COIL_DATA[31], PT := t#1s);
   #_w2 := #Step_Timer[7].Q AND NOT #TRIG[7];   // rising edge
   #TRIG[7] := #Step_Timer[7].Q;
   IF #_w2 THEN #STEP_NO := 7; END_IF;
   IF #_w1 THEN
       #Filled_Gross_Mul := #Modbus_Master_DB.MASTER_READ_DATA.MOD_HOLD_DATA_1[2];
       #Filled_Gross := INT_TO_REAL(#Filled_Gross_Mul);
       #Gross_Weight := #Filled_Gross / 100.0;
       #Filled_Net_Mul := #Modbus_Master_DB.MASTER_READ_DATA.MOD_HOLD_DATA_1[4];
       #Filled_Net := INT_TO_REAL(#Filled_Net_Mul);
       #Net_Wieght := #Filled_Net / 100.0;
       #Filled_Tare_Mul := #Modbus_Master_DB.MASTER_READ_DATA.MOD_HOLD_DATA_1[6];
       #Punched_Tare := INT_TO_REAL(#Filled_Tare_Mul);
       #Tare_Weight := #Punched_Tare / 100.0;
       #Decision := #Modbus_Master_DB.MASTER_READ_DATA.MOD_HOLD_DATA_1[10];
       #OUT_Decision := #Decision;
   END_IF;
   IF #_w1 AND #Modbus_Master_DB.MASTER_READ_DATA.MOD_COIL_DATA[14] THEN #STEP_NO := 11; END_IF;
END_REGION

REGION Network 12: Fill Over Flag Check
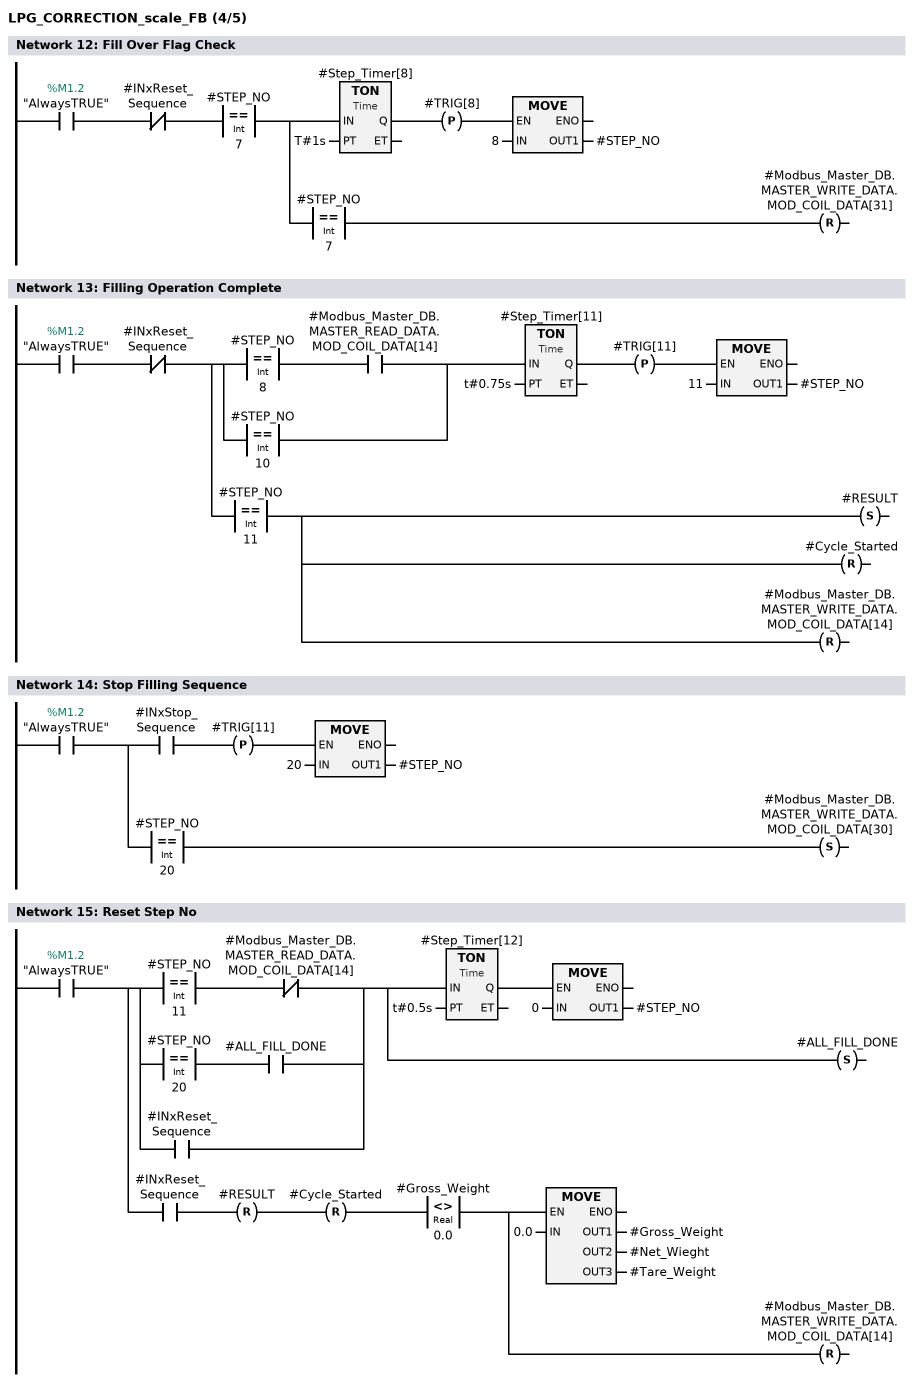
   RUNG wire#powerrail
      Contact( "AlwaysTRUE" )
      I_Contact( #INxReset_Sequence )
      { S7_Templates := "SrcType := Int" } EQ_Contact(in1 := #STEP_NO, in2 := 7)
      wire#w1
      { S7_Templates := "time_type := Time" } #Step_Timer[8].TON(pt := T#1s, et =>)
      P_Trig( #TRIG[8] )
      Move(in := 8, out1 => #STEP_NO)
   END_RUNG
   RUNG wire#w1
      { S7_Templates := "SrcType := Int" } EQ_Contact(in1 := #STEP_NO, in2 := 7)
      R_Coil( #Modbus_Master_DB.MASTER_WRITE_DATA.MOD_COIL_DATA[31] )
   END_RUNG
   // the same network as SCL:
   #_w1 := "AlwaysTRUE" AND NOT #INxReset_Sequence AND (#STEP_NO = 7);
   #Step_Timer[8].TON(IN := #_w1, PT := T#1s);
   #_w2 := #Step_Timer[8].Q AND NOT #TRIG[8];   // rising edge
   #TRIG[8] := #Step_Timer[8].Q;
   IF #_w2 THEN #STEP_NO := 8; END_IF;
   IF #_w1 AND (#STEP_NO = 7) THEN #Modbus_Master_DB.MASTER_WRITE_DATA.MOD_COIL_DATA[31] := FALSE; END_IF;
END_REGION

REGION Network 13: Filling Operation Complete
   RUNG wire#powerrail
      Contact( "AlwaysTRUE" )
      I_Contact( #INxReset_Sequence )
      wire#w1
      { S7_Templates := "SrcType := Int" } EQ_Contact(in1 := #STEP_NO, in2 := 8)
      Contact( #Modbus_Master_DB.MASTER_READ_DATA.MOD_COIL_DATA[14] )
      wire#w2
      { S7_Templates := "time_type := Time" } #Step_Timer[11].TON(pt := t#0.75s, et =>)
      P_Trig( #TRIG[11] )
      Move(in := 11, out1 => #STEP_NO)
   END_RUNG
   RUNG wire#w1
      { S7_Templates := "SrcType := Int" } EQ_Contact(in1 := #STEP_NO, in2 := 10)
   END_RUNG wire#w2
   RUNG wire#w1
      { S7_Templates := "SrcType := Int" } EQ_Contact(in1 := #STEP_NO, in2 := 11)
      wire#w3
      S_Coil( #RESULT )
   END_RUNG
   RUNG wire#w3
      R_Coil( #Cycle_Started )
   END_RUNG
   RUNG wire#w3
      R_Coil( #Modbus_Master_DB.MASTER_WRITE_DATA.MOD_COIL_DATA[14] )
   END_RUNG
   // the same network as SCL:
   #_w1 := "AlwaysTRUE" AND NOT #INxReset_Sequence;
   #Step_Timer[11].TON(IN := #_w1 AND (((#STEP_NO = 8) AND #Modbus_Master_DB.MASTER_READ_DATA.MOD_COIL_DATA[14]) OR (#STEP_NO = 10)),
                       PT := t#0.75s);
   #_w2 := #Step_Timer[11].Q AND NOT #TRIG[11];   // rising edge
   #TRIG[11] := #Step_Timer[11].Q;
   IF #_w2 THEN #STEP_NO := 11; END_IF;
   IF #_w1 AND (#STEP_NO = 11) THEN
       #RESULT := TRUE;
       #Cycle_Started := FALSE;
       #Modbus_Master_DB.MASTER_WRITE_DATA.MOD_COIL_DATA[14] := FALSE;
   END_IF;
END_REGION

REGION Network 14: Stop Filling Sequence
   RUNG wire#powerrail
      Contact( "AlwaysTRUE" )
      wire#w1
      Contact( #INxStop_Sequence )
      P_Trig( #TRIG[11] )
      Move(in := 20, out1 => #STEP_NO)
   END_RUNG
   RUNG wire#w1
      { S7_Templates := "SrcType := Int" } EQ_Contact(in1 := #STEP_NO, in2 := 20)
      S_Coil( #Modbus_Master_DB.MASTER_WRITE_DATA.MOD_COIL_DATA[30] )
   END_RUNG
   // the same network as SCL:
   #_w1 := "AlwaysTRUE" AND #INxStop_Sequence;
   #_w2 := #_w1 AND NOT #TRIG[11];   // rising edge
   #TRIG[11] := #_w1;
   IF #_w2 THEN #STEP_NO := 20; END_IF;
   IF "AlwaysTRUE" AND (#STEP_NO = 20) THEN
       #Modbus_Master_DB.MASTER_WRITE_DATA.MOD_COIL_DATA[30] := TRUE;
   END_IF;
END_REGION

REGION Network 15: Reset Step No
   RUNG wire#powerrail
      Contact( "AlwaysTRUE" )
      wire#w1
      { S7_Templates := "SrcType := Int" } EQ_Contact(in1 := #STEP_NO, in2 := 11)
      I_Contact( #Modbus_Master_DB.MASTER_READ_DATA.MOD_COIL_DATA[14] )
      wire#w2
      { S7_Templates := "time_type := Time" } #Step_Timer[12].TON(pt := t#0.5s, et =>)
      Move(in := 0, out1 => #STEP_NO)
   END_RUNG
   RUNG wire#w1
      { S7_Templates := "SrcType := Int" } EQ_Contact(in1 := #STEP_NO, in2 := 20)
      Contact( #ALL_FILL_DONE )
   END_RUNG wire#w2
   RUNG wire#w1
      Contact( #INxReset_Sequence )
   END_RUNG wire#w2
   RUNG wire#w2
      S_Coil( #ALL_FILL_DONE )
   END_RUNG
   RUNG wire#w1
      Contact( #INxReset_Sequence )
      R_Coil( #RESULT )
      R_Coil( #Cycle_Started )
      { S7_Templates := "SrcType := Real" } NE_Contact(in1 := #Gross_Weight, in2 := 0.0)
      wire#w3
      Move(in := 0.0, out1 => #Gross_Weight, out2 => #Net_Wieght, out3 => #Tare_Weight)
   END_RUNG
   RUNG wire#w3
      R_Coil( #Modbus_Master_DB.MASTER_WRITE_DATA.MOD_COIL_DATA[14] )
   END_RUNG
   // the same network as SCL:
   #_w1 := "AlwaysTRUE" AND (((#STEP_NO = 11) AND NOT #Modbus_Master_DB.MASTER_READ_DATA.MOD_COIL_DATA[14]) OR ((#STEP_NO = 20) AND #ALL_FILL_DONE) OR #INxReset_Sequence);
   #Step_Timer[12].TON(IN := #_w1, PT := t#0.5s);
   IF #Step_Timer[12].Q THEN #STEP_NO := 0; END_IF;
   IF #_w1 THEN #ALL_FILL_DONE := TRUE; END_IF;
   #_w2 := "AlwaysTRUE" AND #INxReset_Sequence;
   IF #_w2 THEN
       #RESULT := FALSE;
       #Cycle_Started := FALSE;
   END_IF;
   #_w3 := #_w2 AND (#Gross_Weight <> 0.0);
   IF #_w3 THEN
       #Gross_Weight := 0.0;
       #Net_Wieght := 0.0;
       #Tare_Weight := 0.0;
       #Modbus_Master_DB.MASTER_WRITE_DATA.MOD_COIL_DATA[14] := FALSE;
   END_IF;
END_REGION

REGION Network 16: Output Mapping
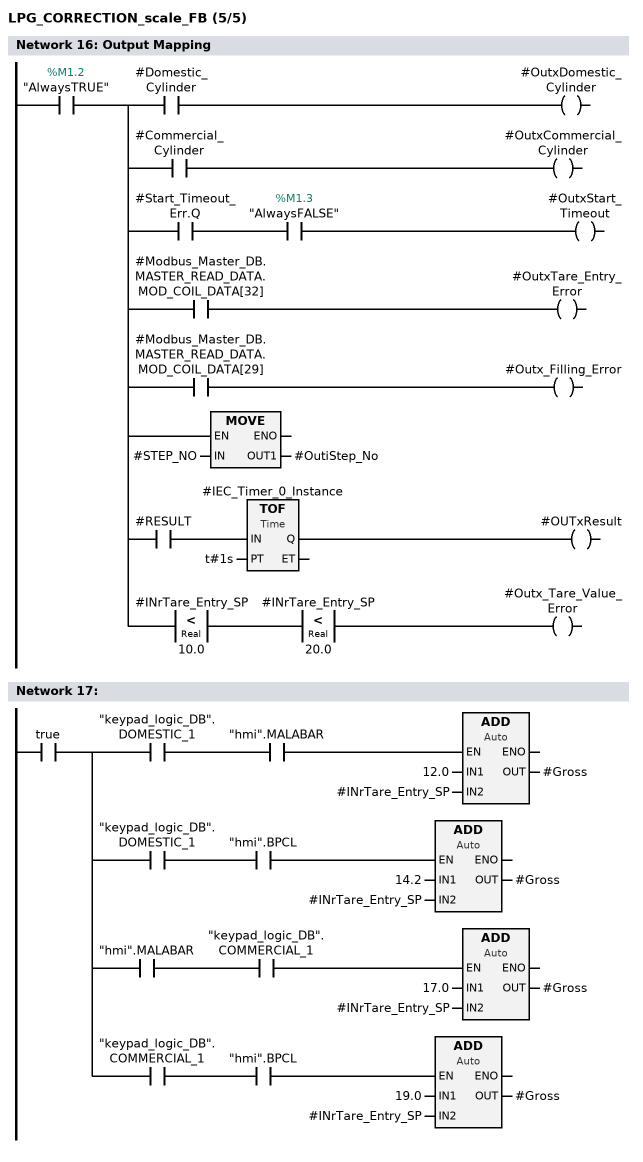
   RUNG wire#powerrail
      Contact( "AlwaysTRUE" )
      wire#w1
      Contact( #Domestic_Cylinder )
      Coil( #OutxDomestic_Cylinder )
   END_RUNG
   RUNG wire#w1
      Contact( #Commercial_Cylinder )
      Coil( #OutxCommercial_Cylinder )
   END_RUNG
   RUNG wire#w1
      Contact( #Start_Timeout_Err.Q )
      Contact( "AlwaysFALSE" )
      Coil( #OutxStart_Timeout )
   END_RUNG
   RUNG wire#w1
      Contact( #Modbus_Master_DB.MASTER_READ_DATA.MOD_COIL_DATA[32] )
      Coil( #OutxTare_Entry_Error )
   END_RUNG
   RUNG wire#w1
      Contact( #Modbus_Master_DB.MASTER_READ_DATA.MOD_COIL_DATA[29] )
      Coil( #Outx_Filling_Error )
   END_RUNG
   RUNG wire#w1
      Move(in := #STEP_NO, out1 => #OutiStep_No)
   END_RUNG
   RUNG wire#w1
      Contact( #RESULT )
      { S7_Templates := "time_type := Time" } #IEC_Timer_0_Instance.TOF(pt := t#1s, et =>)
      Coil( #OUTxResult )
   END_RUNG
   RUNG wire#w1
      { S7_Templates := "SrcType := Real" } LT_Contact(in1 := #INrTare_Entry_SP, in2 := 10.0)
      { S7_Templates := "SrcType := Real" } LT_Contact(in1 := #INrTare_Entry_SP, in2 := 20.0)
      Coil( #Outx_Tare_Value_Error )
   END_RUNG
   // the same network as SCL:
   #OutxDomestic_Cylinder := "AlwaysTRUE" AND #Domestic_Cylinder;
   #OutxCommercial_Cylinder := "AlwaysTRUE" AND #Commercial_Cylinder;
   #OutxStart_Timeout := "AlwaysTRUE" AND #Start_Timeout_Err.Q AND "AlwaysFALSE";
   #OutxTare_Entry_Error := "AlwaysTRUE" AND #Modbus_Master_DB.MASTER_READ_DATA.MOD_COIL_DATA[32];
   #Outx_Filling_Error := "AlwaysTRUE" AND #Modbus_Master_DB.MASTER_READ_DATA.MOD_COIL_DATA[29];
   IF "AlwaysTRUE" THEN #OutiStep_No := #STEP_NO; END_IF;
   #IEC_Timer_0_Instance(IN := "AlwaysTRUE" AND #RESULT, PT := t#1s);   // TOF
   #OUTxResult := #IEC_Timer_0_Instance.Q;
   #Outx_Tare_Value_Error := "AlwaysTRUE" AND (#INrTare_Entry_SP < 10.0) AND (#INrTare_Entry_SP < 20.0);
END_REGION

REGION Network 17
   RUNG wire#powerrail
      Contact( true )
      wire#w1
      Contact( "keypad_logic_DB".DOMESTIC_1 )
      Contact( "hmi".MALABAR )
      Add(in1 := 12.0, in2 := #INrTare_Entry_SP, out => #Gross)
   END_RUNG
   RUNG wire#w1
      Contact( "keypad_logic_DB".DOMESTIC_1 )
      Contact( "hmi".BPCL )
      Add(in1 := 14.2, in2 := #INrTare_Entry_SP, out => #Gross)
   END_RUNG
   RUNG wire#w1
      Contact( "hmi".MALABAR )
      Contact( "keypad_logic_DB".COMMERCIAL_1 )
      Add(in1 := 17.0, in2 := #INrTare_Entry_SP, out => #Gross)
   END_RUNG
   RUNG wire#w1
      Contact( "keypad_logic_DB".COMMERCIAL_1 )
      Contact( "hmi".BPCL )
      Add(in1 := 19.0, in2 := #INrTare_Entry_SP, out => #Gross)
   END_RUNG
   // the same network as SCL:
   IF true AND "keypad_logic_DB".DOMESTIC_1 AND "hmi".MALABAR THEN
       #Gross := 12.0 + #INrTare_Entry_SP;
   END_IF;
   IF true AND "keypad_logic_DB".DOMESTIC_1 AND "hmi".BPCL THEN #Gross := 14.2 + #INrTare_Entry_SP; END_IF;
   IF true AND "hmi".MALABAR AND "keypad_logic_DB".COMMERCIAL_1 THEN
       #Gross := 17.0 + #INrTare_Entry_SP;
   END_IF;
   IF true AND "keypad_logic_DB".COMMERCIAL_1 AND "hmi".BPCL THEN #Gross := 19.0 + #INrTare_Entry_SP; END_IF;
END_REGION
END_FUNCTION_BLOCK

FUNCTION_BLOCK "TCP_CORRECTION_SCALE"   // FB171, LAD
{ S7_Optimized_Access := 'TRUE' }
VERSION : 0.1
// stored: AutoNumber false, IsIECCheckEnabled false, IsRetainMemResEnabled false, MemoryReserve 100, SetENOAutomatically false, UDAEnableTagReadback false
   VAR_OUTPUT
      Modbus_Busy : Bool;
   END_VAR
   VAR_IN_OUT
      Mod_TCP_Setup : "Mod_TCP_Data";
      LPG_Fill_Data : "LPG_FILL_DATA";
   END_VAR
   VAR
      PStep_No : Struct
         MASTER_STEP_NO : "Master_Step_No";
      END_STRUCT;
      Write_Bit_Address : Int;
      TRIG : Array[1..100] of Bool;
      MOD_MASTER1_REQ : Array[1..10] of Bool;
      MOD_MASTER2_REQ : Array[1..10] of Bool;
      MOD_MASTER3_REQ : Array[1..10] of Bool;
      MOD_MASTER4_REQ : Array[1..10] of Bool;
      MOD_MASTER5_REQ : Array[1..10] of Bool;
      MOD_MASTER6_REQ : Array[1..10] of Bool;
      MAS_TRG_EXTN { S7_SetPoint := 'True'} : TOF_TIME;
      Tare_delay { S7_SetPoint := 'True'} : TON_TIME;
   END_VAR
   VAR_TEMP   // added for the SCL form of the ladder/FBD networks
      _w1 : Bool;
      _w2 : Bool;
      _w3 : Bool;
      _w4 : Bool;
   END_VAR
BEGIN

REGION Network 1: FILLING LINE-1 STATION-1
END_REGION

REGION Network 2: Write Master-1 Holding Register Request(Tare Weight Entry)
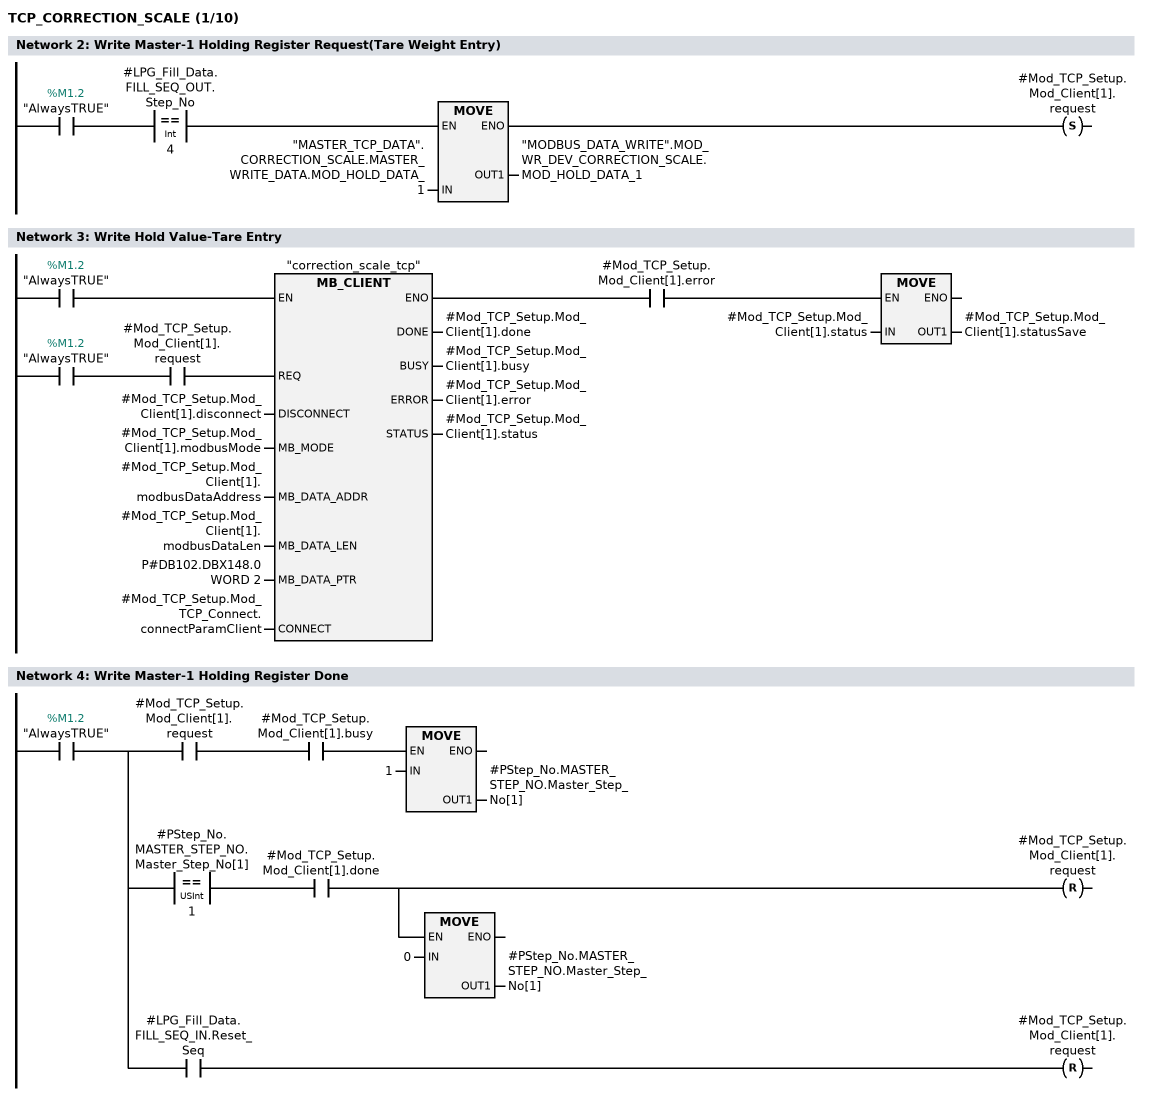
   RUNG wire#powerrail
      Contact( "AlwaysTRUE" )
      { S7_Templates := "SrcType := Int" } EQ_Contact(in1 := #LPG_Fill_Data.FILL_SEQ_OUT.Step_No, in2 := 4)
      Move(in := "MASTER_TCP_DATA".CORRECTION_SCALE.MASTER_WRITE_DATA.MOD_HOLD_DATA_1, out1 => "MODBUS_DATA_WRITE".MOD_WR_DEV_CORRECTION_SCALE.MOD_HOLD_DATA_1)
      S_Coil( #Mod_TCP_Setup.Mod_Client[1].request )
   END_RUNG
   // the same network as SCL:
   IF "AlwaysTRUE" AND (#LPG_Fill_Data.FILL_SEQ_OUT.Step_No = 4) THEN
       "MODBUS_DATA_WRITE".MOD_WR_DEV_CORRECTION_SCALE.MOD_HOLD_DATA_1 := "MASTER_TCP_DATA".CORRECTION_SCALE.MASTER_WRITE_DATA.MOD_HOLD_DATA_1;
       #Mod_TCP_Setup.Mod_Client[1].request := TRUE;
   END_IF;
END_REGION

REGION Network 3: Write Hold Value-Tare Entry
   RUNG wire#powerrail
      Contact( "AlwaysTRUE" )
      "correction_scale_tcp".MB_CLIENT(REQ := wire#w1, DISCONNECT := #Mod_TCP_Setup.Mod_Client[1].disconnect, MB_MODE := #Mod_TCP_Setup.Mod_Client[1].modbusMode, MB_DATA_ADDR := #Mod_TCP_Setup.Mod_Client[1].modbusDataAddress, MB_DATA_LEN := #Mod_TCP_Setup.Mod_Client[1].modbusDataLen, MB_DATA_PTR := P#DB102.DBX148.0 WORD 2, CONNECT := #Mod_TCP_Setup.Mod_TCP_Connect.connectParamClient, DONE => #Mod_TCP_Setup.Mod_Client[1].done, BUSY => #Mod_TCP_Setup.Mod_Client[1].busy, ERROR => #Mod_TCP_Setup.Mod_Client[1].error, STATUS => #Mod_TCP_Setup.Mod_Client[1].status)
      Contact( #Mod_TCP_Setup.Mod_Client[1].error )
      Move(in := #Mod_TCP_Setup.Mod_Client[1].status, out1 => #Mod_TCP_Setup.Mod_Client[1].statusSave)
   END_RUNG
   RUNG wire#powerrail
      Contact( "AlwaysTRUE" )
      Contact( #Mod_TCP_Setup.Mod_Client[1].request )
   END_RUNG wire#w1
   // the same network as SCL:
   "correction_scale_tcp"(EN := "AlwaysTRUE",   // MB_CLIENT
                          REQ := "AlwaysTRUE" AND #Mod_TCP_Setup.Mod_Client[1].request,
                          DISCONNECT := #Mod_TCP_Setup.Mod_Client[1].disconnect,
                          MB_MODE := #Mod_TCP_Setup.Mod_Client[1].modbusMode,
                          MB_DATA_ADDR := #Mod_TCP_Setup.Mod_Client[1].modbusDataAddress,
                          MB_DATA_LEN := #Mod_TCP_Setup.Mod_Client[1].modbusDataLen,
                          MB_DATA_PTR := P#DB102.DBX148.0 WORD 2,
                          CONNECT := #Mod_TCP_Setup.Mod_TCP_Connect.connectParamClient,
                          DONE => #Mod_TCP_Setup.Mod_Client[1].done,
                          BUSY => #Mod_TCP_Setup.Mod_Client[1].busy,
                          ERROR => #Mod_TCP_Setup.Mod_Client[1].error,
                          STATUS => #Mod_TCP_Setup.Mod_Client[1].status,
                          ENO => #_w1);
   IF #_w1 AND #Mod_TCP_Setup.Mod_Client[1].error THEN
       #Mod_TCP_Setup.Mod_Client[1].statusSave := #Mod_TCP_Setup.Mod_Client[1].status;
   END_IF;
END_REGION

REGION Network 4: Write Master-1 Holding Register Done
   RUNG wire#powerrail
      Contact( "AlwaysTRUE" )
      wire#w1
      Contact( #Mod_TCP_Setup.Mod_Client[1].request )
      Contact( #Mod_TCP_Setup.Mod_Client[1].busy )
      Move(in := 1, out1 => #PStep_No.MASTER_STEP_NO.Master_Step_No[1])
   END_RUNG
   RUNG wire#w1
      { S7_Templates := "SrcType := USInt" } EQ_Contact(in1 := #PStep_No.MASTER_STEP_NO.Master_Step_No[1], in2 := 1)
      Contact( #Mod_TCP_Setup.Mod_Client[1].done )
      wire#w2
      R_Coil( #Mod_TCP_Setup.Mod_Client[1].request )
   END_RUNG
   RUNG wire#w2
      Move(in := 0, out1 => #PStep_No.MASTER_STEP_NO.Master_Step_No[1])
   END_RUNG
   RUNG wire#w1
      Contact( #LPG_Fill_Data.FILL_SEQ_IN.Reset_Seq )
      R_Coil( #Mod_TCP_Setup.Mod_Client[1].request )
   END_RUNG
   // the same network as SCL:
   IF "AlwaysTRUE" AND #Mod_TCP_Setup.Mod_Client[1].request AND #Mod_TCP_Setup.Mod_Client[1].busy THEN
       #PStep_No.MASTER_STEP_NO.Master_Step_No[1] := 1;
   END_IF;
   #_w1 := "AlwaysTRUE" AND (#PStep_No.MASTER_STEP_NO.Master_Step_No[1] = 1) AND #Mod_TCP_Setup.Mod_Client[1].done;
   IF #_w1 THEN
       #Mod_TCP_Setup.Mod_Client[1].request := FALSE;
       #PStep_No.MASTER_STEP_NO.Master_Step_No[1] := 0;
   END_IF;
   IF "AlwaysTRUE" AND #LPG_Fill_Data.FILL_SEQ_IN.Reset_Seq THEN
       #Mod_TCP_Setup.Mod_Client[1].request := FALSE;
   END_IF;
END_REGION

REGION Network 5: Modbus Master2 Read Request(Filled Data)
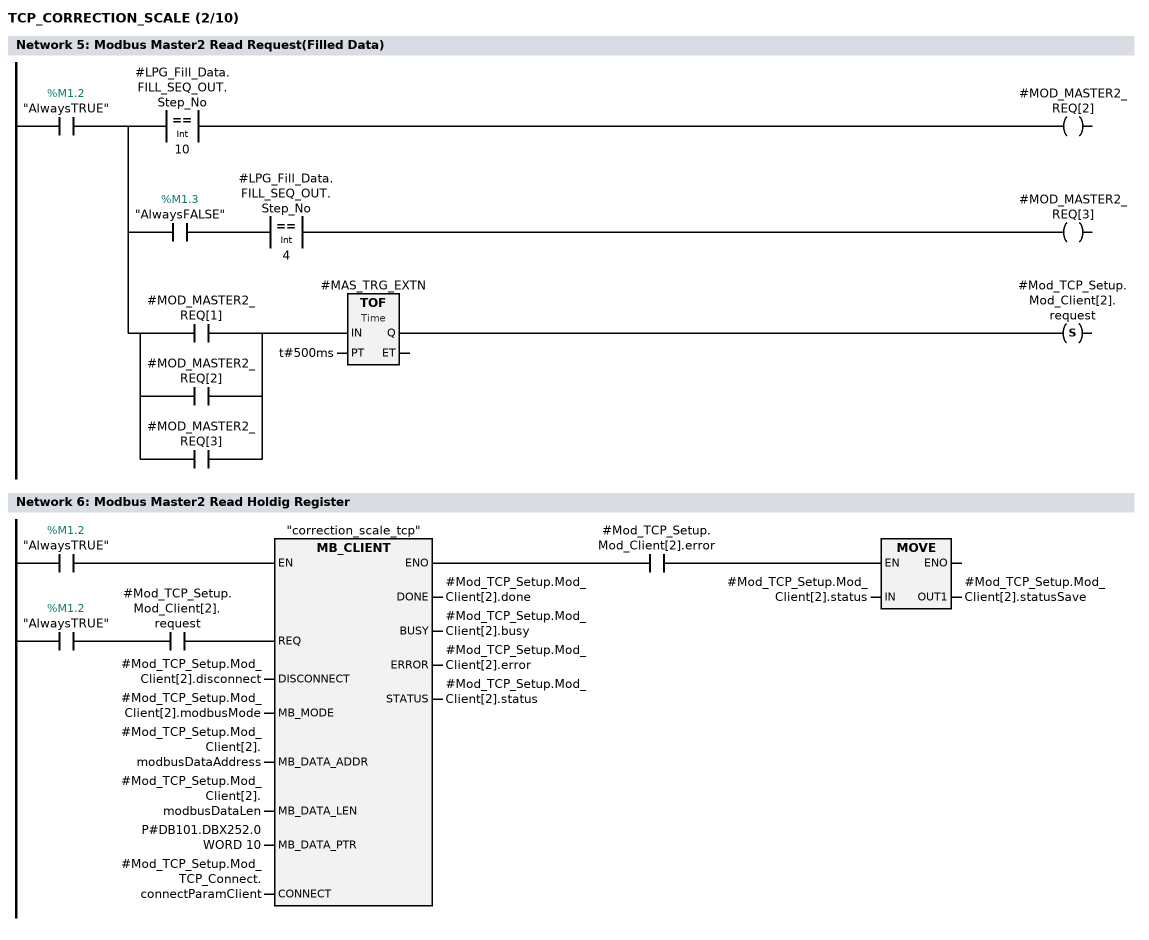
   RUNG wire#powerrail
      Contact( "AlwaysTRUE" )
      wire#w1
      { S7_Templates := "SrcType := Int" } EQ_Contact(in1 := #LPG_Fill_Data.FILL_SEQ_OUT.Step_No, in2 := 10)
      Coil( #MOD_MASTER2_REQ[2] )
   END_RUNG
   RUNG wire#w1
      Contact( "AlwaysFALSE" )
      { S7_Templates := "SrcType := Int" } EQ_Contact(in1 := #LPG_Fill_Data.FILL_SEQ_OUT.Step_No, in2 := 4)
      Coil( #MOD_MASTER2_REQ[3] )
   END_RUNG
   RUNG wire#w1
      Contact( #MOD_MASTER2_REQ[1] )
      wire#w2
      { S7_Templates := "time_type := Time" } #MAS_TRG_EXTN.TOF(pt := t#500ms, et =>)
      S_Coil( #Mod_TCP_Setup.Mod_Client[2].request )
   END_RUNG
   RUNG wire#w1
      Contact( #MOD_MASTER2_REQ[2] )
   END_RUNG wire#w2
   RUNG wire#w1
      Contact( #MOD_MASTER2_REQ[3] )
   END_RUNG wire#w2
   // the same network as SCL:
   #MOD_MASTER2_REQ[2] := "AlwaysTRUE" AND (#LPG_Fill_Data.FILL_SEQ_OUT.Step_No = 10);
   #MOD_MASTER2_REQ[3] := "AlwaysTRUE" AND "AlwaysFALSE" AND (#LPG_Fill_Data.FILL_SEQ_OUT.Step_No = 4);
   #MAS_TRG_EXTN(IN := "AlwaysTRUE" AND (#MOD_MASTER2_REQ[1] OR #MOD_MASTER2_REQ[2] OR #MOD_MASTER2_REQ[3]),   // TOF
                 PT := t#500ms);
   IF #MAS_TRG_EXTN.Q THEN #Mod_TCP_Setup.Mod_Client[2].request := TRUE; END_IF;
END_REGION

